   S701_TL_LOCATE1_ERR.Visu_Adv_Arr[15] := FALSE;
   S701_TL_LOCATE1_ERR.Visu_Ret_Arr[0] := FALSE;
   S701_TL_LOCATE1_ERR.Visu_Ret_Arr[1] := FALSE;
   S701_TL_LOCATE1_ERR.Visu_Ret_Arr[2] := FALSE;
   S701_TL_LOCATE1_ERR.Visu_Ret_Arr[3] := FALSE;
   S701_TL_LOCATE1_ERR.Visu_Ret_Arr[4] := FALSE;
   S701_TL_LOCATE1_ERR.Visu_Ret_Arr[5] := FALSE;
   S701_TL_LOCATE1_ERR.Visu_Ret_Arr[6] := FALSE;
   S701_TL_LOCATE1_ERR.Visu_Ret_Arr[7] := FALSE;
   S701_TL_LOCATE1_ERR.Visu_Ret_Arr[8] := FALSE;
   S701_TL_LOCATE1_ERR.Visu_Ret_Arr[9] := FALSE;
   S701_TL_LOCATE1_ERR.Visu_Ret_Arr[10] := FALSE;
   S701_TL_LOCATE1_ERR.Visu_Ret_Arr[11] := FALSE;
   S701_TL_LOCATE1_ERR.Visu_Ret_Arr[12] := FALSE;
   S701_TL_LOCATE1_ERR.Visu_Ret_Arr[13] := FALSE;
   S701_TL_LOCATE1_ERR.Visu_Ret_Arr[14] := FALSE;
   S701_TL_LOCATE1_ERR.Visu_Ret_Arr[15] := FALSE;
   S701_TL_LOCATE1_ERR.BLK_Move_Ret := 0;
   S701_TL_LOCATE1_ERR.Enable := FALSE;
   S701_TL_LOCATE1_ERR.Adv_End := FALSE;
   S701_TL_LOCATE1_ERR.Ret_End := FALSE;
   S701_TL_LOCATE2_ERR.Enable_Aux := FALSE;
   S701_TL_LOCATE2_ERR.Adv_Amount := 0;
   S701_TL_LOCATE2_ERR.Ret_Amount := 0;
   S701_TL_LOCATE2_ERR.LS_Adv1 := FALSE;
   S701_TL_LOCATE2_ERR.LS_Ret1 := FALSE;
   S701_TL_LOCATE2_ERR.LS_Adv2 := FALSE;
   S701_TL_LOCATE2_ERR.LS_Ret2 := FALSE;
   S701_TL_LOCATE2_ERR.LS_Adv3 := FALSE;
   S701_TL_LOCATE2_ERR.LS_Ret3 := FALSE;
   S701_TL_LOCATE2_ERR.LS_Adv4 := FALSE;
   S701_TL_LOCATE2_ERR.LS_Ret4 := FALSE;
   S701_TL_LOCATE2_ERR.SOL_Adv := FALSE;
   S701_TL_LOCATE2_ERR.SOL_Ret := FALSE;
   S701_TL_LOCATE2_ERR.M_Ready := FALSE;
   S701_TL_LOCATE2_ERR.T_CHK1 := T#0MS;
   S701_TL_LOCATE2_ERR.T_CHK2 := T#0MS;
   S701_TL_LOCATE2_ERR.PB_Lamp_CHK := FALSE;
   S701_TL_LOCATE2_ERR.PB_Error_Rst := FALSE;
   S701_TL_LOCATE2_ERR.M_FLICK := FALSE;
   S701_TL_LOCATE2_ERR.M_Adv_Err := FALSE;
   S701_TL_LOCATE2_ERR.M_Ret_Err := FALSE;
   S701_TL_LOCATE2_ERR.LP_Adv := FALSE;
   S701_TL_LOCATE2_ERR.LP_Ret := FALSE;
   S701_TL_LOCATE2_ERR.Visu_Adv := W#16#0;
   S701_TL_LOCATE2_ERR.Visu_Ret := W#16#0;
   S701_TL_LOCATE2_ERR.Error_T1.IN := FALSE;
   S701_TL_LOCATE2_ERR.Error_T1.PT := T#0MS;
   S701_TL_LOCATE2_ERR.Error_T1.Q := FALSE;
   S701_TL_LOCATE2_ERR.Error_T1.ET := T#0MS;
   S701_TL_LOCATE2_ERR.Error_T1.STATE := B#16#0;
   S701_TL_LOCATE2_ERR.Error_T1.STIME := T#0MS;
   S701_TL_LOCATE2_ERR.Error_T1.ATIME := T#0MS;
   S701_TL_LOCATE2_ERR.Error_T2.IN := FALSE;
   S701_TL_LOCATE2_ERR.Error_T2.PT := T#0MS;
   S701_TL_LOCATE2_ERR.Error_T2.Q := FALSE;
   S701_TL_LOCATE2_ERR.Error_T2.ET := T#0MS;
   S701_TL_LOCATE2_ERR.Error_T2.STATE := B#16#0;
   S701_TL_LOCATE2_ERR.Error_T2.STIME := T#0MS;
   S701_TL_LOCATE2_ERR.Error_T2.ATIME := T#0MS;
   S701_TL_LOCATE2_ERR.CHK_Aux1 := FALSE;
   S701_TL_LOCATE2_ERR.CHK_Aux2 := FALSE;
   S701_TL_LOCATE2_ERR.Error_T1_DN := FALSE;
   S701_TL_LOCATE2_ERR.Error_T2_DN := FALSE;
   S701_TL_LOCATE2_ERR.Adv_Memo := FALSE;
   S701_TL_LOCATE2_ERR.Visu_Adv_Arr[0] := FALSE;
   S701_TL_LOCATE2_ERR.Visu_Adv_Arr[1] := FALSE;
   S701_TL_LOCATE2_ERR.Visu_Adv_Arr[2] := FALSE;
   S701_TL_LOCATE2_ERR.Visu_Adv_Arr[3] := FALSE;
   S701_TL_LOCATE2_ERR.Visu_Adv_Arr[4] := FALSE;
   S701_TL_LOCATE2_ERR.Visu_Adv_Arr[5] := FALSE;
   S701_TL_LOCATE2_ERR.Visu_Adv_Arr[6] := FALSE;
   S701_TL_LOCATE2_ERR.Visu_Adv_Arr[7] := FALSE;
   S701_TL_LOCATE2_ERR.Visu_Adv_Arr[8] := FALSE;
   S701_TL_LOCATE2_ERR.Visu_Adv_Arr[9] := FALSE;
   S701_TL_LOCATE2_ERR.Visu_Adv_Arr[10] := FALSE;
   S701_TL_LOCATE2_ERR.Visu_Adv_Arr[11] := FALSE;
   S701_TL_LOCATE2_ERR.Visu_Adv_Arr[12] := FALSE;
   S701_TL_LOCATE2_ERR.Visu_Adv_Arr[13] := FALSE;
   S701_TL_LOCATE2_ERR.Visu_Adv_Arr[14] := FALSE;
   S701_TL_LOCATE2_ERR.Visu_Adv_Arr[15] := FALSE;
   S701_TL_LOCATE2_ERR.Visu_Ret_Arr[0] := FALSE;
   S701_TL_LOCATE2_ERR.Visu_Ret_Arr[1] := FALSE;
   S701_TL_LOCATE2_ERR.Visu_Ret_Arr[2] := FALSE;
   S701_TL_LOCATE2_ERR.Visu_Ret_Arr[3] := FALSE;
   S701_TL_LOCATE2_ERR.Visu_Ret_Arr[4] := FALSE;
   S701_TL_LOCATE2_ERR.Visu_Ret_Arr[5] := FALSE;
   S701_TL_LOCATE2_ERR.Visu_Ret_Arr[6] := FALSE;
   S701_TL_LOCATE2_ERR.Visu_Ret_Arr[7] := FALSE;
   S701_TL_LOCATE2_ERR.Visu_Ret_Arr[8] := FALSE;
   S701_TL_LOCATE2_ERR.Visu_Ret_Arr[9] := FALSE;
   S701_TL_LOCATE2_ERR.Visu_Ret_Arr[10] := FALSE;
   S701_TL_LOCATE2_ERR.Visu_Ret_Arr[11] := FALSE;
   S701_TL_LOCATE2_ERR.Visu_Ret_Arr[12] := FALSE;
   S701_TL_LOCATE2_ERR.Visu_Ret_Arr[13] := FALSE;
   S701_TL_LOCATE2_ERR.Visu_Ret_Arr[14] := FALSE;
   S701_TL_LOCATE2_ERR.Visu_Ret_Arr[15] := FALSE;
   S701_TL_LOCATE2_ERR.BLK_Move_Ret := 0;
   S701_TL_LOCATE2_ERR.Enable := FALSE;
   S701_TL_LOCATE2_ERR.Adv_End := FALSE;
   S701_TL_LOCATE2_ERR.Ret_End := FALSE;
   S701_TL_LOCATE3_ERR.Enable_Aux := FALSE;
   S701_TL_LOCATE3_ERR.Adv_Amount := 0;
   S701_TL_LOCATE3_ERR.Ret_Amount := 0;
   S701_TL_LOCATE3_ERR.LS_Adv1 := FALSE;
   S701_TL_LOCATE3_ERR.LS_Ret1 := FALSE;
   S701_TL_LOCATE3_ERR.LS_Adv2 := FALSE;
   S701_TL_LOCATE3_ERR.LS_Ret2 := FALSE;
   S701_TL_LOCATE3_ERR.LS_Adv3 := FALSE;
   S701_TL_LOCATE3_ERR.LS_Ret3 := FALSE;
   S701_TL_LOCATE3_ERR.LS_Adv4 := FALSE;
   S701_TL_LOCATE3_ERR.LS_Ret4 := FALSE;
   S701_TL_LOCATE3_ERR.SOL_Adv := FALSE;
   S701_TL_LOCATE3_ERR.SOL_Ret := FALSE;
   S701_TL_LOCATE3_ERR.M_Ready := FALSE;
   S701_TL_LOCATE3_ERR.T_CHK1 := T#0MS;
   S701_TL_LOCATE3_ERR.T_CHK2 := T#0MS;
   S701_TL_LOCATE3_ERR.PB_Lamp_CHK := FALSE;
   S701_TL_LOCATE3_ERR.PB_Error_Rst := FALSE;
   S701_TL_LOCATE3_ERR.M_FLICK := FALSE;
   S701_TL_LOCATE3_ERR.M_Adv_Err := FALSE;
   S701_TL_LOCATE3_ERR.M_Ret_Err := FALSE;
   S701_TL_LOCATE3_ERR.LP_Adv := FALSE;
   S701_TL_LOCATE3_ERR.LP_Ret := FALSE;
   S701_TL_LOCATE3_ERR.Visu_Adv := W#16#0;
   S701_TL_LOCATE3_ERR.Visu_Ret := W#16#0;
   S701_TL_LOCATE3_ERR.Error_T1.IN := FALSE;
   S701_TL_LOCATE3_ERR.Error_T1.PT := T#0MS;
   S701_TL_LOCATE3_ERR.Error_T1.Q := FALSE;
   S701_TL_LOCATE3_ERR.Error_T1.ET := T#0MS;
   S701_TL_LOCATE3_ERR.Error_T1.STATE := B#16#0;
   S701_TL_LOCATE3_ERR.Error_T1.STIME := T#0MS;
   S701_TL_LOCATE3_ERR.Error_T1.ATIME := T#0MS;
   S701_TL_LOCATE3_ERR.Error_T2.IN := FALSE;
   S701_TL_LOCATE3_ERR.Error_T2.PT := T#0MS;
   S701_TL_LOCATE3_ERR.Error_T2.Q := FALSE;
   S701_TL_LOCATE3_ERR.Error_T2.ET := T#0MS;
   S701_TL_LOCATE3_ERR.Error_T2.STATE := B#16#0;
   S701_TL_LOCATE3_ERR.Error_T2.STIME := T#0MS;
   S701_TL_LOCATE3_ERR.Error_T2.ATIME := T#0MS;
   S701_TL_LOCATE3_ERR.CHK_Aux1 := FALSE;
   S701_TL_LOCATE3_ERR.CHK_Aux2 := FALSE;
   S701_TL_LOCATE3_ERR.Error_T1_DN := FALSE;
   S701_TL_LOCATE3_ERR.Error_T2_DN := FALSE;
   S701_TL_LOCATE3_ERR.Adv_Memo := FALSE;
   S701_TL_LOCATE3_ERR.Visu_Adv_Arr[0] := FALSE;
   S701_TL_LOCATE3_ERR.Visu_Adv_Arr[1] := FALSE;
   S701_TL_LOCATE3_ERR.Visu_Adv_Arr[2] := FALSE;
   S701_TL_LOCATE3_ERR.Visu_Adv_Arr[3] := FALSE;
   S701_TL_LOCATE3_ERR.Visu_Adv_Arr[4] := FALSE;
   S701_TL_LOCATE3_ERR.Visu_Adv_Arr[5] := FALSE;
   S701_TL_LOCATE3_ERR.Visu_Adv_Arr[6] := FALSE;
   S701_TL_LOCATE3_ERR.Visu_Adv_Arr[7] := FALSE;
   S701_TL_LOCATE3_ERR.Visu_Adv_Arr[8] := FALSE;
   S701_TL_LOCATE3_ERR.Visu_Adv_Arr[9] := FALSE;
   S701_TL_LOCATE3_ERR.Visu_Adv_Arr[10] := FALSE;
   S701_TL_LOCATE3_ERR.Visu_Adv_Arr[11] := FALSE;
   S701_TL_LOCATE3_ERR.Visu_Adv_Arr[12] := FALSE;
   S701_TL_LOCATE3_ERR.Visu_Adv_Arr[13] := FALSE;
   S701_TL_LOCATE3_ERR.Visu_Adv_Arr[14] := FALSE;
   S701_TL_LOCATE3_ERR.Visu_Adv_Arr[15] := FALSE;
   S701_TL_LOCATE3_ERR.Visu_Ret_Arr[0] := FALSE;
   S701_TL_LOCATE3_ERR.Visu_Ret_Arr[1] := FALSE;
   S701_TL_LOCATE3_ERR.Visu_Ret_Arr[2] := FALSE;
   S701_TL_LOCATE3_ERR.Visu_Ret_Arr[3] := FALSE;
   S701_TL_LOCATE3_ERR.Visu_Ret_Arr[4] := FALSE;
   S701_TL_LOCATE3_ERR.Visu_Ret_Arr[5] := FALSE;
   S701_TL_LOCATE3_ERR.Visu_Ret_Arr[6] := FALSE;
   S701_TL_LOCATE3_ERR.Visu_Ret_Arr[7] := FALSE;
   S701_TL_LOCATE3_ERR.Visu_Ret_Arr[8] := FALSE;
   S701_TL_LOCATE3_ERR.Visu_Ret_Arr[9] := FALSE;
   S701_TL_LOCATE3_ERR.Visu_Ret_Arr[10] := FALSE;
   S701_TL_LOCATE3_ERR.Visu_Ret_Arr[11] := FALSE;
   S701_TL_LOCATE3_ERR.Visu_Ret_Arr[12] := FALSE;
   S701_TL_LOCATE3_ERR.Visu_Ret_Arr[13] := FALSE;
   S701_TL_LOCATE3_ERR.Visu_Ret_Arr[14] := FALSE;
   S701_TL_LOCATE3_ERR.Visu_Ret_Arr[15] := FALSE;
   S701_TL_LOCATE3_ERR.BLK_Move_Ret := 0;
   S701_TL_LOCATE3_ERR.Enable := FALSE;
   S701_TL_LOCATE3_ERR.Adv_End := FALSE;
   S701_TL_LOCATE3_ERR.Ret_End := FALSE;
   S701_TL_1_CLAMP1_ERR.Enable_Aux := FALSE;
   S701_TL_1_CLAMP1_ERR.Adv_Amount := 0;
   S701_TL_1_CLAMP1_ERR.Ret_Amount := 0;
   S701_TL_1_CLAMP1_ERR.LS_Adv1 := FALSE;
   S701_TL_1_CLAMP1_ERR.LS_Ret1 := FALSE;
   S701_TL_1_CLAMP1_ERR.LS_Adv2 := FALSE;
   S701_TL_1_CLAMP1_ERR.LS_Ret2 := FALSE;
   S701_TL_1_CLAMP1_ERR.LS_Adv3 := FALSE;
   S701_TL_1_CLAMP1_ERR.LS_Ret3 := FALSE;
   S701_TL_1_CLAMP1_ERR.LS_Adv4 := FALSE;
   S701_TL_1_CLAMP1_ERR.LS_Ret4 := FALSE;
   S701_TL_1_CLAMP1_ERR.LS_Adv5 := FALSE;
   S701_TL_1_CLAMP1_ERR.LS_Ret5 := FALSE;
   S701_TL_1_CLAMP1_ERR.LS_Adv6 := FALSE;
   S701_TL_1_CLAMP1_ERR.LS_Ret6 := FALSE;
   S701_TL_1_CLAMP1_ERR.LS_Adv7 := FALSE;
   S701_TL_1_CLAMP1_ERR.LS_Ret7 := FALSE;
   S701_TL_1_CLAMP1_ERR.LS_Adv8 := FALSE;
   S701_TL_1_CLAMP1_ERR.LS_Ret8 := FALSE;
   S701_TL_1_CLAMP1_ERR.SOL_Adv := FALSE;
   S701_TL_1_CLAMP1_ERR.SOL_Ret := FALSE;
   S701_TL_1_CLAMP1_ERR.M_Ready := FALSE;
   S701_TL_1_CLAMP1_ERR.T_CHK1 := T#0MS;
   S701_TL_1_CLAMP1_ERR.T_CHK2 := T#0MS;
   S701_TL_1_CLAMP1_ERR.PB_Lamp_CHK := FALSE;
   S701_TL_1_CLAMP1_ERR.PB_Error_Rst := FALSE;
   S701_TL_1_CLAMP1_ERR.M_FLICK := FALSE;
   S701_TL_1_CLAMP1_ERR.M_Adv_Err := FALSE;
   S701_TL_1_CLAMP1_ERR.M_Ret_Err := FALSE;
   S701_TL_1_CLAMP1_ERR.LP_Adv := FALSE;
   S701_TL_1_CLAMP1_ERR.LP_Ret := FALSE;
   S701_TL_1_CLAMP1_ERR.Visu_Adv := W#16#0;
   S701_TL_1_CLAMP1_ERR.Visu_Ret := W#16#0;
   S701_TL_1_CLAMP1_ERR.Error_T1.IN := FALSE;
   S701_TL_1_CLAMP1_ERR.Error_T1.PT := T#0MS;
   S701_TL_1_CLAMP1_ERR.Error_T1.Q := FALSE;
   S701_TL_1_CLAMP1_ERR.Error_T1.ET := T#0MS;
   S701_TL_1_CLAMP1_ERR.Error_T1.STATE := B#16#0;
   S701_TL_1_CLAMP1_ERR.Error_T1.STIME := T#0MS;
   S701_TL_1_CLAMP1_ERR.Error_T1.ATIME := T#0MS;
   S701_TL_1_CLAMP1_ERR.Error_T2.IN := FALSE;
   S701_TL_1_CLAMP1_ERR.Error_T2.PT := T#0MS;
   S701_TL_1_CLAMP1_ERR.Error_T2.Q := FALSE;
   S701_TL_1_CLAMP1_ERR.Error_T2.ET := T#0MS;
   S701_TL_1_CLAMP1_ERR.Error_T2.STATE := B#16#0;
   S701_TL_1_CLAMP1_ERR.Error_T2.STIME := T#0MS;
   S701_TL_1_CLAMP1_ERR.Error_T2.ATIME := T#0MS;
   S701_TL_1_CLAMP1_ERR.Adv_End_Aux := FALSE;
   S701_TL_1_CLAMP1_ERR.Ret_End_Aux := FALSE;
   S701_TL_1_CLAMP1_ERR.CHK_Aux1 := FALSE;
   S701_TL_1_CLAMP1_ERR.CHK_Aux2 := FALSE;
   S701_TL_1_CLAMP1_ERR.Error_T1_DN := FALSE;
   S701_TL_1_CLAMP1_ERR.Error_T2_DN := FALSE;
   S701_TL_1_CLAMP1_ERR.Adv_Memo := FALSE;
   S701_TL_1_CLAMP1_ERR.Visu_Adv_Arr[0] := FALSE;
   S701_TL_1_CLAMP1_ERR.Visu_Adv_Arr[1] := FALSE;
   S701_TL_1_CLAMP1_ERR.Visu_Adv_Arr[2] := FALSE;
   S701_TL_1_CLAMP1_ERR.Visu_Adv_Arr[3] := FALSE;
   S701_TL_1_CLAMP1_ERR.Visu_Adv_Arr[4] := FALSE;
   S701_TL_1_CLAMP1_ERR.Visu_Adv_Arr[5] := FALSE;
   S701_TL_1_CLAMP1_ERR.Visu_Adv_Arr[6] := FALSE;
   S701_TL_1_CLAMP1_ERR.Visu_Adv_Arr[7] := FALSE;
   S701_TL_1_CLAMP1_ERR.Visu_Adv_Arr[8] := FALSE;
   S701_TL_1_CLAMP1_ERR.Visu_Adv_Arr[9] := FALSE;
   S701_TL_1_CLAMP1_ERR.Visu_Adv_Arr[10] := FALSE;
   S701_TL_1_CLAMP1_ERR.Visu_Adv_Arr[11] := FALSE;
   S701_TL_1_CLAMP1_ERR.Visu_Adv_Arr[12] := FALSE;
   S701_TL_1_CLAMP1_ERR.Visu_Adv_Arr[13] := FALSE;
   S701_TL_1_CLAMP1_ERR.Visu_Adv_Arr[14] := FALSE;
   S701_TL_1_CLAMP1_ERR.Visu_Adv_Arr[15] := FALSE;
   S701_TL_1_CLAMP1_ERR.Visu_Ret_Arr[0] := FALSE;
   S701_TL_1_CLAMP1_ERR.Visu_Ret_Arr[1] := FALSE;
   S701_TL_1_CLAMP1_ERR.Visu_Ret_Arr[2] := FALSE;
   S701_TL_1_CLAMP1_ERR.Visu_Ret_Arr[3] := FALSE;
   S701_TL_1_CLAMP1_ERR.Visu_Ret_Arr[4] := FALSE;
   S701_TL_1_CLAMP1_ERR.Visu_Ret_Arr[5] := FALSE;
   S701_TL_1_CLAMP1_ERR.Visu_Ret_Arr[6] := FALSE;
   S701_TL_1_CLAMP1_ERR.Visu_Ret_Arr[7] := FALSE;
   S701_TL_1_CLAMP1_ERR.Visu_Ret_Arr[8] := FALSE;
   S701_TL_1_CLAMP1_ERR.Visu_Ret_Arr[9] := FALSE;
   S701_TL_1_CLAMP1_ERR.Visu_Ret_Arr[10] := FALSE;
   S701_TL_1_CLAMP1_ERR.Visu_Ret_Arr[11] := FALSE;
   S701_TL_1_CLAMP1_ERR.Visu_Ret_Arr[12] := FALSE;
   S701_TL_1_CLAMP1_ERR.Visu_Ret_Arr[13] := FALSE;
   S701_TL_1_CLAMP1_ERR.Visu_Ret_Arr[14] := FALSE;
   S701_TL_1_CLAMP1_ERR.Visu_Ret_Arr[15] := FALSE;
   S701_TL_1_CLAMP1_ERR.BLK_Move_Ret := 0;
   S701_TL_1_CLAMP1_ERR.Enable := FALSE;
   S701_TL_1_CLAMP1_ERR.Adv_End := FALSE;
   S701_TL_1_CLAMP1_ERR.Ret_End := FALSE;
   S701_TL_1_CLAMP2_ERR.Enable_Aux := FALSE;
   S701_TL_1_CLAMP2_ERR.Adv_Amount := 0;
   S701_TL_1_CLAMP2_ERR.Ret_Amount := 0;
   S701_TL_1_CLAMP2_ERR.LS_Adv1 := FALSE;
   S701_TL_1_CLAMP2_ERR.LS_Ret1 := FALSE;
   S701_TL_1_CLAMP2_ERR.LS_Adv2 := FALSE;
   S701_TL_1_CLAMP2_ERR.LS_Ret2 := FALSE;
   S701_TL_1_CLAMP2_ERR.LS_Adv3 := FALSE;
   S701_TL_1_CLAMP2_ERR.LS_Ret3 := FALSE;
   S701_TL_1_CLAMP2_ERR.LS_Adv4 := FALSE;
   S701_TL_1_CLAMP2_ERR.LS_Ret4 := FALSE;
   S701_TL_1_CLAMP2_ERR.LS_Adv5 := FALSE;
   S701_TL_1_CLAMP2_ERR.LS_Ret5 := FALSE;
   S701_TL_1_CLAMP2_ERR.LS_Adv6 := FALSE;
   S701_TL_1_CLAMP2_ERR.LS_Ret6 := FALSE;
   S701_TL_1_CLAMP2_ERR.LS_Adv7 := FALSE;
   S701_TL_1_CLAMP2_ERR.LS_Ret7 := FALSE;
   S701_TL_1_CLAMP2_ERR.LS_Adv8 := FALSE;
   S701_TL_1_CLAMP2_ERR.LS_Ret8 := FALSE;
   S701_TL_1_CLAMP2_ERR.SOL_Adv := FALSE;
   S701_TL_1_CLAMP2_ERR.SOL_Ret := FALSE;
   S701_TL_1_CLAMP2_ERR.M_Ready := FALSE;
   S701_TL_1_CLAMP2_ERR.T_CHK1 := T#0MS;
   S701_TL_1_CLAMP2_ERR.T_CHK2 := T#0MS;
   S701_TL_1_CLAMP2_ERR.PB_Lamp_CHK := FALSE;
   S701_TL_1_CLAMP2_ERR.PB_Error_Rst := FALSE;
   S701_TL_1_CLAMP2_ERR.M_FLICK := FALSE;
   S701_TL_1_CLAMP2_ERR.M_Adv_Err := FALSE;
   S701_TL_1_CLAMP2_ERR.M_Ret_Err := FALSE;
   S701_TL_1_CLAMP2_ERR.LP_Adv := FALSE;
   S701_TL_1_CLAMP2_ERR.LP_Ret := FALSE;
   S701_TL_1_CLAMP2_ERR.Visu_Adv := W#16#0;
   S701_TL_1_CLAMP2_ERR.Visu_Ret := W#16#0;
   S701_TL_1_CLAMP2_ERR.Error_T1.IN := FALSE;
   S701_TL_1_CLAMP2_ERR.Error_T1.PT := T#0MS;
   S701_TL_1_CLAMP2_ERR.Error_T1.Q := FALSE;
   S701_TL_1_CLAMP2_ERR.Error_T1.ET := T#0MS;
   S701_TL_1_CLAMP2_ERR.Error_T1.STATE := B#16#0;
   S701_TL_1_CLAMP2_ERR.Error_T1.STIME := T#0MS;
   S701_TL_1_CLAMP2_ERR.Error_T1.ATIME := T#0MS;
   S701_TL_1_CLAMP2_ERR.Error_T2.IN := FALSE;
   S701_TL_1_CLAMP2_ERR.Error_T2.PT := T#0MS;
   S701_TL_1_CLAMP2_ERR.Error_T2.Q := FALSE;
   S701_TL_1_CLAMP2_ERR.Error_T2.ET := T#0MS;
   S701_TL_1_CLAMP2_ERR.Error_T2.STATE := B#16#0;
   S701_TL_1_CLAMP2_ERR.Error_T2.STIME := T#0MS;
   S701_TL_1_CLAMP2_ERR.Error_T2.ATIME := T#0MS;
   S701_TL_1_CLAMP2_ERR.Adv_End_Aux := FALSE;
   S701_TL_1_CLAMP2_ERR.Ret_End_Aux := FALSE;
   S701_TL_1_CLAMP2_ERR.CHK_Aux1 := FALSE;
   S701_TL_1_CLAMP2_ERR.CHK_Aux2 := FALSE;
   S701_TL_1_CLAMP2_ERR.Error_T1_DN := FALSE;
   S701_TL_1_CLAMP2_ERR.Error_T2_DN := FALSE;
   S701_TL_1_CLAMP2_ERR.Adv_Memo := FALSE;
   S701_TL_1_CLAMP2_ERR.Visu_Adv_Arr[0] := FALSE;
   S701_TL_1_CLAMP2_ERR.Visu_Adv_Arr[1] := FALSE;
   S701_TL_1_CLAMP2_ERR.Visu_Adv_Arr[2] := FALSE;
   S701_TL_1_CLAMP2_ERR.Visu_Adv_Arr[3] := FALSE;
   S701_TL_1_CLAMP2_ERR.Visu_Adv_Arr[4] := FALSE;
   S701_TL_1_CLAMP2_ERR.Visu_Adv_Arr[5] := FALSE;
   S701_TL_1_CLAMP2_ERR.Visu_Adv_Arr[6] := FALSE;
   S701_TL_1_CLAMP2_ERR.Visu_Adv_Arr[7] := FALSE;
   S701_TL_1_CLAMP2_ERR.Visu_Adv_Arr[8] := FALSE;
   S701_TL_1_CLAMP2_ERR.Visu_Adv_Arr[9] := FALSE;
   S701_TL_1_CLAMP2_ERR.Visu_Adv_Arr[10] := FALSE;
   S701_TL_1_CLAMP2_ERR.Visu_Adv_Arr[11] := FALSE;
   S701_TL_1_CLAMP2_ERR.Visu_Adv_Arr[12] := FALSE;
   S701_TL_1_CLAMP2_ERR.Visu_Adv_Arr[13] := FALSE;
   S701_TL_1_CLAMP2_ERR.Visu_Adv_Arr[14] := FALSE;
   S701_TL_1_CLAMP2_ERR.Visu_Adv_Arr[15] := FALSE;
   S701_TL_1_CLAMP2_ERR.Visu_Ret_Arr[0] := FALSE;
   S701_TL_1_CLAMP2_ERR.Visu_Ret_Arr[1] := FALSE;
   S701_TL_1_CLAMP2_ERR.Visu_Ret_Arr[2] := FALSE;
   S701_TL_1_CLAMP2_ERR.Visu_Ret_Arr[3] := FALSE;
   S701_TL_1_CLAMP2_ERR.Visu_Ret_Arr[4] := FALSE;
   S701_TL_1_CLAMP2_ERR.Visu_Ret_Arr[5] := FALSE;
   S701_TL_1_CLAMP2_ERR.Visu_Ret_Arr[6] := FALSE;
   S701_TL_1_CLAMP2_ERR.Visu_Ret_Arr[7] := FALSE;
   S701_TL_1_CLAMP2_ERR.Visu_Ret_Arr[8] := FALSE;
   S701_TL_1_CLAMP2_ERR.Visu_Ret_Arr[9] := FALSE;
   S701_TL_1_CLAMP2_ERR.Visu_Ret_Arr[10] := FALSE;
   S701_TL_1_CLAMP2_ERR.Visu_Ret_Arr[11] := FALSE;
   S701_TL_1_CLAMP2_ERR.Visu_Ret_Arr[12] := FALSE;
   S701_TL_1_CLAMP2_ERR.Visu_Ret_Arr[13] := FALSE;
   S701_TL_1_CLAMP2_ERR.Visu_Ret_Arr[14] := FALSE;
   S701_TL_1_CLAMP2_ERR.Visu_Ret_Arr[15] := FALSE;
   S701_TL_1_CLAMP2_ERR.BLK_Move_Ret := 0;
   S701_TL_1_CLAMP2_ERR.Enable := FALSE;
   S701_TL_1_CLAMP2_ERR.Adv_End := FALSE;
   S701_TL_1_CLAMP2_ERR.Ret_End := FALSE;
   S701_TL_2_CLAMP_ERR.Enable_Aux := FALSE;
   S701_TL_2_CLAMP_ERR.Adv_Amount := 0;
   S701_TL_2_CLAMP_ERR.Ret_Amount := 0;
   S701_TL_2_CLAMP_ERR.LS_Adv1 := FALSE;
   S701_TL_2_CLAMP_ERR.LS_Ret1 := FALSE;
   S701_TL_2_CLAMP_ERR.LS_Adv2 := FALSE;
   S701_TL_2_CLAMP_ERR.LS_Ret2 := FALSE;
   S701_TL_2_CLAMP_ERR.LS_Adv3 := FALSE;
   S701_TL_2_CLAMP_ERR.LS_Ret3 := FALSE;
   S701_TL_2_CLAMP_ERR.LS_Adv4 := FALSE;
   S701_TL_2_CLAMP_ERR.LS_Ret4 := FALSE;
   S701_TL_2_CLAMP_ERR.LS_Adv5 := FALSE;
   S701_TL_2_CLAMP_ERR.LS_Ret5 := FALSE;
   S701_TL_2_CLAMP_ERR.LS_Adv6 := FALSE;
   S701_TL_2_CLAMP_ERR.LS_Ret6 := FALSE;
   S701_TL_2_CLAMP_ERR.LS_Adv7 := FALSE;
   S701_TL_2_CLAMP_ERR.LS_Ret7 := FALSE;
   S701_TL_2_CLAMP_ERR.LS_Adv8 := FALSE;
   S701_TL_2_CLAMP_ERR.LS_Ret8 := FALSE;
   S701_TL_2_CLAMP_ERR.SOL_Adv := FALSE;
   S701_TL_2_CLAMP_ERR.SOL_Ret := FALSE;
   S701_TL_2_CLAMP_ERR.M_Ready := FALSE;
   S701_TL_2_CLAMP_ERR.T_CHK1 := T#0MS;
   S701_TL_2_CLAMP_ERR.T_CHK2 := T#0MS;
   S701_TL_2_CLAMP_ERR.PB_Lamp_CHK := FALSE;
   S701_TL_2_CLAMP_ERR.PB_Error_Rst := FALSE;
   S701_TL_2_CLAMP_ERR.M_FLICK := FALSE;
   S701_TL_2_CLAMP_ERR.M_Adv_Err := FALSE;
   S701_TL_2_CLAMP_ERR.M_Ret_Err := FALSE;
   S701_TL_2_CLAMP_ERR.LP_Adv := FALSE;
   S701_TL_2_CLAMP_ERR.LP_Ret := FALSE;
   S701_TL_2_CLAMP_ERR.Visu_Adv := W#16#0;
   S701_TL_2_CLAMP_ERR.Visu_Ret := W#16#0;
   S701_TL_2_CLAMP_ERR.Error_T1.IN := FALSE;
   S701_TL_2_CLAMP_ERR.Error_T1.PT := T#0MS;
   S701_TL_2_CLAMP_ERR.Error_T1.Q := FALSE;
   S701_TL_2_CLAMP_ERR.Error_T1.ET := T#0MS;
   S701_TL_2_CLAMP_ERR.Error_T1.STATE := B#16#0;
   S701_TL_2_CLAMP_ERR.Error_T1.STIME := T#0MS;
   S701_TL_2_CLAMP_ERR.Error_T1.ATIME := T#0MS;
   S701_TL_2_CLAMP_ERR.Error_T2.IN := FALSE;
   S701_TL_2_CLAMP_ERR.Error_T2.PT := T#0MS;
   S701_TL_2_CLAMP_ERR.Error_T2.Q := FALSE;
   S701_TL_2_CLAMP_ERR.Error_T2.ET := T#0MS;
   S701_TL_2_CLAMP_ERR.Error_T2.STATE := B#16#0;
   S701_TL_2_CLAMP_ERR.Error_T2.STIME := T#0MS;
   S701_TL_2_CLAMP_ERR.Error_T2.ATIME := T#0MS;
   S701_TL_2_CLAMP_ERR.Adv_End_Aux := FALSE;
   S701_TL_2_CLAMP_ERR.Ret_End_Aux := FALSE;
   S701_TL_2_CLAMP_ERR.CHK_Aux1 := FALSE;
   S701_TL_2_CLAMP_ERR.CHK_Aux2 := FALSE;
   S701_TL_2_CLAMP_ERR.Error_T1_DN := FALSE;
   S701_TL_2_CLAMP_ERR.Error_T2_DN := FALSE;
   S701_TL_2_CLAMP_ERR.Adv_Memo := FALSE;
   S701_TL_2_CLAMP_ERR.Visu_Adv_Arr[0] := FALSE;
   S701_TL_2_CLAMP_ERR.Visu_Adv_Arr[1] := FALSE;
   S701_TL_2_CLAMP_ERR.Visu_Adv_Arr[2] := FALSE;
   S701_TL_2_CLAMP_ERR.Visu_Adv_Arr[3] := FALSE;
   S701_TL_2_CLAMP_ERR.Visu_Adv_Arr[4] := FALSE;
   S701_TL_2_CLAMP_ERR.Visu_Adv_Arr[5] := FALSE;
   S701_TL_2_CLAMP_ERR.Visu_Adv_Arr[6] := FALSE;
   S701_TL_2_CLAMP_ERR.Visu_Adv_Arr[7] := FALSE;
   S701_TL_2_CLAMP_ERR.Visu_Adv_Arr[8] := FALSE;
   S701_TL_2_CLAMP_ERR.Visu_Adv_Arr[9] := FALSE;
   S701_TL_2_CLAMP_ERR.Visu_Adv_Arr[10] := FALSE;
   S701_TL_2_CLAMP_ERR.Visu_Adv_Arr[11] := FALSE;
   S701_TL_2_CLAMP_ERR.Visu_Adv_Arr[12] := FALSE;
   S701_TL_2_CLAMP_ERR.Visu_Adv_Arr[13] := FALSE;
   S701_TL_2_CLAMP_ERR.Visu_Adv_Arr[14] := FALSE;
   S701_TL_2_CLAMP_ERR.Visu_Adv_Arr[15] := FALSE;
   S701_TL_2_CLAMP_ERR.Visu_Ret_Arr[0] := FALSE;
   S701_TL_2_CLAMP_ERR.Visu_Ret_Arr[1] := FALSE;
   S701_TL_2_CLAMP_ERR.Visu_Ret_Arr[2] := FALSE;
   S701_TL_2_CLAMP_ERR.Visu_Ret_Arr[3] := FALSE;
   S701_TL_2_CLAMP_ERR.Visu_Ret_Arr[4] := FALSE;
   S701_TL_2_CLAMP_ERR.Visu_Ret_Arr[5] := FALSE;
   S701_TL_2_CLAMP_ERR.Visu_Ret_Arr[6] := FALSE;
   S701_TL_2_CLAMP_ERR.Visu_Ret_Arr[7] := FALSE;
   S701_TL_2_CLAMP_ERR.Visu_Ret_Arr[8] := FALSE;
   S701_TL_2_CLAMP_ERR.Visu_Ret_Arr[9] := FALSE;
   S701_TL_2_CLAMP_ERR.Visu_Ret_Arr[10] := FALSE;
   S701_TL_2_CLAMP_ERR.Visu_Ret_Arr[11] := FALSE;
   S701_TL_2_CLAMP_ERR.Visu_Ret_Arr[12] := FALSE;
   S701_TL_2_CLAMP_ERR.Visu_Ret_Arr[13] := FALSE;
   S701_TL_2_CLAMP_ERR.Visu_Ret_Arr[14] := FALSE;
   S701_TL_2_CLAMP_ERR.Visu_Ret_Arr[15] := FALSE;
   S701_TL_2_CLAMP_ERR.BLK_Move_Ret := 0;
   S701_TL_2_CLAMP_ERR.Enable := FALSE;
   S701_TL_2_CLAMP_ERR.Adv_End := FALSE;
   S701_TL_2_CLAMP_ERR.Ret_End := FALSE;
   S701_TL_3_CLAMP_ERR.Enable_Aux := FALSE;
   S701_TL_3_CLAMP_ERR.Adv_Amount := 0;
   S701_TL_3_CLAMP_ERR.Ret_Amount := 0;
   S701_TL_3_CLAMP_ERR.LS_Adv1 := FALSE;
   S701_TL_3_CLAMP_ERR.LS_Ret1 := FALSE;
   S701_TL_3_CLAMP_ERR.LS_Adv2 := FALSE;
   S701_TL_3_CLAMP_ERR.LS_Ret2 := FALSE;
   S701_TL_3_CLAMP_ERR.LS_Adv3 := FALSE;
   S701_TL_3_CLAMP_ERR.LS_Ret3 := FALSE;
   S701_TL_3_CLAMP_ERR.LS_Adv4 := FALSE;
   S701_TL_3_CLAMP_ERR.LS_Ret4 := FALSE;
   S701_TL_3_CLAMP_ERR.LS_Adv5 := FALSE;
   S701_TL_3_CLAMP_ERR.LS_Ret5 := FALSE;
   S701_TL_3_CLAMP_ERR.LS_Adv6 := FALSE;
   S701_TL_3_CLAMP_ERR.LS_Ret6 := FALSE;
   S701_TL_3_CLAMP_ERR.LS_Adv7 := FALSE;
   S701_TL_3_CLAMP_ERR.LS_Ret7 := FALSE;
   S701_TL_3_CLAMP_ERR.LS_Adv8 := FALSE;
   S701_TL_3_CLAMP_ERR.LS_Ret8 := FALSE;
   S701_TL_3_CLAMP_ERR.SOL_Adv := FALSE;
   S701_TL_3_CLAMP_ERR.SOL_Ret := FALSE;
   S701_TL_3_CLAMP_ERR.M_Ready := FALSE;
   S701_TL_3_CLAMP_ERR.T_CHK1 := T#0MS;
   S701_TL_3_CLAMP_ERR.T_CHK2 := T#0MS;
   S701_TL_3_CLAMP_ERR.PB_Lamp_CHK := FALSE;
   S701_TL_3_CLAMP_ERR.PB_Error_Rst := FALSE;
   S701_TL_3_CLAMP_ERR.M_FLICK := FALSE;
   S701_TL_3_CLAMP_ERR.M_Adv_Err := FALSE;
   S701_TL_3_CLAMP_ERR.M_Ret_Err := FALSE;
   S701_TL_3_CLAMP_ERR.LP_Adv := FALSE;
   S701_TL_3_CLAMP_ERR.LP_Ret := FALSE;
   S701_TL_3_CLAMP_ERR.Visu_Adv := W#16#0;
   S701_TL_3_CLAMP_ERR.Visu_Ret := W#16#0;
   S701_TL_3_CLAMP_ERR.Error_T1.IN := FALSE;
   S701_TL_3_CLAMP_ERR.Error_T1.PT := T#0MS;
   S701_TL_3_CLAMP_ERR.Error_T1.Q := FALSE;
   S701_TL_3_CLAMP_ERR.Error_T1.ET := T#0MS;
   S701_TL_3_CLAMP_ERR.Error_T1.STATE := B#16#0;
   S701_TL_3_CLAMP_ERR.Error_T1.STIME := T#0MS;
   S701_TL_3_CLAMP_ERR.Error_T1.ATIME := T#0MS;
   S701_TL_3_CLAMP_ERR.Error_T2.IN := FALSE;
   S701_TL_3_CLAMP_ERR.Error_T2.PT := T#0MS;
   S701_TL_3_CLAMP_ERR.Error_T2.Q := FALSE;
   S701_TL_3_CLAMP_ERR.Error_T2.ET := T#0MS;
   S701_TL_3_CLAMP_ERR.Error_T2.STATE := B#16#0;
   S701_TL_3_CLAMP_ERR.Error_T2.STIME := T#0MS;
   S701_TL_3_CLAMP_ERR.Error_T2.ATIME := T#0MS;
   S701_TL_3_CLAMP_ERR.Adv_End_Aux := FALSE;
   S701_TL_3_CLAMP_ERR.Ret_End_Aux := FALSE;
   S701_TL_3_CLAMP_ERR.CHK_Aux1 := FALSE;
   S701_TL_3_CLAMP_ERR.CHK_Aux2 := FALSE;
   S701_TL_3_CLAMP_ERR.Error_T1_DN := FALSE;
   S701_TL_3_CLAMP_ERR.Error_T2_DN := FALSE;
   S701_TL_3_CLAMP_ERR.Adv_Memo := FALSE;
   S701_TL_3_CLAMP_ERR.Visu_Adv_Arr[0] := FALSE;
   S701_TL_3_CLAMP_ERR.Visu_Adv_Arr[1] := FALSE;
   S701_TL_3_CLAMP_ERR.Visu_Adv_Arr[2] := FALSE;
   S701_TL_3_CLAMP_ERR.Visu_Adv_Arr[3] := FALSE;
   S701_TL_3_CLAMP_ERR.Visu_Adv_Arr[4] := FALSE;
   S701_TL_3_CLAMP_ERR.Visu_Adv_Arr[5] := FALSE;
   S701_TL_3_CLAMP_ERR.Visu_Adv_Arr[6] := FALSE;
   S701_TL_3_CLAMP_ERR.Visu_Adv_Arr[7] := FALSE;
   S701_TL_3_CLAMP_ERR.Visu_Adv_Arr[8] := FALSE;
   S701_TL_3_CLAMP_ERR.Visu_Adv_Arr[9] := FALSE;
   S701_TL_3_CLAMP_ERR.Visu_Adv_Arr[10] := FALSE;
   S701_TL_3_CLAMP_ERR.Visu_Adv_Arr[11] := FALSE;
   S701_TL_3_CLAMP_ERR.Visu_Adv_Arr[12] := FALSE;
   S701_TL_3_CLAMP_ERR.Visu_Adv_Arr[13] := FALSE;
   S701_TL_3_CLAMP_ERR.Visu_Adv_Arr[14] := FALSE;
   S701_TL_3_CLAMP_ERR.Visu_Adv_Arr[15] := FALSE;
   S701_TL_3_CLAMP_ERR.Visu_Ret_Arr[0] := FALSE;
   S701_TL_3_CLAMP_ERR.Visu_Ret_Arr[1] := FALSE;
   S701_TL_3_CLAMP_ERR.Visu_Ret_Arr[2] := FALSE;
   S701_TL_3_CLAMP_ERR.Visu_Ret_Arr[3] := FALSE;
   S701_TL_3_CLAMP_ERR.Visu_Ret_Arr[4] := FALSE;
   S701_TL_3_CLAMP_ERR.Visu_Ret_Arr[5] := FALSE;
   S701_TL_3_CLAMP_ERR.Visu_Ret_Arr[6] := FALSE;
   S701_TL_3_CLAMP_ERR.Visu_Ret_Arr[7] := FALSE;
   S701_TL_3_CLAMP_ERR.Visu_Ret_Arr[8] := FALSE;
   S701_TL_3_CLAMP_ERR.Visu_Ret_Arr[9] := FALSE;
   S701_TL_3_CLAMP_ERR.Visu_Ret_Arr[10] := FALSE;
   S701_TL_3_CLAMP_ERR.Visu_Ret_Arr[11] := FALSE;
   S701_TL_3_CLAMP_ERR.Visu_Ret_Arr[12] := FALSE;
   S701_TL_3_CLAMP_ERR.Visu_Ret_Arr[13] := FALSE;
   S701_TL_3_CLAMP_ERR.Visu_Ret_Arr[14] := FALSE;
   S701_TL_3_CLAMP_ERR.Visu_Ret_Arr[15] := FALSE;
   S701_TL_3_CLAMP_ERR.BLK_Move_Ret := 0;
   S701_TL_3_CLAMP_ERR.Enable := FALSE;
   S701_TL_3_CLAMP_ERR.Adv_End := FALSE;
   S701_TL_3_CLAMP_ERR.Ret_End := FALSE;
   S701_TL_4_CLAMP_ERR.Enable_Aux := FALSE;
   S701_TL_4_CLAMP_ERR.Adv_Amount := 0;
   S701_TL_4_CLAMP_ERR.Ret_Amount := 0;
   S701_TL_4_CLAMP_ERR.LS_Adv1 := FALSE;
   S701_TL_4_CLAMP_ERR.LS_Ret1 := FALSE;
   S701_TL_4_CLAMP_ERR.LS_Adv2 := FALSE;
   S701_TL_4_CLAMP_ERR.LS_Ret2 := FALSE;
   S701_TL_4_CLAMP_ERR.LS_Adv3 := FALSE;
   S701_TL_4_CLAMP_ERR.LS_Ret3 := FALSE;
   S701_TL_4_CLAMP_ERR.LS_Adv4 := FALSE;
   S701_TL_4_CLAMP_ERR.LS_Ret4 := FALSE;
   S701_TL_4_CLAMP_ERR.LS_Adv5 := FALSE;
   S701_TL_4_CLAMP_ERR.LS_Ret5 := FALSE;
   S701_TL_4_CLAMP_ERR.LS_Adv6 := FALSE;
   S701_TL_4_CLAMP_ERR.LS_Ret6 := FALSE;
   S701_TL_4_CLAMP_ERR.LS_Adv7 := FALSE;
   S701_TL_4_CLAMP_ERR.LS_Ret7 := FALSE;
   S701_TL_4_CLAMP_ERR.LS_Adv8 := FALSE;
   S701_TL_4_CLAMP_ERR.LS_Ret8 := FALSE;
   S701_TL_4_CLAMP_ERR.SOL_Adv := FALSE;
   S701_TL_4_CLAMP_ERR.SOL_Ret := FALSE;
   S701_TL_4_CLAMP_ERR.M_Ready := FALSE;
   S701_TL_4_CLAMP_ERR.T_CHK1 := T#0MS;
   S701_TL_4_CLAMP_ERR.T_CHK2 := T#0MS;
   S701_TL_4_CLAMP_ERR.PB_Lamp_CHK := FALSE;
   S701_TL_4_CLAMP_ERR.PB_Error_Rst := FALSE;
   S701_TL_4_CLAMP_ERR.M_FLICK := FALSE;
   S701_TL_4_CLAMP_ERR.M_Adv_Err := FALSE;
   S701_TL_4_CLAMP_ERR.M_Ret_Err := FALSE;
   S701_TL_4_CLAMP_ERR.LP_Adv := FALSE;
   S701_TL_4_CLAMP_ERR.LP_Ret := FALSE;
   S701_TL_4_CLAMP_ERR.Visu_Adv := W#16#0;
   S701_TL_4_CLAMP_ERR.Visu_Ret := W#16#0;
   S701_TL_4_CLAMP_ERR.Error_T1.IN := FALSE;
   S701_TL_4_CLAMP_ERR.Error_T1.PT := T#0MS;
   S701_TL_4_CLAMP_ERR.Error_T1.Q := FALSE;
   S701_TL_4_CLAMP_ERR.Error_T1.ET := T#0MS;
   S701_TL_4_CLAMP_ERR.Error_T1.STATE := B#16#0;
   S701_TL_4_CLAMP_ERR.Error_T1.STIME := T#0MS;
   S701_TL_4_CLAMP_ERR.Error_T1.ATIME := T#0MS;
   S701_TL_4_CLAMP_ERR.Error_T2.IN := FALSE;
   S701_TL_4_CLAMP_ERR.Error_T2.PT := T#0MS;
   S701_TL_4_CLAMP_ERR.Error_T2.Q := FALSE;
   S701_TL_4_CLAMP_ERR.Error_T2.ET := T#0MS;
   S701_TL_4_CLAMP_ERR.Error_T2.STATE := B#16#0;
   S701_TL_4_CLAMP_ERR.Error_T2.STIME := T#0MS;
   S701_TL_4_CLAMP_ERR.Error_T2.ATIME := T#0MS;
   S701_TL_4_CLAMP_ERR.Adv_End_Aux := FALSE;
   S701_TL_4_CLAMP_ERR.Ret_End_Aux := FALSE;
   S701_TL_4_CLAMP_ERR.CHK_Aux1 := FALSE;
   S701_TL_4_CLAMP_ERR.CHK_Aux2 := FALSE;
   S701_TL_4_CLAMP_ERR.Error_T1_DN := FALSE;
   S701_TL_4_CLAMP_ERR.Error_T2_DN := FALSE;
   S701_TL_4_CLAMP_ERR.Adv_Memo := FALSE;
   S701_TL_4_CLAMP_ERR.Visu_Adv_Arr[0] := FALSE;
   S701_TL_4_CLAMP_ERR.Visu_Adv_Arr[1] := FALSE;
   S701_TL_4_CLAMP_ERR.Visu_Adv_Arr[2] := FALSE;
   S701_TL_4_CLAMP_ERR.Visu_Adv_Arr[3] := FALSE;
   S701_TL_4_CLAMP_ERR.Visu_Adv_Arr[4] := FALSE;
   S701_TL_4_CLAMP_ERR.Visu_Adv_Arr[5] := FALSE;
   S701_TL_4_CLAMP_ERR.Visu_Adv_Arr[6] := FALSE;
   S701_TL_4_CLAMP_ERR.Visu_Adv_Arr[7] := FALSE;
   S701_TL_4_CLAMP_ERR.Visu_Adv_Arr[8] := FALSE;
   S701_TL_4_CLAMP_ERR.Visu_Adv_Arr[9] := FALSE;
   S701_TL_4_CLAMP_ERR.Visu_Adv_Arr[10] := FALSE;
   S701_TL_4_CLAMP_ERR.Visu_Adv_Arr[11] := FALSE;
   S701_TL_4_CLAMP_ERR.Visu_Adv_Arr[12] := FALSE;
   S701_TL_4_CLAMP_ERR.Visu_Adv_Arr[13] := FALSE;
   S701_TL_4_CLAMP_ERR.Visu_Adv_Arr[14] := FALSE;
   S701_TL_4_CLAMP_ERR.Visu_Adv_Arr[15] := FALSE;
   S701_TL_4_CLAMP_ERR.Visu_Ret_Arr[0] := FALSE;
   S701_TL_4_CLAMP_ERR.Visu_Ret_Arr[1] := FALSE;
   S701_TL_4_CLAMP_ERR.Visu_Ret_Arr[2] := FALSE;
   S701_TL_4_CLAMP_ERR.Visu_Ret_Arr[3] := FALSE;
   S701_TL_4_CLAMP_ERR.Visu_Ret_Arr[4] := FALSE;
   S701_TL_4_CLAMP_ERR.Visu_Ret_Arr[5] := FALSE;
   S701_TL_4_CLAMP_ERR.Visu_Ret_Arr[6] := FALSE;
   S701_TL_4_CLAMP_ERR.Visu_Ret_Arr[7] := FALSE;
   S701_TL_4_CLAMP_ERR.Visu_Ret_Arr[8] := FALSE;
   S701_TL_4_CLAMP_ERR.Visu_Ret_Arr[9] := FALSE;
   S701_TL_4_CLAMP_ERR.Visu_Ret_Arr[10] := FALSE;
   S701_TL_4_CLAMP_ERR.Visu_Ret_Arr[11] := FALSE;
   S701_TL_4_CLAMP_ERR.Visu_Ret_Arr[12] := FALSE;
   S701_TL_4_CLAMP_ERR.Visu_Ret_Arr[13] := FALSE;
   S701_TL_4_CLAMP_ERR.Visu_Ret_Arr[14] := FALSE;
   S701_TL_4_CLAMP_ERR.Visu_Ret_Arr[15] := FALSE;
   S701_TL_4_CLAMP_ERR.BLK_Move_Ret := 0;
   S701_TL_4_CLAMP_ERR.Enable := FALSE;
   S701_TL_4_CLAMP_ERR.Adv_End := FALSE;
   S701_TL_4_CLAMP_ERR.Ret_End := FALSE;
   S701_TL_FDR_SFT_ERR.Enable_Aux := FALSE;
   S701_TL_FDR_SFT_ERR.Adv_Amount := 0;
   S701_TL_FDR_SFT_ERR.Ret_Amount := 0;
   S701_TL_FDR_SFT_ERR.LS_Adv1 := FALSE;
   S701_TL_FDR_SFT_ERR.LS_Ret1 := FALSE;
   S701_TL_FDR_SFT_ERR.LS_Adv2 := FALSE;
   S701_TL_FDR_SFT_ERR.LS_Ret2 := FALSE;
   S701_TL_FDR_SFT_ERR.LS_Adv3 := FALSE;
   S701_TL_FDR_SFT_ERR.LS_Ret3 := FALSE;
   S701_TL_FDR_SFT_ERR.LS_Adv4 := FALSE;
   S701_TL_FDR_SFT_ERR.LS_Ret4 := FALSE;
   S701_TL_FDR_SFT_ERR.LS_Adv5 := FALSE;
   S701_TL_FDR_SFT_ERR.LS_Ret5 := FALSE;
   S701_TL_FDR_SFT_ERR.LS_Adv6 := FALSE;
   S701_TL_FDR_SFT_ERR.LS_Ret6 := FALSE;
   S701_TL_FDR_SFT_ERR.LS_Adv7 := FALSE;
   S701_TL_FDR_SFT_ERR.LS_Ret7 := FALSE;
   S701_TL_FDR_SFT_ERR.LS_Adv8 := FALSE;
   S701_TL_FDR_SFT_ERR.LS_Ret8 := FALSE;
   S701_TL_FDR_SFT_ERR.SOL_Adv := FALSE;
   S701_TL_FDR_SFT_ERR.SOL_Ret := FALSE;
   S701_TL_FDR_SFT_ERR.M_Ready := FALSE;
   S701_TL_FDR_SFT_ERR.T_CHK1 := T#0MS;
   S701_TL_FDR_SFT_ERR.T_CHK2 := T#0MS;
   S701_TL_FDR_SFT_ERR.PB_Lamp_CHK := FALSE;
   S701_TL_FDR_SFT_ERR.PB_Error_Rst := FALSE;
   S701_TL_FDR_SFT_ERR.M_FLICK := FALSE;
   S701_TL_FDR_SFT_ERR.M_Adv_Err := FALSE;
   S701_TL_FDR_SFT_ERR.M_Ret_Err := FALSE;
   S701_TL_FDR_SFT_ERR.LP_Adv := FALSE;
   S701_TL_FDR_SFT_ERR.LP_Ret := FALSE;
   S701_TL_FDR_SFT_ERR.Visu_Adv := W#16#0;
   S701_TL_FDR_SFT_ERR.Visu_Ret := W#16#0;
   S701_TL_FDR_SFT_ERR.Error_T1.IN := FALSE;
   S701_TL_FDR_SFT_ERR.Error_T1.PT := T#0MS;
   S701_TL_FDR_SFT_ERR.Error_T1.Q := FALSE;
   S701_TL_FDR_SFT_ERR.Error_T1.ET := T#0MS;
   S701_TL_FDR_SFT_ERR.Error_T1.STATE := B#16#0;
   S701_TL_FDR_SFT_ERR.Error_T1.STIME := T#0MS;
   S701_TL_FDR_SFT_ERR.Error_T1.ATIME := T#0MS;
   S701_TL_FDR_SFT_ERR.Error_T2.IN := FALSE;
   S701_TL_FDR_SFT_ERR.Error_T2.PT := T#0MS;
   S701_TL_FDR_SFT_ERR.Error_T2.Q := FALSE;
   S701_TL_FDR_SFT_ERR.Error_T2.ET := T#0MS;
   S701_TL_FDR_SFT_ERR.Error_T2.STATE := B#16#0;
   S701_TL_FDR_SFT_ERR.Error_T2.STIME := T#0MS;
   S701_TL_FDR_SFT_ERR.Error_T2.ATIME := T#0MS;
   S701_TL_FDR_SFT_ERR.Adv_End_Aux := FALSE;
   S701_TL_FDR_SFT_ERR.Ret_End_Aux := FALSE;
   S701_TL_FDR_SFT_ERR.CHK_Aux1 := FALSE;
   S701_TL_FDR_SFT_ERR.CHK_Aux2 := FALSE;
   S701_TL_FDR_SFT_ERR.Error_T1_DN := FALSE;
   S701_TL_FDR_SFT_ERR.Error_T2_DN := FALSE;
   S701_TL_FDR_SFT_ERR.Adv_Memo := FALSE;
   S701_TL_FDR_SFT_ERR.Visu_Adv_Arr[0] := FALSE;
   S701_TL_FDR_SFT_ERR.Visu_Adv_Arr[1] := FALSE;
   S701_TL_FDR_SFT_ERR.Visu_Adv_Arr[2] := FALSE;
   S701_TL_FDR_SFT_ERR.Visu_Adv_Arr[3] := FALSE;
   S701_TL_FDR_SFT_ERR.Visu_Adv_Arr[4] := FALSE;
   S701_TL_FDR_SFT_ERR.Visu_Adv_Arr[5] := FALSE;
   S701_TL_FDR_SFT_ERR.Visu_Adv_Arr[6] := FALSE;
   S701_TL_FDR_SFT_ERR.Visu_Adv_Arr[7] := FALSE;
   S701_TL_FDR_SFT_ERR.Visu_Adv_Arr[8] := FALSE;
   S701_TL_FDR_SFT_ERR.Visu_Adv_Arr[9] := FALSE;
   S701_TL_FDR_SFT_ERR.Visu_Adv_Arr[10] := FALSE;
   S701_TL_FDR_SFT_ERR.Visu_Adv_Arr[11] := FALSE;
   S701_TL_FDR_SFT_ERR.Visu_Adv_Arr[12] := FALSE;
   S701_TL_FDR_SFT_ERR.Visu_Adv_Arr[13] := FALSE;
   S701_TL_FDR_SFT_ERR.Visu_Adv_Arr[14] := FALSE;
   S701_TL_FDR_SFT_ERR.Visu_Adv_Arr[15] := FALSE;
   S701_TL_FDR_SFT_ERR.Visu_Ret_Arr[0] := FALSE;
   S701_TL_FDR_SFT_ERR.Visu_Ret_Arr[1] := FALSE;
   S701_TL_FDR_SFT_ERR.Visu_Ret_Arr[2] := FALSE;
   S701_TL_FDR_SFT_ERR.Visu_Ret_Arr[3] := FALSE;
   S701_TL_FDR_SFT_ERR.Visu_Ret_Arr[4] := FALSE;
   S701_TL_FDR_SFT_ERR.Visu_Ret_Arr[5] := FALSE;
   S701_TL_FDR_SFT_ERR.Visu_Ret_Arr[6] := FALSE;
   S701_TL_FDR_SFT_ERR.Visu_Ret_Arr[7] := FALSE;
   S701_TL_FDR_SFT_ERR.Visu_Ret_Arr[8] := FALSE;
   S701_TL_FDR_SFT_ERR.Visu_Ret_Arr[9] := FALSE;
   S701_TL_FDR_SFT_ERR.Visu_Ret_Arr[10] := FALSE;
   S701_TL_FDR_SFT_ERR.Visu_Ret_Arr[11] := FALSE;
   S701_TL_FDR_SFT_ERR.Visu_Ret_Arr[12] := FALSE;
   S701_TL_FDR_SFT_ERR.Visu_Ret_Arr[13] := FALSE;
   S701_TL_FDR_SFT_ERR.Visu_Ret_Arr[14] := FALSE;
   S701_TL_FDR_SFT_ERR.Visu_Ret_Arr[15] := FALSE;
   S701_TL_FDR_SFT_ERR.BLK_Move_Ret := 0;
   S701_TL_FDR_SFT_ERR.Enable := FALSE;
   S701_TL_FDR_SFT_ERR.Adv_End := FALSE;
   S701_TL_FDR_SFT_ERR.Ret_End := FALSE;
END_DATA_BLOCK

FUNCTION FC 121 : VOID
TITLE =
VERSION : 0.1

BEGIN
NETWORK
TITLE =
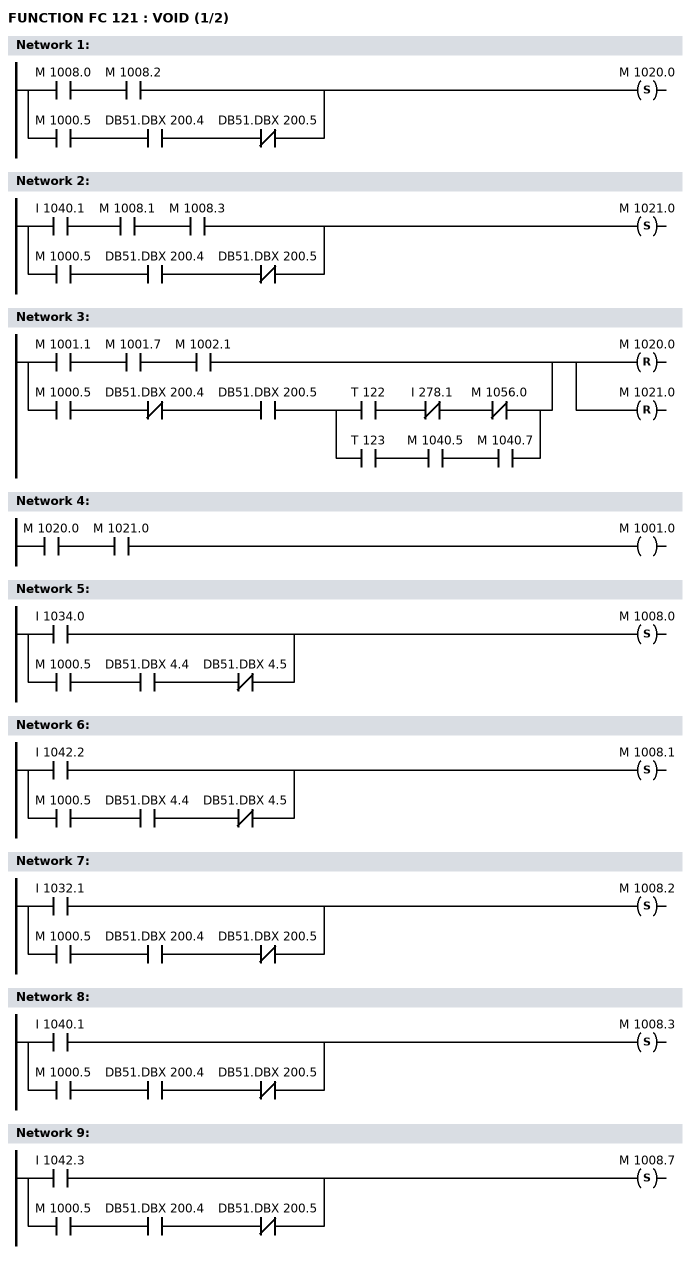

      A     M   1008.0;
      A     M   1008.2;
      O     ;
      A     M   1000.5;
      A     DB51.DBX  200.4;
      AN    DB51.DBX  200.5;
      S     M   1020.0;
NETWORK
TITLE =

      A     I   1040.1;
      A     M   1008.1;
      A     M   1008.3;
      O     ;
      A     M   1000.5;
      A     DB51.DBX  200.4;
      AN    DB51.DBX  200.5;
      S     M   1021.0;
NETWORK
TITLE =

      A     M   1001.1;
      A     M   1001.7;
      A     M   1002.1;
      O     ;
      A     M   1000.5;
      AN    DB51.DBX  200.4;
      A     DB51.DBX  200.5;
      A(    ;
      A     T    122;
      AN    I    278.1;
      AN    M   1056.0;
      O     ;
      A     T    123;
      A     M   1040.5;
      A     M   1040.7;
      )     ;
      R     M   1020.0;
      R     M   1021.0;
NETWORK
TITLE =

      A     M   1020.0;
      A     M   1021.0;
      =     M   1001.0;
NETWORK
TITLE =

      O     I   1034.0;
      O     ;
      A     M   1000.5;
      A     DB51.DBX    4.4;
      AN    DB51.DBX    4.5;
      S     M   1008.0;
NETWORK
TITLE =

      O     I   1042.2;
      O     ;
      A     M   1000.5;
      A     DB51.DBX    4.4;
      AN    DB51.DBX    4.5;
      S     M   1008.1;
NETWORK
TITLE =

      O     I   1032.1;
      O     ;
      A     M   1000.5;
      A     DB51.DBX  200.4;
      AN    DB51.DBX  200.5;
      S     M   1008.2;
NETWORK
TITLE =

      O     I   1040.1;
      O     ;
      A     M   1000.5;
      A     DB51.DBX  200.4;
      AN    DB51.DBX  200.5;
      S     M   1008.3;
NETWORK
TITLE =

      O     I   1042.3;
      O     ;
      A     M   1000.5;
      A     DB51.DBX  200.4;
      AN    DB51.DBX  200.5;
      S     M   1008.7;
NETWORK
TITLE =
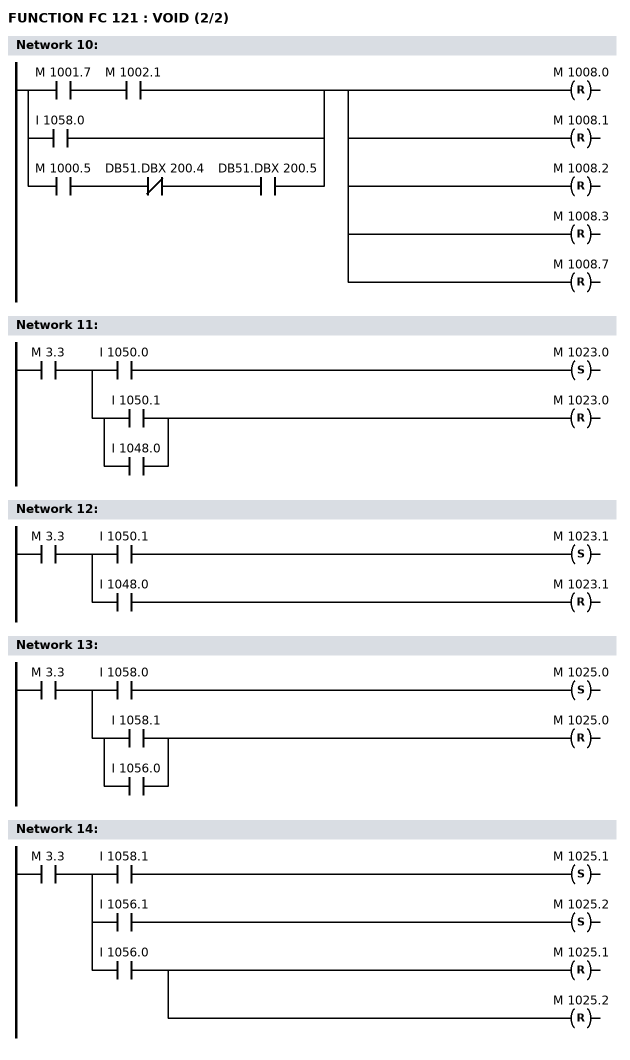

      A     M   1001.7;
      A     M   1002.1;
      O     I   1058.0;
      O     ;
      A     M   1000.5;
      AN    DB51.DBX  200.4;
      A     DB51.DBX  200.5;
      R     M   1008.0;
      R     M   1008.1;
      R     M   1008.2;
      R     M   1008.3;
      R     M   1008.7;
NETWORK
TITLE =

      A     M      3.3;
      =     L      0.0;
      A     L      0.0;
      A     I   1050.0;
      S     M   1023.0;
      A     L      0.0;
      A(    ;
      O     I   1050.1;
      O     I   1048.0;
      )     ;
      R     M   1023.0;
NETWORK
TITLE =

      A     M      3.3;
      =     L      0.0;
      A     L      0.0;
      A     I   1050.1;
      S     M   1023.1;
      A     L      0.0;
      A     I   1048.0;
      R     M   1023.1;
NETWORK
TITLE =

      A     M      3.3;
      =     L      0.0;
      A     L      0.0;
      A     I   1058.0;
      S     M   1025.0;
      A     L      0.0;
      A(    ;
      O     I   1058.1;
      O     I   1056.0;
      )     ;
      R     M   1025.0;
NETWORK
TITLE =

      A     M      3.3;
      =     L      0.0;
      A     L      0.0;
      A     I   1058.1;
      S     M   1025.1;
      A     L      0.0;
      A     I   1056.1;
      S     M   1025.2;
      A     L      0.0;
      A     I   1056.0;
      R     M   1025.1;
      R     M   1025.2;
END_FUNCTION

FUNCTION_BLOCK FB 122
TITLE =
VERSION : 0.1

BEGIN
NETWORK
TITLE =
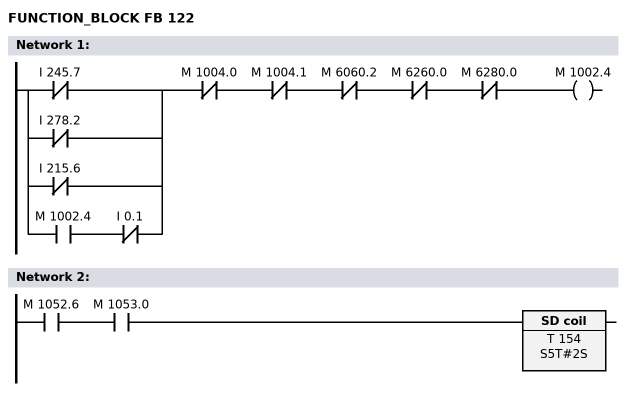

      A(    ;
      ON    I    245.7;
      ON    I    278.2;
      ON    I    215.6;
      O     ;
      A     M   1002.4;
      AN    I      0.1;
      )     ;
      AN    M   1004.0;
      AN    M   1004.1;
      AN    M   6060.2;
      AN    M   6260.0;
      AN    M   6280.0;
      =     M   1002.4;
NETWORK
TITLE =

      A     M   1052.6;
      A     M   1053.0;
      L     S5T#2S;
      SD    T    154;
NETWORK
TITLE =

      A(    ;
      A(    ;
      AN    I    278.6;
      A     I    278.6;
      A     M    205.2;
      A     M    205.6;
      O     ;
      A     I    278.6;
      A(    ;
      O     M    205.1;
      O     ;
      A     M    205.2;
      A(    ;
      ON    M    205.6;
      O     M    205.7;
      )     ;
      )     ;
      )     ;
      =     M     16.0;
      A     M     16.0;
      O(    ;
      A(    ;
      AN    I    278.7;
      A(    ;
      O     M    205.5;
      O     ;
      A     M    205.4;
      A     M    205.2;
      O     ;
      A     M    205.6;
      A     M    205.2;
      O     ;
      A     M    205.7;
      A     M    205.2;
      )     ;
      O     ;
      A     I    278.7;
      AN    M    205.4;
      AN    M    205.5;
      AN    M    205.6;
      AN    M    205.7;
      )     ;
      =     M     16.1;
      A     M     16.1;
      )     ;
      O(    ;
      A(    ;
      AN    I    279.0;
      A     M    205.5;
      O     ;
      A     I    279.0;
      AN    M    205.5;
      )     ;
      =     M     16.2;
      A     M     16.2;
      )     ;
      )     ;
      A     M    204.1;
      A     T    154;
      AN    M   1001.0;
      A(    ;
      O     T    131;
      O     T    122;
      )     ;
      O     ;
      A     M    204.0;
      A(    ;
      A     M    208.2;
      AN    I    209.4;
      O     ;
      A     M    208.6;
      A     I    209.4;
      )     ;
      A     M   1042.4;
      AN    M   1001.0;
      A     T    123;
      O     ;
      A     M   1002.5;
      AN    I      0.1;
      AN    I    180.1;
      =     L      0.0;
      A     L      0.0;
      A     T    134;
      =     M   1002.5;
      A     L      0.0;
      AN    M   1004.0;
      AN    M   1004.1;
      AN    M   6060.2;
      AN    M   6260.0;
      AN    M   6280.0;
      AN    M   1002.4;
      L     S5T#1S;
      SD    T    134;
NETWORK
TITLE =
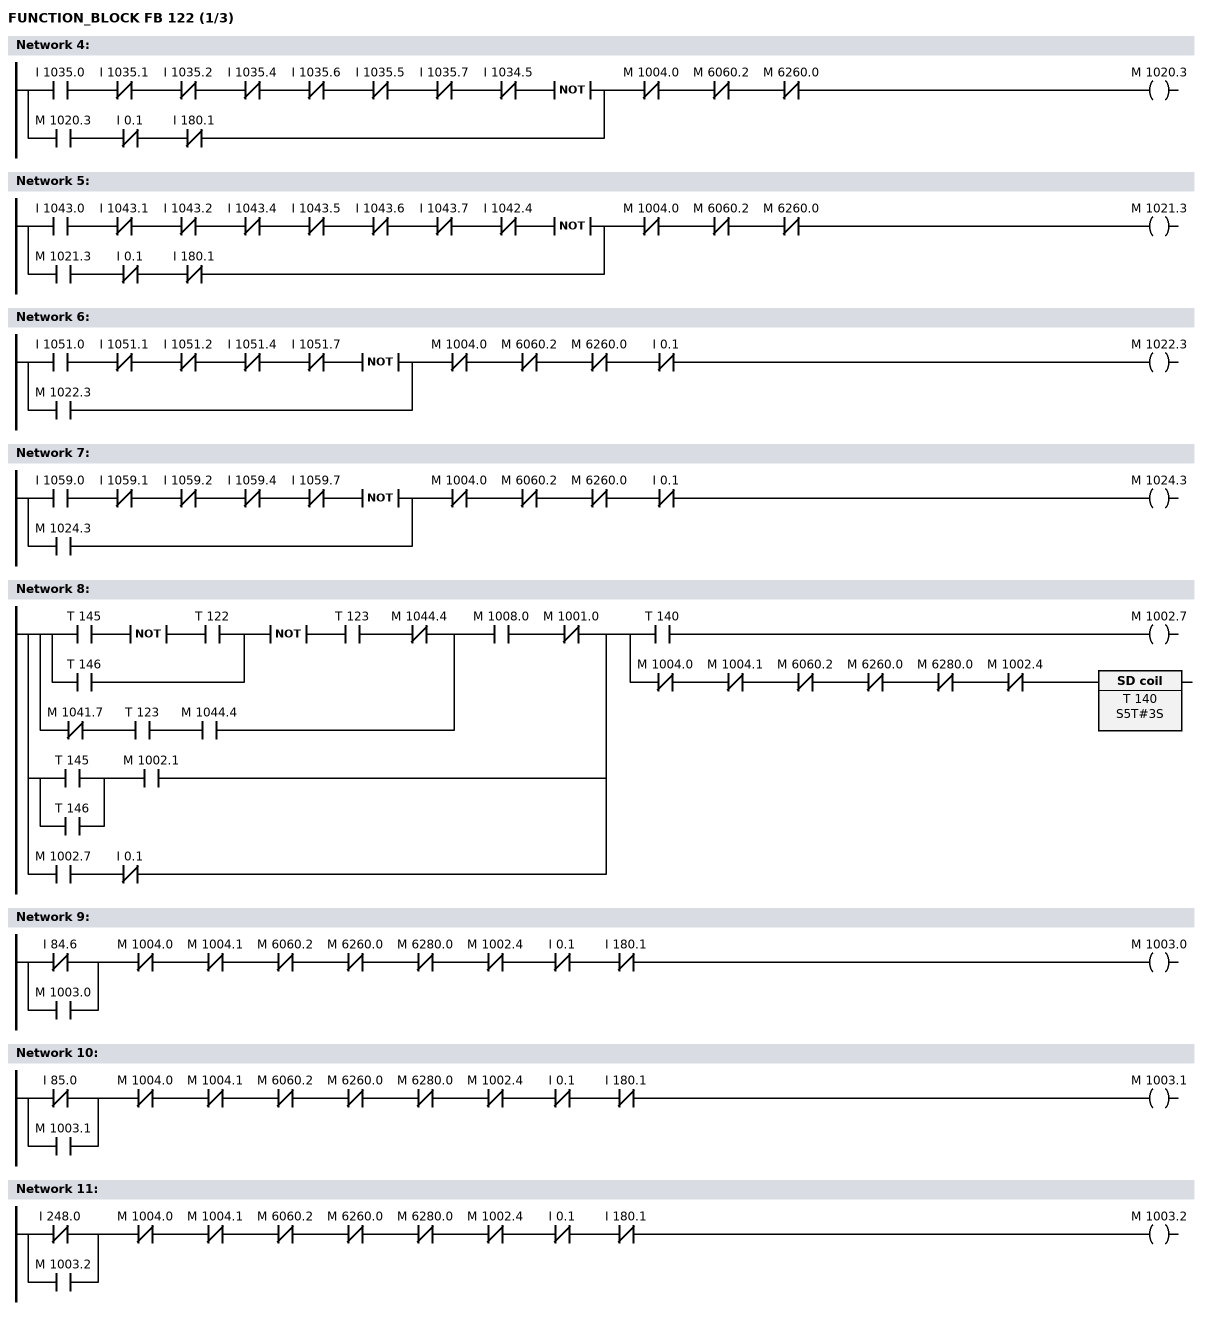

      A(    ;
      A     I   1035.0;
      AN    I   1035.1;
      AN    I   1035.2;
      AN    I   1035.4;
      AN    I   1035.6;
      AN    I   1035.5;
      AN    I   1035.7;
      AN    I   1034.5;
      NOT   ;
      O     ;
      A     M   1020.3;
      AN    I      0.1;
      AN    I    180.1;
      )     ;
      AN    M   1004.0;
      AN    M   6060.2;
      AN    M   6260.0;
      =     M   1020.3;
NETWORK
TITLE =

      A(    ;
      A     I   1043.0;
      AN    I   1043.1;
      AN    I   1043.2;
      AN    I   1043.4;
      AN    I   1043.5;
      AN    I   1043.6;
      AN    I   1043.7;
      AN    I   1042.4;
      NOT   ;
      O     ;
      A     M   1021.3;
      AN    I      0.1;
      AN    I    180.1;
      )     ;
      AN    M   1004.0;
      AN    M   6060.2;
      AN    M   6260.0;
      =     M   1021.3;
NETWORK
TITLE =

      A(    ;
      A     I   1051.0;
      AN    I   1051.1;
      AN    I   1051.2;
      AN    I   1051.4;
      AN    I   1051.7;
      NOT   ;
      O     M   1022.3;
      )     ;
      AN    M   1004.0;
      AN    M   6060.2;
      AN    M   6260.0;
      AN    I      0.1;
      =     M   1022.3;
NETWORK
TITLE =

      A(    ;
      A     I   1059.0;
      AN    I   1059.1;
      AN    I   1059.2;
      AN    I   1059.4;
      AN    I   1059.7;
      NOT   ;
      O     M   1024.3;
      )     ;
      AN    M   1004.0;
      AN    M   6060.2;
      AN    M   6260.0;
      AN    I      0.1;
      =     M   1024.3;
NETWORK
TITLE =

      A(    ;
      A     T    145;
      NOT   ;
      A     T    122;
      O     ;
      A     T    146;
      NOT   ;
      A     T    123;
      AN    M   1044.4;
      O     ;
      AN    M   1041.7;
      A     T    123;
      A     M   1044.4;
      )     ;
      A     M   1008.0;
      AN    M   1001.0;
      O     ;
      A(    ;
      O     T    145;
      O     T    146;
      )     ;
      A     M   1002.1;
      O     ;
      A     M   1002.7;
      AN    I      0.1;
      =     L      0.0;
      A     L      0.0;
      A     T    140;
      =     M   1002.7;
      A     L      0.0;
      AN    M   1004.0;
      AN    M   1004.1;
      AN    M   6060.2;
      AN    M   6260.0;
      AN    M   6280.0;
      AN    M   1002.4;
      L     S5T#3S;
      SD    T    140;
NETWORK
TITLE =

      A(    ;
      ON    I     84.6;
      O     M   1003.0;
      )     ;
      AN    M   1004.0;
      AN    M   1004.1;
      AN    M   6060.2;
      AN    M   6260.0;
      AN    M   6280.0;
      AN    M   1002.4;
      AN    I      0.1;
      AN    I    180.1;
      =     M   1003.0;
NETWORK
TITLE =

      A(    ;
      ON    I     85.0;
      O     M   1003.1;
      )     ;
      AN    M   1004.0;
      AN    M   1004.1;
      AN    M   6060.2;
      AN    M   6260.0;
      AN    M   6280.0;
      AN    M   1002.4;
      AN    I      0.1;
      AN    I    180.1;
      =     M   1003.1;
NETWORK
TITLE =

      A(    ;
      ON    I    248.0;
      O     M   1003.2;
      )     ;
      AN    M   1004.0;
      AN    M   1004.1;
      AN    M   6060.2;
      AN    M   6260.0;
      AN    M   6280.0;
      AN    M   1002.4;
      AN    I      0.1;
      AN    I    180.1;
      =     M   1003.2;
NETWORK
TITLE =
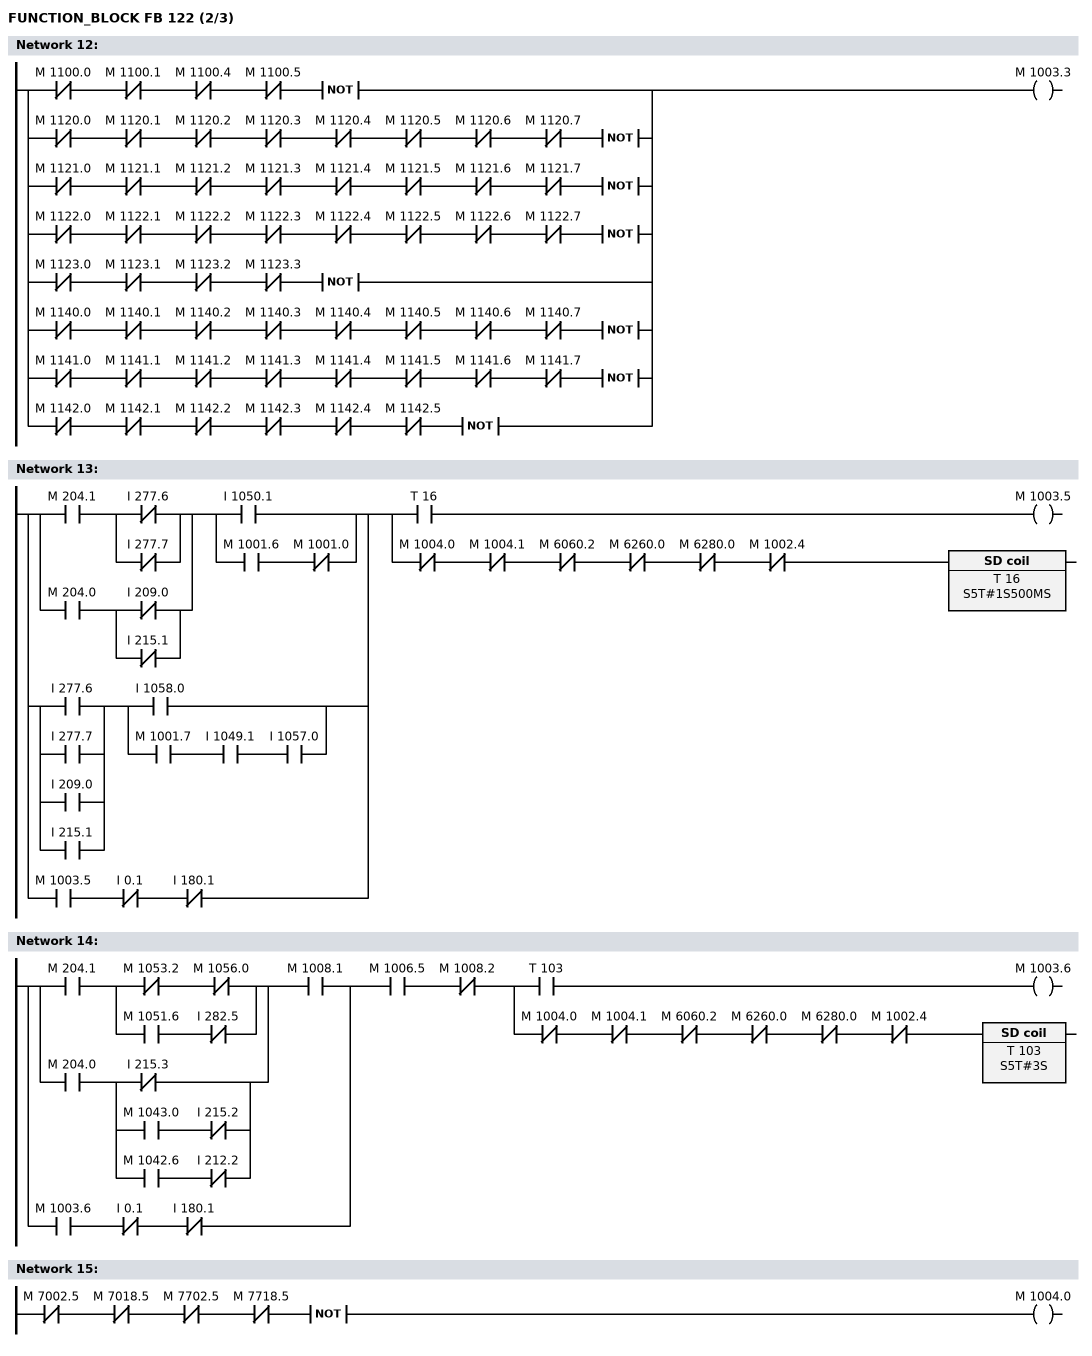

      AN    M   1100.0;
      AN    M   1100.1;
      AN    M   1100.4;
      AN    M   1100.5;
      NOT   ;
      O(    ;
      AN    M   1120.0;
      AN    M   1120.1;
      AN    M   1120.2;
      AN    M   1120.3;
      AN    M   1120.4;
      AN    M   1120.5;
      AN    M   1120.6;
      AN    M   1120.7;
      NOT   ;
      )     ;
      O(    ;
      AN    M   1121.0;
      AN    M   1121.1;
      AN    M   1121.2;
      AN    M   1121.3;
      AN    M   1121.4;
      AN    M   1121.5;
      AN    M   1121.6;
      AN    M   1121.7;
      NOT   ;
      )     ;
      O(    ;
      AN    M   1122.0;
      AN    M   1122.1;
      AN    M   1122.2;
      AN    M   1122.3;
      AN    M   1122.4;
      AN    M   1122.5;
      AN    M   1122.6;
      AN    M   1122.7;
      NOT   ;
      )     ;
      O(    ;
      AN    M   1123.0;
      AN    M   1123.1;
      AN    M   1123.2;
      AN    M   1123.3;
      NOT   ;
      )     ;
      O(    ;
      AN    M   1140.0;
      AN    M   1140.1;
      AN    M   1140.2;
      AN    M   1140.3;
      AN    M   1140.4;
      AN    M   1140.5;
      AN    M   1140.6;
      AN    M   1140.7;
      NOT   ;
      )     ;
      O(    ;
      AN    M   1141.0;
      AN    M   1141.1;
      AN    M   1141.2;
      AN    M   1141.3;
      AN    M   1141.4;
      AN    M   1141.5;
      AN    M   1141.6;
      AN    M   1141.7;
      NOT   ;
      )     ;
      O(    ;
      AN    M   1142.0;
      AN    M   1142.1;
      AN    M   1142.2;
      AN    M   1142.3;
      AN    M   1142.4;
      AN    M   1142.5;
      NOT   ;
      )     ;
      =     M   1003.3;
NETWORK
TITLE =

      A(    ;
      A     M    204.1;
      A(    ;
      ON    I    277.6;
      ON    I    277.7;
      )     ;
      O     ;
      A     M    204.0;
      A(    ;
      ON    I    209.0;
      ON    I    215.1;
      )     ;
      )     ;
      A(    ;
      O     I   1050.1;
      O     ;
      A     M   1001.6;
      AN    M   1001.0;
      )     ;
      O     ;
      A(    ;
      O     I    277.6;
      O     I    277.7;
      O     I    209.0;
      O     I    215.1;
      )     ;
      A(    ;
      O     I   1058.0;
      O     ;
      A     M   1001.7;
      A     I   1049.1;
      A     I   1057.0;
      )     ;
      O     ;
      A     M   1003.5;
      AN    I      0.1;
      AN    I    180.1;
      =     L      0.0;
      A     L      0.0;
      A     T     16;
      =     M   1003.5;
      A     L      0.0;
      AN    M   1004.0;
      AN    M   1004.1;
      AN    M   6060.2;
      AN    M   6260.0;
      AN    M   6280.0;
      AN    M   1002.4;
      L     S5T#1S500MS;
      SD    T     16;
NETWORK
TITLE =

      A(    ;
      A(    ;
      A     M    204.1;
      A(    ;
      AN    M   1053.2;
      AN    M   1056.0;
      O     ;
      A     M   1051.6;
      AN    I    282.5;
      )     ;
      O     ;
      A     M    204.0;
      A(    ;
      ON    I    215.3;
      O     ;
      A     M   1043.0;
      AN    I    215.2;
      O     ;
      A     M   1042.6;
      AN    I    212.2;
      )     ;
      )     ;
      A     M   1008.1;
      O     ;
      A     M   1003.6;
      AN    I      0.1;
      AN    I    180.1;
      )     ;
      A     M   1006.5;
      AN    M   1008.2;
      =     L      0.0;
      A     L      0.0;
      A     T    103;
      =     M   1003.6;
      A     L      0.0;
      AN    M   1004.0;
      AN    M   1004.1;
      AN    M   6060.2;
      AN    M   6260.0;
      AN    M   6280.0;
      AN    M   1002.4;
      L     S5T#3S;
      SD    T    103;
NETWORK
TITLE =

      AN    M   7002.5;
      AN    M   7018.5;
      AN    M   7702.5;
      AN    M   7718.5;
      NOT   ;
      =     M   1004.0;
NETWORK
TITLE =
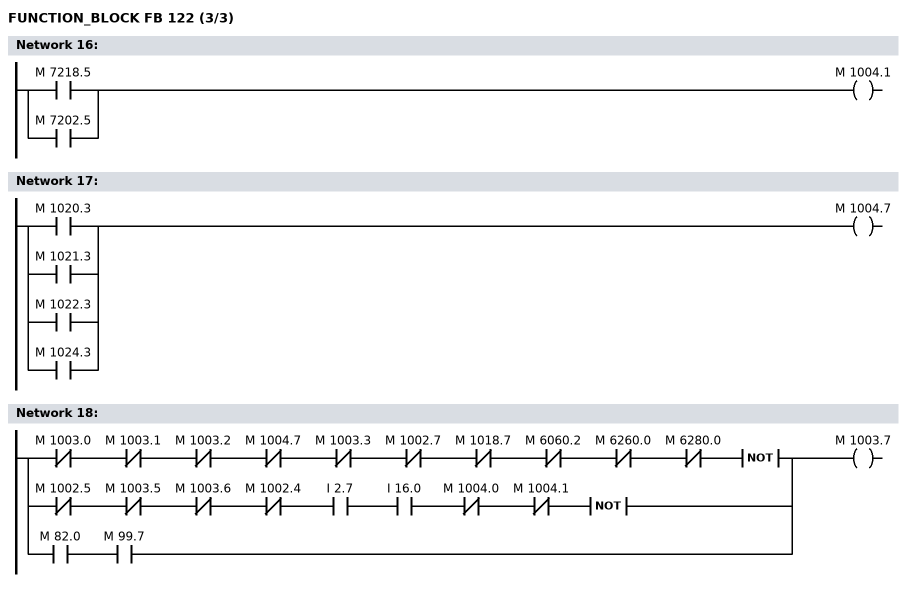

      O     M   7218.5;
      O     M   7202.5;
      =     M   1004.1;
NETWORK
TITLE =

      O     M   1020.3;
      O     M   1021.3;
      O     M   1022.3;
      O     M   1024.3;
      =     M   1004.7;
NETWORK
TITLE =

      AN    M   1003.0;
      AN    M   1003.1;
      AN    M   1003.2;
      AN    M   1004.7;
      AN    M   1003.3;
      AN    M   1002.7;
      AN    M   1018.7;
      AN    M   6060.2;
      AN    M   6260.0;
      AN    M   6280.0;
      NOT   ;
      O(    ;
      AN    M   1002.5;
      AN    M   1003.5;
      AN    M   1003.6;
      AN    M   1002.4;
      A     I      2.7;
      A     I     16.0;
      AN    M   1004.0;
      AN    M   1004.1;
      NOT   ;
      )     ;
      O     ;
      A     M     82.0;
      A     M     99.7;
      =     M   1003.7;
END_FUNCTION_BLOCK

DATA_BLOCK DB 122
TITLE =
VERSION : 0.0

 FB 122
BEGIN
END_DATA_BLOCK

FUNCTION FC 122 : VOID
TITLE =
VERSION : 0.1

BEGIN
NETWORK
TITLE =INDEX

NETWORK
TITLE =
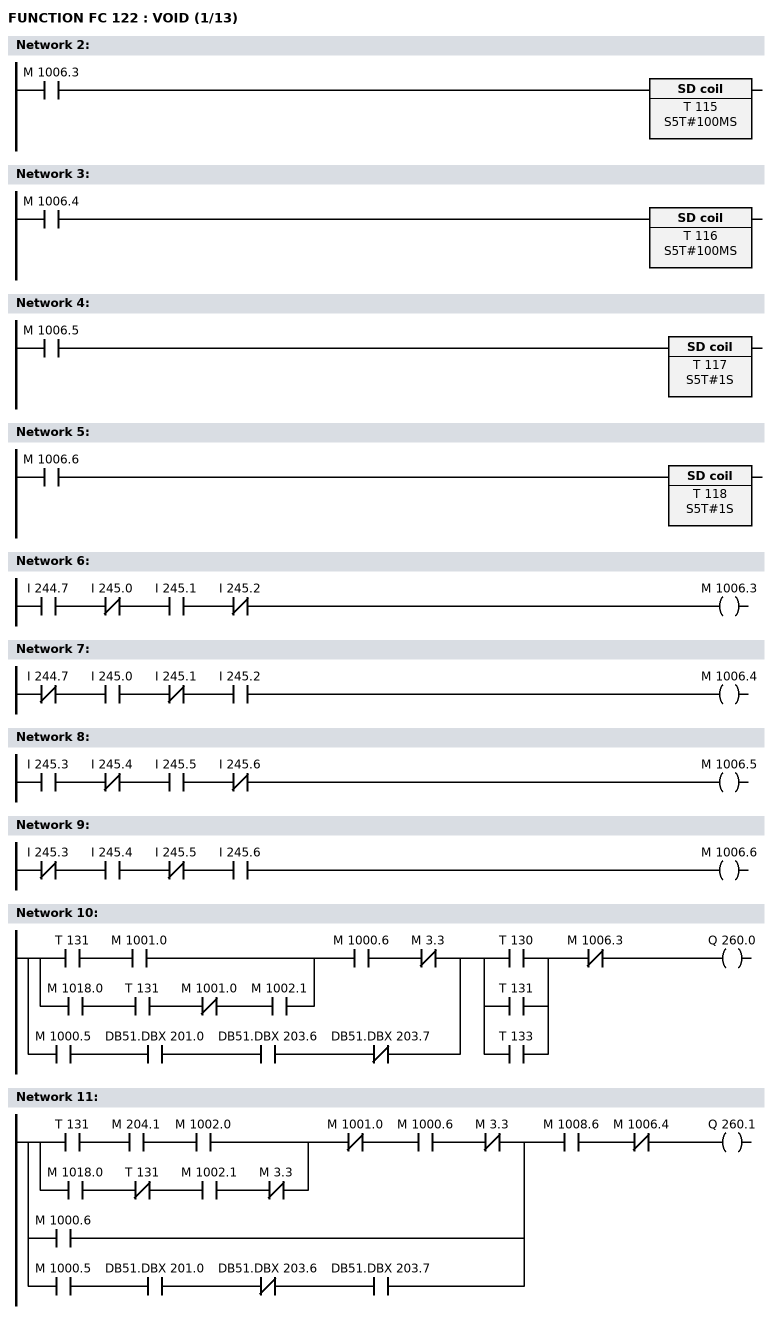

      A     M   1006.3;
      L     S5T#100MS;
      SD    T    115;
NETWORK
TITLE =

      A     M   1006.4;
      L     S5T#100MS;
      SD    T    116;
NETWORK
TITLE =

      A     M   1006.5;
      L     S5T#1S;
      SD    T    117;
NETWORK
TITLE =

      A     M   1006.6;
      L     S5T#1S;
      SD    T    118;
NETWORK
TITLE =

      A     I    244.7;
      AN    I    245.0;
      A     I    245.1;
      AN    I    245.2;
      =     M   1006.3;
NETWORK
TITLE =

      AN    I    244.7;
      A     I    245.0;
      AN    I    245.1;
      A     I    245.2;
      =     M   1006.4;
NETWORK
TITLE =

      A     I    245.3;
      AN    I    245.4;
      A     I    245.5;
      AN    I    245.6;
      =     M   1006.5;
NETWORK
TITLE =

      AN    I    245.3;
      A     I    245.4;
      AN    I    245.5;
      A     I    245.6;
      =     M   1006.6;
NETWORK
TITLE =

      A(    ;
      A(    ;
      A     T    131;
      A     M   1001.0;
      O     ;
      A     M   1018.0;
      A     T    131;
      AN    M   1001.0;
      A     M   1002.1;
      )     ;
      A     M   1000.6;
      AN    M      3.3;
      O     ;
      A     M   1000.5;
      A     DB51.DBX  201.0;
      A     DB51.DBX  203.6;
      AN    DB51.DBX  203.7;
      )     ;
      A(    ;
      O     T    130;
      O     T    131;
      O     T    133;
      )     ;
      AN    M   1006.3;
      =     Q    260.0;
NETWORK
TITLE =

      A(    ;
      A(    ;
      A     T    131;
      A     M    204.1;
      A     M   1002.0;
      O     ;
      A     M   1018.0;
      AN    T    131;
      A     M   1002.1;
      AN    M      3.3;
      )     ;
      AN    M   1001.0;
      A     M   1000.6;
      AN    M      3.3;
      O     M   1000.6;
      O     ;
      A     M   1000.5;
      A     DB51.DBX  201.0;
      AN    DB51.DBX  203.6;
      A     DB51.DBX  203.7;
      )     ;
      A     M   1008.6;
      AN    M   1006.4;
      =     Q    260.1;
NETWORK
TITLE =
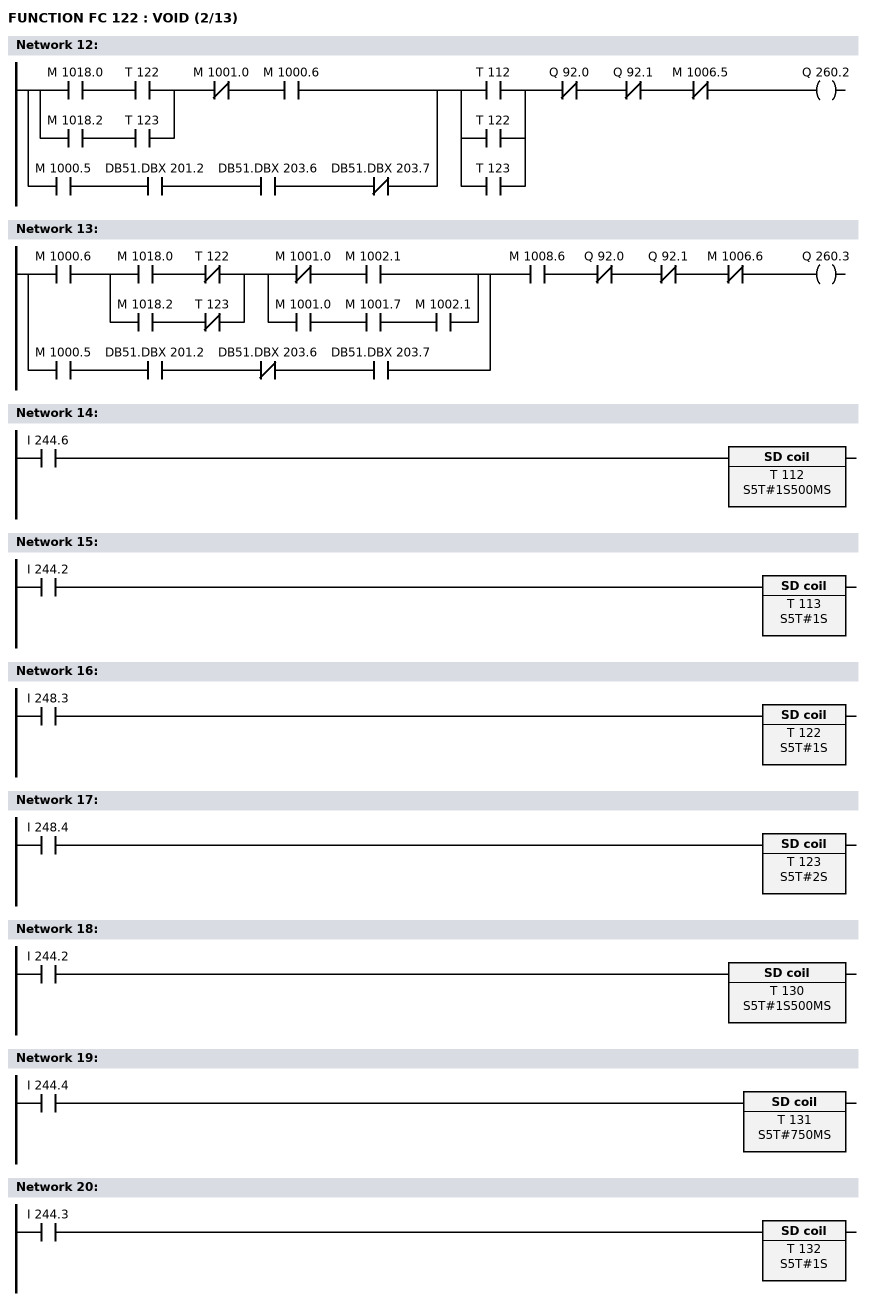

      A(    ;
      A(    ;
      A     M   1018.0;
      A     T    122;
      O     ;
      A     M   1018.2;
      A     T    123;
      )     ;
      AN    M   1001.0;
      A     M   1000.6;
      O     ;
      A     M   1000.5;
      A     DB51.DBX  201.2;
      A     DB51.DBX  203.6;
      AN    DB51.DBX  203.7;
      )     ;
      A(    ;
      O     T    112;
      O     T    122;
      O     T    123;
      )     ;
      AN    Q     92.0;
      AN    Q     92.1;
      AN    M   1006.5;
      =     Q    260.2;
NETWORK
TITLE =

      A(    ;
      A     M   1000.6;
      A(    ;
      A     M   1018.0;
      AN    T    122;
      O     ;
      A     M   1018.2;
      AN    T    123;
      )     ;
      A(    ;
      AN    M   1001.0;
      A     M   1002.1;
      O     ;
      A     M   1001.0;
      A     M   1001.7;
      A     M   1002.1;
      )     ;
      O     ;
      A     M   1000.5;
      A     DB51.DBX  201.2;
      AN    DB51.DBX  203.6;
      A     DB51.DBX  203.7;
      )     ;
      A     M   1008.6;
      AN    Q     92.0;
      AN    Q     92.1;
      AN    M   1006.6;
      =     Q    260.3;
NETWORK
TITLE =

      A     I    244.6;
      L     S5T#1S500MS;
      SD    T    112;
NETWORK
TITLE =

      A     I    244.2;
      L     S5T#1S;
      SD    T    113;
NETWORK
TITLE =

      A     I    248.3;
      L     S5T#1S;
      SD    T    122;
NETWORK
TITLE =

      A     I    248.4;
      L     S5T#2S;
      SD    T    123;
NETWORK
TITLE =

      A     I    244.2;
      L     S5T#1S500MS;
      SD    T    130;
NETWORK
TITLE =

      A     I    244.4;
      L     S5T#750MS;
      SD    T    131;
NETWORK
TITLE =

      A     I    244.3;
      L     S5T#1S;
      SD    T    132;
NETWORK
TITLE =
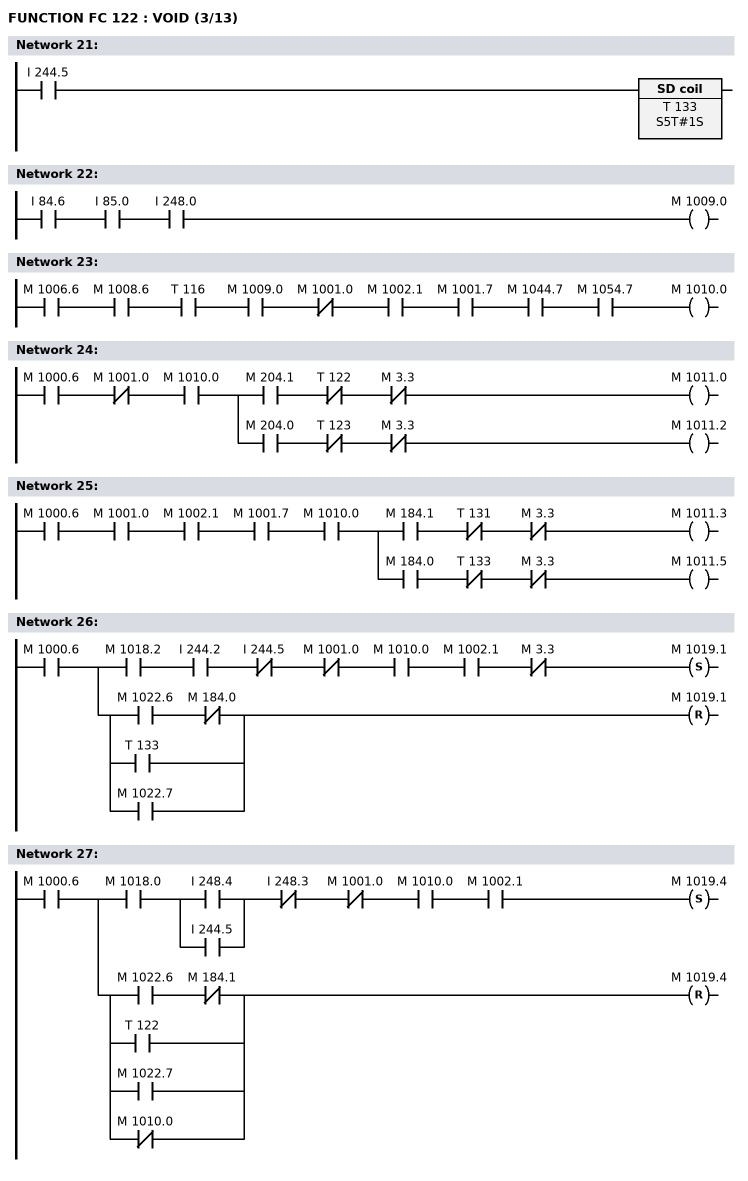

      A     I    244.5;
      L     S5T#1S;
      SD    T    133;
NETWORK
TITLE =

      A     I     84.6;
      A     I     85.0;
      A     I    248.0;
      =     M   1009.0;
NETWORK
TITLE =

      A     M   1006.6;
      A     M   1008.6;
      A     T    116;
      A     M   1009.0;
      AN    M   1001.0;
      A     M   1002.1;
      A     M   1001.7;
      A     M   1044.7;
      A     M   1054.7;
      =     M   1010.0;
NETWORK
TITLE =

      A     M   1000.6;
      AN    M   1001.0;
      A     M   1010.0;
      =     L      0.0;
      A     L      0.0;
      A     M    204.1;
      AN    T    122;
      AN    M      3.3;
      =     M   1011.0;
      A     L      0.0;
      A     M    204.0;
      AN    T    123;
      AN    M      3.3;
      =     M   1011.2;
NETWORK
TITLE =

      A     M   1000.6;
      A     M   1001.0;
      A     M   1002.1;
      A     M   1001.7;
      A     M   1010.0;
      =     L      0.0;
      A     L      0.0;
      A     M    184.1;
      AN    T    131;
      AN    M      3.3;
      =     M   1011.3;
      A     L      0.0;
      A     M    184.0;
      AN    T    133;
      AN    M      3.3;
      =     M   1011.5;
NETWORK
TITLE =

      A     M   1000.6;
      =     L      0.0;
      A     L      0.0;
      A     M   1018.2;
      A     I    244.2;
      AN    I    244.5;
      AN    M   1001.0;
      A     M   1010.0;
      A     M   1002.1;
      AN    M      3.3;
      S     M   1019.1;
      A     L      0.0;
      A(    ;
      A     M   1022.6;
      AN    M    184.0;
      O     T    133;
      O     M   1022.7;
      )     ;
      R     M   1019.1;
NETWORK
TITLE =

      A     M   1000.6;
      =     L      0.0;
      A     L      0.0;
      A     M   1018.0;
      A(    ;
      O     I    248.4;
      O     I    244.5;
      )     ;
      AN    I    248.3;
      AN    M   1001.0;
      A     M   1010.0;
      A     M   1002.1;
      S     M   1019.4;
      A     L      0.0;
      A(    ;
      A     M   1022.6;
      AN    M    184.1;
      O     T    122;
      O     M   1022.7;
      ON    M   1010.0;
      )     ;
      R     M   1019.4;
NETWORK
TITLE =
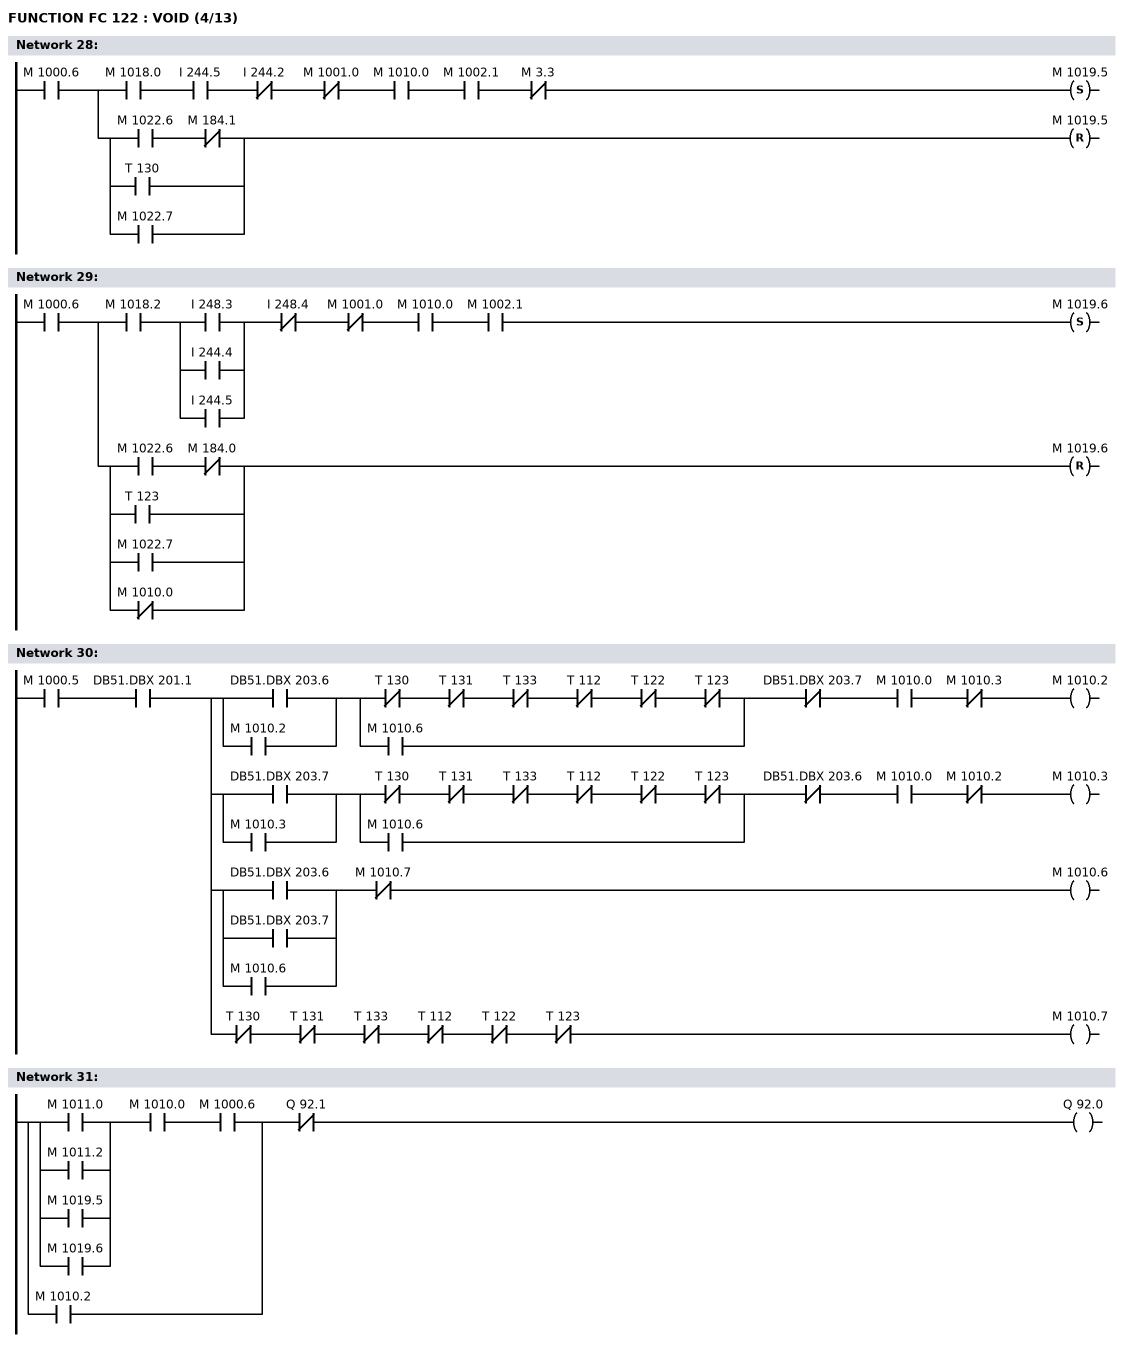

      A     M   1000.6;
      =     L      0.0;
      A     L      0.0;
      A     M   1018.0;
      A     I    244.5;
      AN    I    244.2;
      AN    M   1001.0;
      A     M   1010.0;
      A     M   1002.1;
      AN    M      3.3;
      S     M   1019.5;
      A     L      0.0;
      A(    ;
      A     M   1022.6;
      AN    M    184.1;
      O     T    130;
      O     M   1022.7;
      )     ;
      R     M   1019.5;
NETWORK
TITLE =

      A     M   1000.6;
      =     L      0.0;
      A     L      0.0;
      A     M   1018.2;
      A(    ;
      O     I    248.3;
      O     I    244.4;
      O     I    244.5;
      )     ;
      AN    I    248.4;
      AN    M   1001.0;
      A     M   1010.0;
      A     M   1002.1;
      S     M   1019.6;
      A     L      0.0;
      A(    ;
      A     M   1022.6;
      AN    M    184.0;
      O     T    123;
      O     M   1022.7;
      ON    M   1010.0;
      )     ;
      R     M   1019.6;
NETWORK
TITLE =

      A     M   1000.5;
      A     DB51.DBX  201.1;
      =     L      0.0;
      A     L      0.0;
      A(    ;
      O     DB51.DBX  203.6;
      O     M   1010.2;
      )     ;
      A(    ;
      AN    T    130;
      AN    T    131;
      AN    T    133;
      AN    T    112;
      AN    T    122;
      AN    T    123;
      O     M   1010.6;
      )     ;
      AN    DB51.DBX  203.7;
      A     M   1010.0;
      AN    M   1010.3;
      =     M   1010.2;
      A     L      0.0;
      A(    ;
      O     DB51.DBX  203.7;
      O     M   1010.3;
      )     ;
      A(    ;
      AN    T    130;
      AN    T    131;
      AN    T    133;
      AN    T    112;
      AN    T    122;
      AN    T    123;
      O     M   1010.6;
      )     ;
      AN    DB51.DBX  203.6;
      A     M   1010.0;
      AN    M   1010.2;
      =     M   1010.3;
      A     L      0.0;
      A(    ;
      O     DB51.DBX  203.6;
      O     DB51.DBX  203.7;
      O     M   1010.6;
      )     ;
      AN    M   1010.7;
      =     M   1010.6;
      A     L      0.0;
      AN    T    130;
      AN    T    131;
      AN    T    133;
      AN    T    112;
      AN    T    122;
      AN    T    123;
      =     M   1010.7;
NETWORK
TITLE =

      A(    ;
      A(    ;
      O     M   1011.0;
      O     M   1011.2;
      O     M   1019.5;
      O     M   1019.6;
      )     ;
      A     M   1010.0;
      A     M   1000.6;
      O     M   1010.2;
      )     ;
      AN    Q     92.1;
      =     Q     92.0;
NETWORK
TITLE =
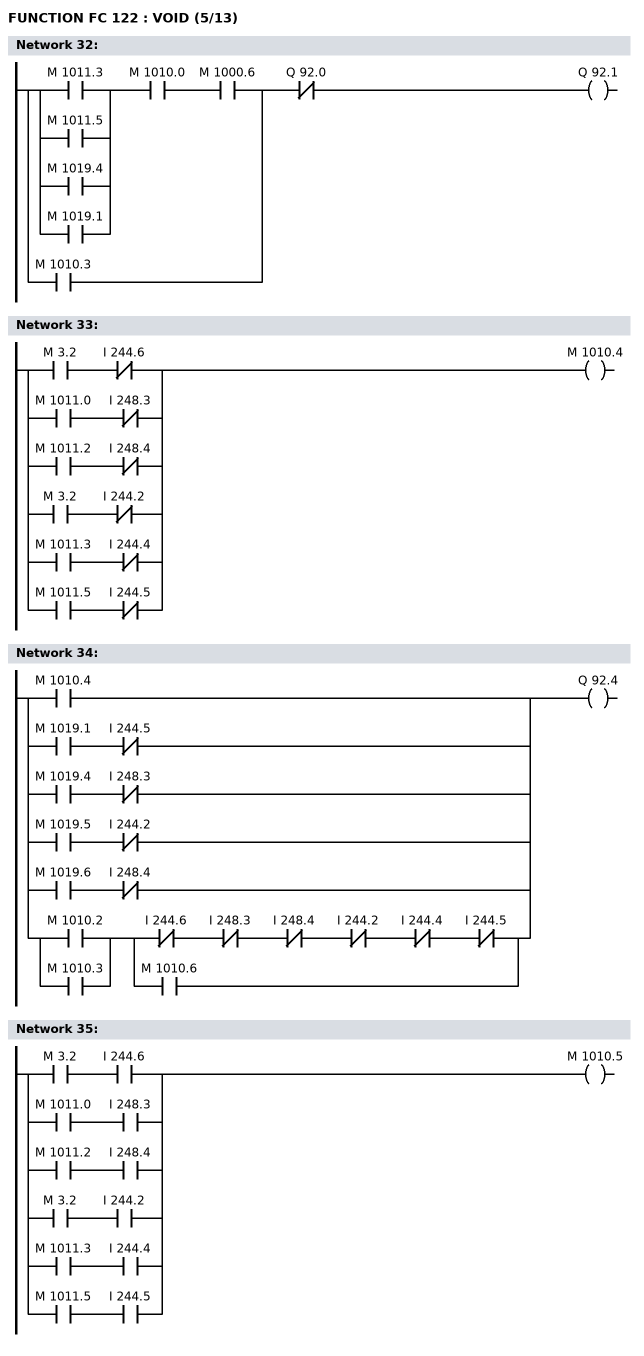

      A(    ;
      A(    ;
      O     M   1011.3;
      O     M   1011.5;
      O     M   1019.4;
      O     M   1019.1;
      )     ;
      A     M   1010.0;
      A     M   1000.6;
      O     M   1010.3;
      )     ;
      AN    Q     92.0;
      =     Q     92.1;
NETWORK
TITLE =

      A     M      3.2;
      AN    I    244.6;
      O     ;
      A     M   1011.0;
      AN    I    248.3;
      O     ;
      A     M   1011.2;
      AN    I    248.4;
      O     ;
      A     M      3.2;
      AN    I    244.2;
      O     ;
      A     M   1011.3;
      AN    I    244.4;
      O     ;
      A     M   1011.5;
      AN    I    244.5;
      =     M   1010.4;
NETWORK
TITLE =

      O     M   1010.4;
      O     ;
      A     M   1019.1;
      AN    I    244.5;
      O     ;
      A     M   1019.4;
      AN    I    248.3;
      O     ;
      A     M   1019.5;
      AN    I    244.2;
      O     ;
      A     M   1019.6;
      AN    I    248.4;
      O     ;
      A(    ;
      O     M   1010.2;
      O     M   1010.3;
      )     ;
      A(    ;
      AN    I    244.6;
      AN    I    248.3;
      AN    I    248.4;
      AN    I    244.2;
      AN    I    244.4;
      AN    I    244.5;
      O     M   1010.6;
      )     ;
      =     Q     92.4;
NETWORK
TITLE =

      A     M      3.2;
      A     I    244.6;
      O     ;
      A     M   1011.0;
      A     I    248.3;
      O     ;
      A     M   1011.2;
      A     I    248.4;
      O     ;
      A     M      3.2;
      A     I    244.2;
      O     ;
      A     M   1011.3;
      A     I    244.4;
      O     ;
      A     M   1011.5;
      A     I    244.5;
      =     M   1010.5;
NETWORK
TITLE =
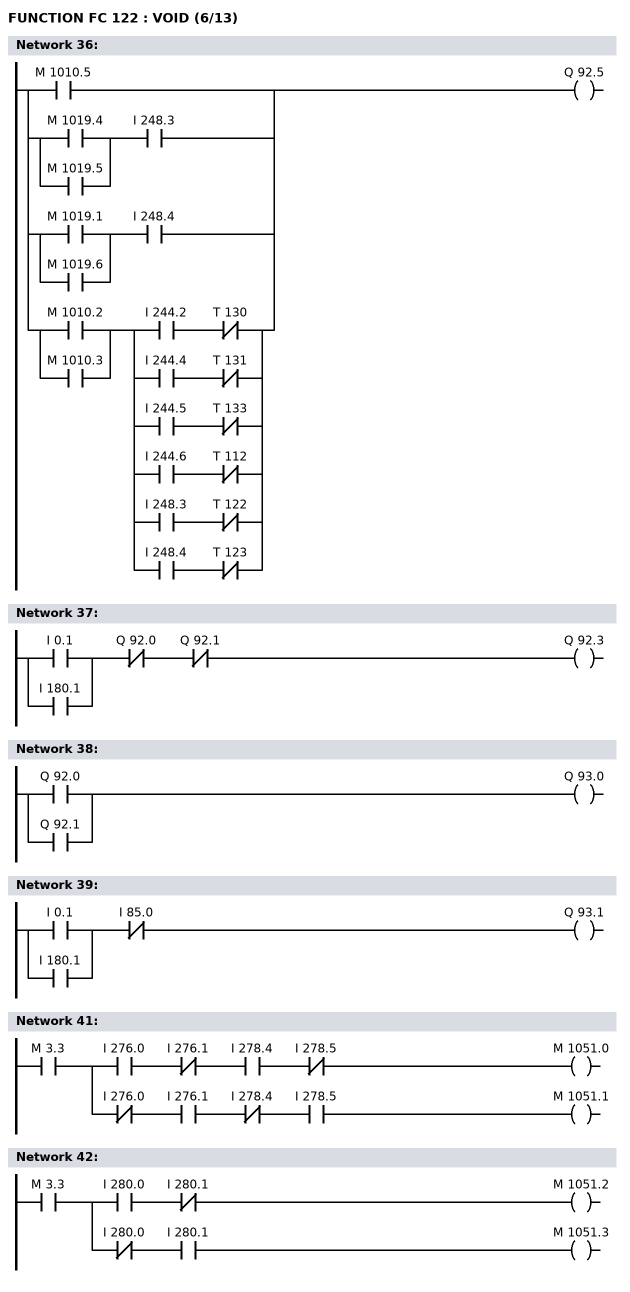

      O     M   1010.5;
      O     ;
      A(    ;
      O     M   1019.4;
      O     M   1019.5;
      )     ;
      A     I    248.3;
      O     ;
      A(    ;
      O     M   1019.1;
      O     M   1019.6;
      )     ;
      A     I    248.4;
      O     ;
      A(    ;
      O     M   1010.2;
      O     M   1010.3;
      )     ;
      A(    ;
      A     I    244.2;
      AN    T    130;
      O     ;
      A     I    244.4;
      AN    T    131;
      O     ;
      A     I    244.5;
      AN    T    133;
      O     ;
      A     I    244.6;
      AN    T    112;
      O     ;
      A     I    248.3;
      AN    T    122;
      O     ;
      A     I    248.4;
      AN    T    123;
      )     ;
      =     Q     92.5;
NETWORK
TITLE =

      A(    ;
      O     I      0.1;
      O     I    180.1;
      )     ;
      AN    Q     92.0;
      AN    Q     92.1;
      =     Q     92.3;
NETWORK
TITLE =

      O     Q     92.0;
      O     Q     92.1;
      =     Q     93.0;
NETWORK
TITLE =

      A(    ;
      O     I      0.1;
      O     I    180.1;
      )     ;
      AN    I     85.0;
      =     Q     93.1;
NETWORK
TITLE =INDEX LM

NETWORK
TITLE =

      A     M      3.3;
      =     L      0.0;
      A     L      0.0;
      A     I    276.0;
      AN    I    276.1;
      A     I    278.4;
      AN    I    278.5;
      =     M   1051.0;
      A     L      0.0;
      AN    I    276.0;
      A     I    276.1;
      AN    I    278.4;
      A     I    278.5;
      =     M   1051.1;
NETWORK
TITLE =

      A     M      3.3;
      =     L      0.0;
      A     L      0.0;
      A     I    280.0;
      AN    I    280.1;
      =     M   1051.2;
      A     L      0.0;
      AN    I    280.0;
      A     I    280.1;
      =     M   1051.3;
NETWORK
TITLE =
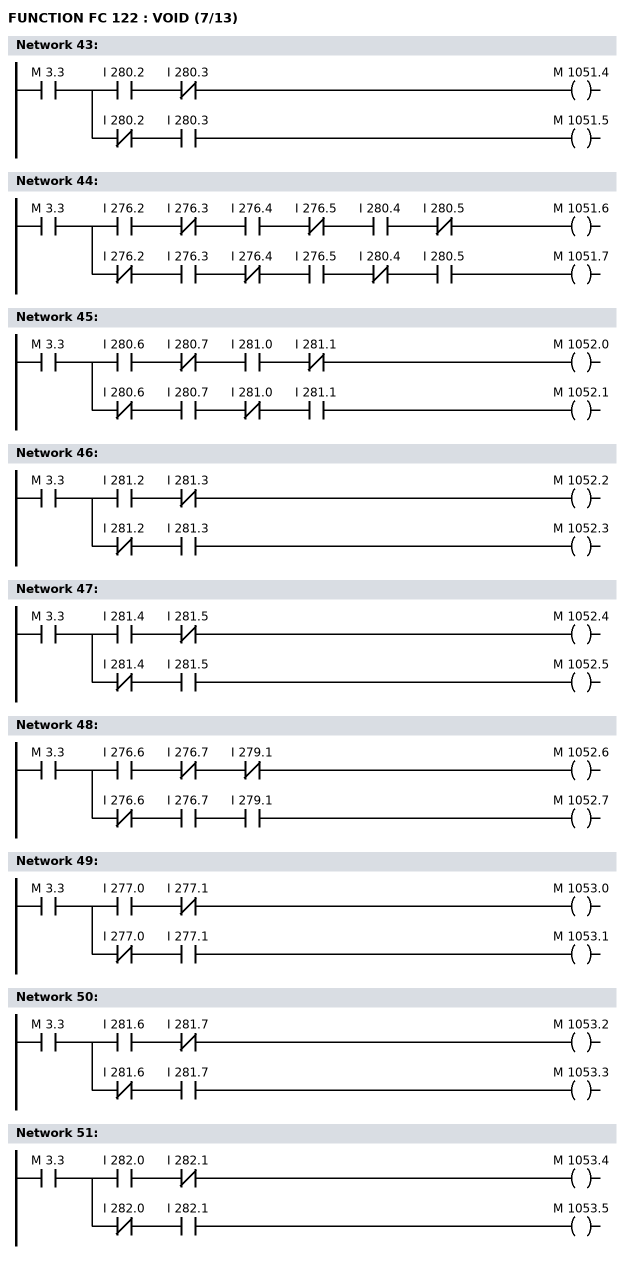

      A     M      3.3;
      =     L      0.0;
      A     L      0.0;
      A     I    280.2;
      AN    I    280.3;
      =     M   1051.4;
      A     L      0.0;
      AN    I    280.2;
      A     I    280.3;
      =     M   1051.5;
NETWORK
TITLE =

      A     M      3.3;
      =     L      0.0;
      A     L      0.0;
      A     I    276.2;
      AN    I    276.3;
      A     I    276.4;
      AN    I    276.5;
      A     I    280.4;
      AN    I    280.5;
      =     M   1051.6;
      A     L      0.0;
      AN    I    276.2;
      A     I    276.3;
      AN    I    276.4;
      A     I    276.5;
      AN    I    280.4;
      A     I    280.5;
      =     M   1051.7;
NETWORK
TITLE =

      A     M      3.3;
      =     L      0.0;
      A     L      0.0;
      A     I    280.6;
      AN    I    280.7;
      A     I    281.0;
      AN    I    281.1;
      =     M   1052.0;
      A     L      0.0;
      AN    I    280.6;
      A     I    280.7;
      AN    I    281.0;
      A     I    281.1;
      =     M   1052.1;
NETWORK
TITLE =

      A     M      3.3;
      =     L      0.0;
      A     L      0.0;
      A     I    281.2;
      AN    I    281.3;
      =     M   1052.2;
      A     L      0.0;
      AN    I    281.2;
      A     I    281.3;
      =     M   1052.3;
NETWORK
TITLE =

      A     M      3.3;
      =     L      0.0;
      A     L      0.0;
      A     I    281.4;
      AN    I    281.5;
      =     M   1052.4;
      A     L      0.0;
      AN    I    281.4;
      A     I    281.5;
      =     M   1052.5;
NETWORK
TITLE =

      A     M      3.3;
      =     L      0.0;
      A     L      0.0;
      A     I    276.6;
      AN    I    276.7;
      AN    I    279.1;
      =     M   1052.6;
      A     L      0.0;
      AN    I    276.6;
      A     I    276.7;
      A     I    279.1;
      =     M   1052.7;
NETWORK
TITLE =

      A     M      3.3;
      =     L      0.0;
      A     L      0.0;
      A     I    277.0;
      AN    I    277.1;
      =     M   1053.0;
      A     L      0.0;
      AN    I    277.0;
      A     I    277.1;
      =     M   1053.1;
NETWORK
TITLE =

      A     M      3.3;
      =     L      0.0;
      A     L      0.0;
      A     I    281.6;
      AN    I    281.7;
      =     M   1053.2;
      A     L      0.0;
      AN    I    281.6;
      A     I    281.7;
      =     M   1053.3;
NETWORK
TITLE =

      A     M      3.3;
      =     L      0.0;
      A     L      0.0;
      A     I    282.0;
      AN    I    282.1;
      =     M   1053.4;
      A     L      0.0;
      AN    I    282.0;
      A     I    282.1;
      =     M   1053.5;
NETWORK
TITLE =
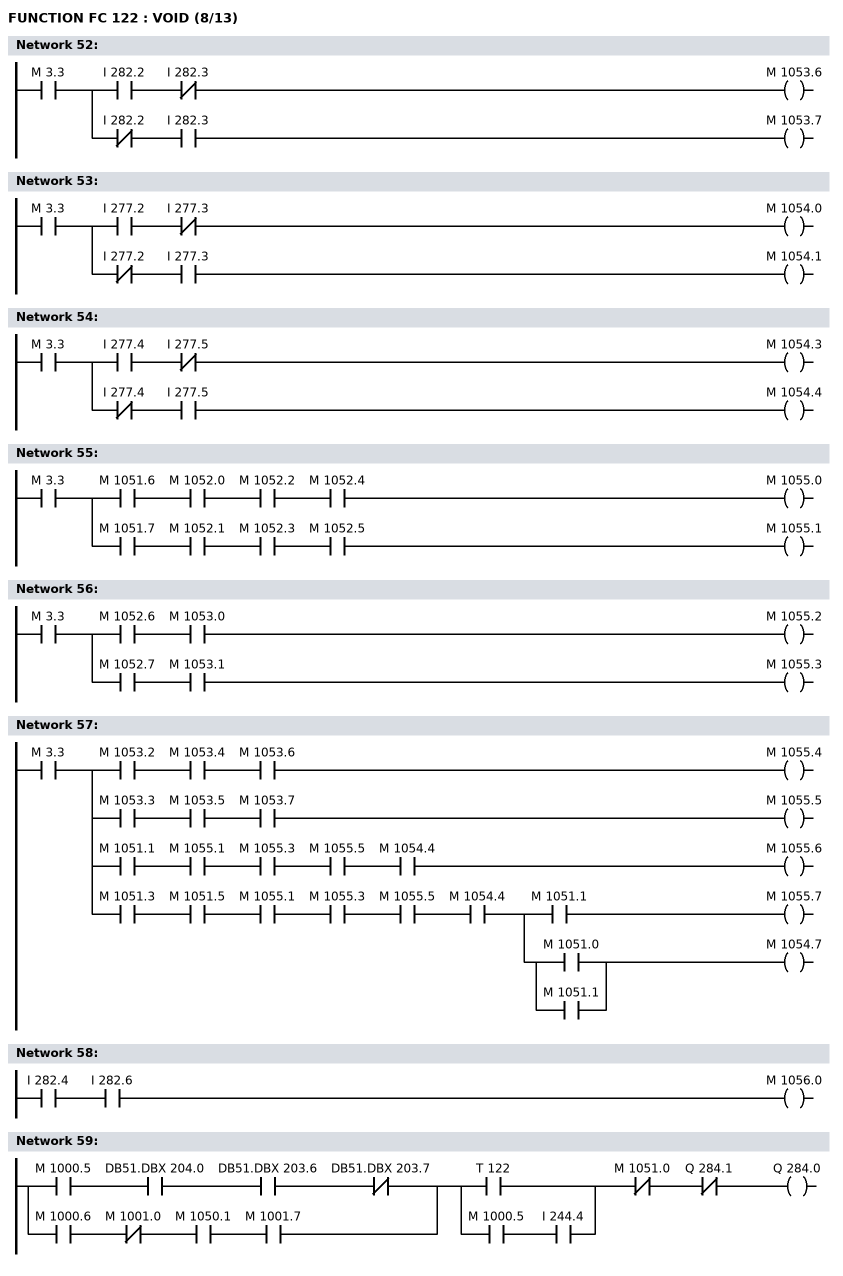

      A     M      3.3;
      =     L      0.0;
      A     L      0.0;
      A     I    282.2;
      AN    I    282.3;
      =     M   1053.6;
      A     L      0.0;
      AN    I    282.2;
      A     I    282.3;
      =     M   1053.7;
NETWORK
TITLE =

      A     M      3.3;
      =     L      0.0;
      A     L      0.0;
      A     I    277.2;
      AN    I    277.3;
      =     M   1054.0;
      A     L      0.0;
      AN    I    277.2;
      A     I    277.3;
      =     M   1054.1;
NETWORK
TITLE =

      A     M      3.3;
      =     L      0.0;
      A     L      0.0;
      A     I    277.4;
      AN    I    277.5;
      =     M   1054.3;
      A     L      0.0;
      AN    I    277.4;
      A     I    277.5;
      =     M   1054.4;
NETWORK
TITLE =

      A     M      3.3;
      =     L      0.0;
      A     L      0.0;
      A     M   1051.6;
      A     M   1052.0;
      A     M   1052.2;
      A     M   1052.4;
      =     M   1055.0;
      A     L      0.0;
      A     M   1051.7;
      A     M   1052.1;
      A     M   1052.3;
      A     M   1052.5;
      =     M   1055.1;
NETWORK
TITLE =

      A     M      3.3;
      =     L      0.0;
      A     L      0.0;
      A     M   1052.6;
      A     M   1053.0;
      =     M   1055.2;
      A     L      0.0;
      A     M   1052.7;
      A     M   1053.1;
      =     M   1055.3;
NETWORK
TITLE =

      A     M      3.3;
      =     L      0.0;
      A     L      0.0;
      A     M   1053.2;
      A     M   1053.4;
      A     M   1053.6;
      =     M   1055.4;
      A     L      0.0;
      A     M   1053.3;
      A     M   1053.5;
      A     M   1053.7;
      =     M   1055.5;
      A     L      0.0;
      A     M   1051.1;
      A     M   1055.1;
      A     M   1055.3;
      A     M   1055.5;
      A     M   1054.4;
      =     M   1055.6;
      A     L      0.0;
      A     M   1051.3;
      A     M   1051.5;
      A     M   1055.1;
      A     M   1055.3;
      A     M   1055.5;
      A     M   1054.4;
      =     L      0.1;
      A     L      0.1;
      A     M   1051.1;
      =     M   1055.7;
      A     L      0.1;
      A(    ;
      O     M   1051.0;
      O     M   1051.1;
      )     ;
      =     M   1054.7;
NETWORK
TITLE =

      A     I    282.4;
      A     I    282.6;
      =     M   1056.0;
NETWORK
TITLE =

      A(    ;
      A     M   1000.5;
      A     DB51.DBX  204.0;
      A     DB51.DBX  203.6;
      AN    DB51.DBX  203.7;
      O     ;
      A     M   1000.6;
      AN    M   1001.0;
      A     M   1050.1;
      A     M   1001.7;
      )     ;
      A(    ;
      O     T    122;
      O     ;
      A     M   1000.5;
      A     I    244.4;
      )     ;
      AN    M   1051.0;
      AN    Q    284.1;
      =     Q    284.0;
NETWORK
TITLE =
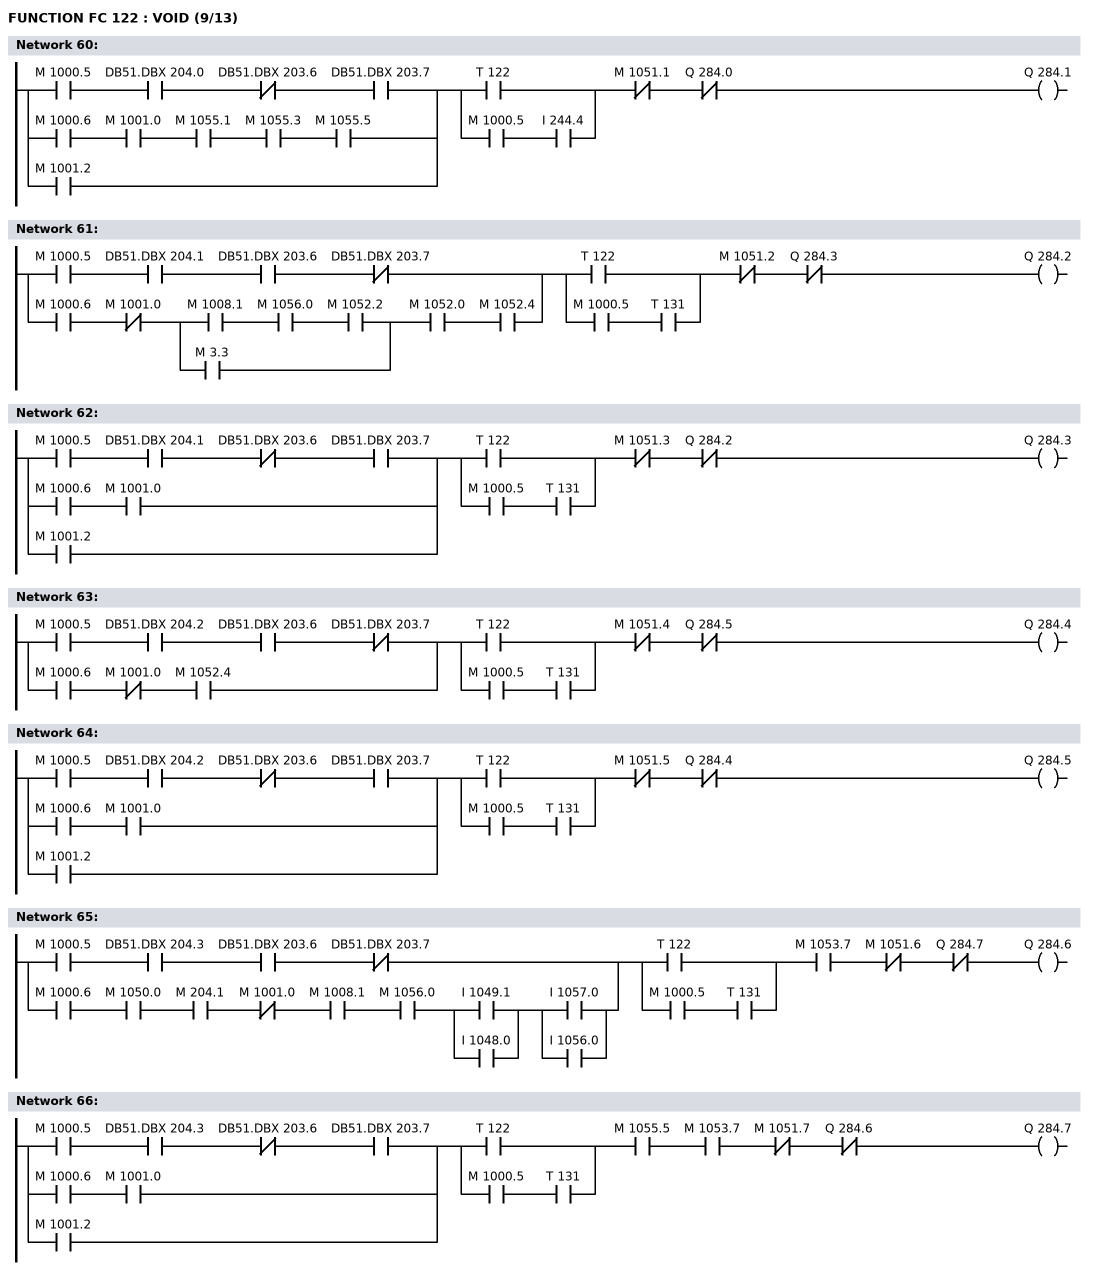

      A(    ;
      A     M   1000.5;
      A     DB51.DBX  204.0;
      AN    DB51.DBX  203.6;
      A     DB51.DBX  203.7;
      O     ;
      A     M   1000.6;
      A     M   1001.0;
      A     M   1055.1;
      A     M   1055.3;
      A     M   1055.5;
      O     M   1001.2;
      )     ;
      A(    ;
      O     T    122;
      O     ;
      A     M   1000.5;
      A     I    244.4;
      )     ;
      AN    M   1051.1;
      AN    Q    284.0;
      =     Q    284.1;
NETWORK
TITLE =

      A(    ;
      A     M   1000.5;
      A     DB51.DBX  204.1;
      A     DB51.DBX  203.6;
      AN    DB51.DBX  203.7;
      O     ;
      A     M   1000.6;
      AN    M   1001.0;
      A(    ;
      A     M   1008.1;
      A     M   1056.0;
      A     M   1052.2;
      O     M      3.3;
      )     ;
      A     M   1052.0;
      A     M   1052.4;
      )     ;
      A(    ;
      O     T    122;
      O     ;
      A     M   1000.5;
      A     T    131;
      )     ;
      AN    M   1051.2;
      AN    Q    284.3;
      =     Q    284.2;
NETWORK
TITLE =

      A(    ;
      A     M   1000.5;
      A     DB51.DBX  204.1;
      AN    DB51.DBX  203.6;
      A     DB51.DBX  203.7;
      O     ;
      A     M   1000.6;
      A     M   1001.0;
      O     M   1001.2;
      )     ;
      A(    ;
      O     T    122;
      O     ;
      A     M   1000.5;
      A     T    131;
      )     ;
      AN    M   1051.3;
      AN    Q    284.2;
      =     Q    284.3;
NETWORK
TITLE =

      A(    ;
      A     M   1000.5;
      A     DB51.DBX  204.2;
      A     DB51.DBX  203.6;
      AN    DB51.DBX  203.7;
      O     ;
      A     M   1000.6;
      AN    M   1001.0;
      A     M   1052.4;
      )     ;
      A(    ;
      O     T    122;
      O     ;
      A     M   1000.5;
      A     T    131;
      )     ;
      AN    M   1051.4;
      AN    Q    284.5;
      =     Q    284.4;
NETWORK
TITLE =

      A(    ;
      A     M   1000.5;
      A     DB51.DBX  204.2;
      AN    DB51.DBX  203.6;
      A     DB51.DBX  203.7;
      O     ;
      A     M   1000.6;
      A     M   1001.0;
      O     M   1001.2;
      )     ;
      A(    ;
      O     T    122;
      O     ;
      A     M   1000.5;
      A     T    131;
      )     ;
      AN    M   1051.5;
      AN    Q    284.4;
      =     Q    284.5;
NETWORK
TITLE =

      A(    ;
      A     M   1000.5;
      A     DB51.DBX  204.3;
      A     DB51.DBX  203.6;
      AN    DB51.DBX  203.7;
      O     ;
      A     M   1000.6;
      A     M   1050.0;
      A     M    204.1;
      AN    M   1001.0;
      A     M   1008.1;
      A     M   1056.0;
      A(    ;
      O     I   1049.1;
      O     I   1048.0;
      )     ;
      A(    ;
      O     I   1057.0;
      O     I   1056.0;
      )     ;
      )     ;
      A(    ;
      O     T    122;
      O     ;
      A     M   1000.5;
      A     T    131;
      )     ;
      A     M   1053.7;
      AN    M   1051.6;
      AN    Q    284.7;
      =     Q    284.6;
NETWORK
TITLE =

      A(    ;
      A     M   1000.5;
      A     DB51.DBX  204.3;
      AN    DB51.DBX  203.6;
      A     DB51.DBX  203.7;
      O     ;
      A     M   1000.6;
      A     M   1001.0;
      O     M   1001.2;
      )     ;
      A(    ;
      O     T    122;
      O     ;
      A     M   1000.5;
      A     T    131;
      )     ;
      A     M   1055.5;
      A     M   1053.7;
      AN    M   1051.7;
      AN    Q    284.6;
      =     Q    284.7;
NETWORK
TITLE =
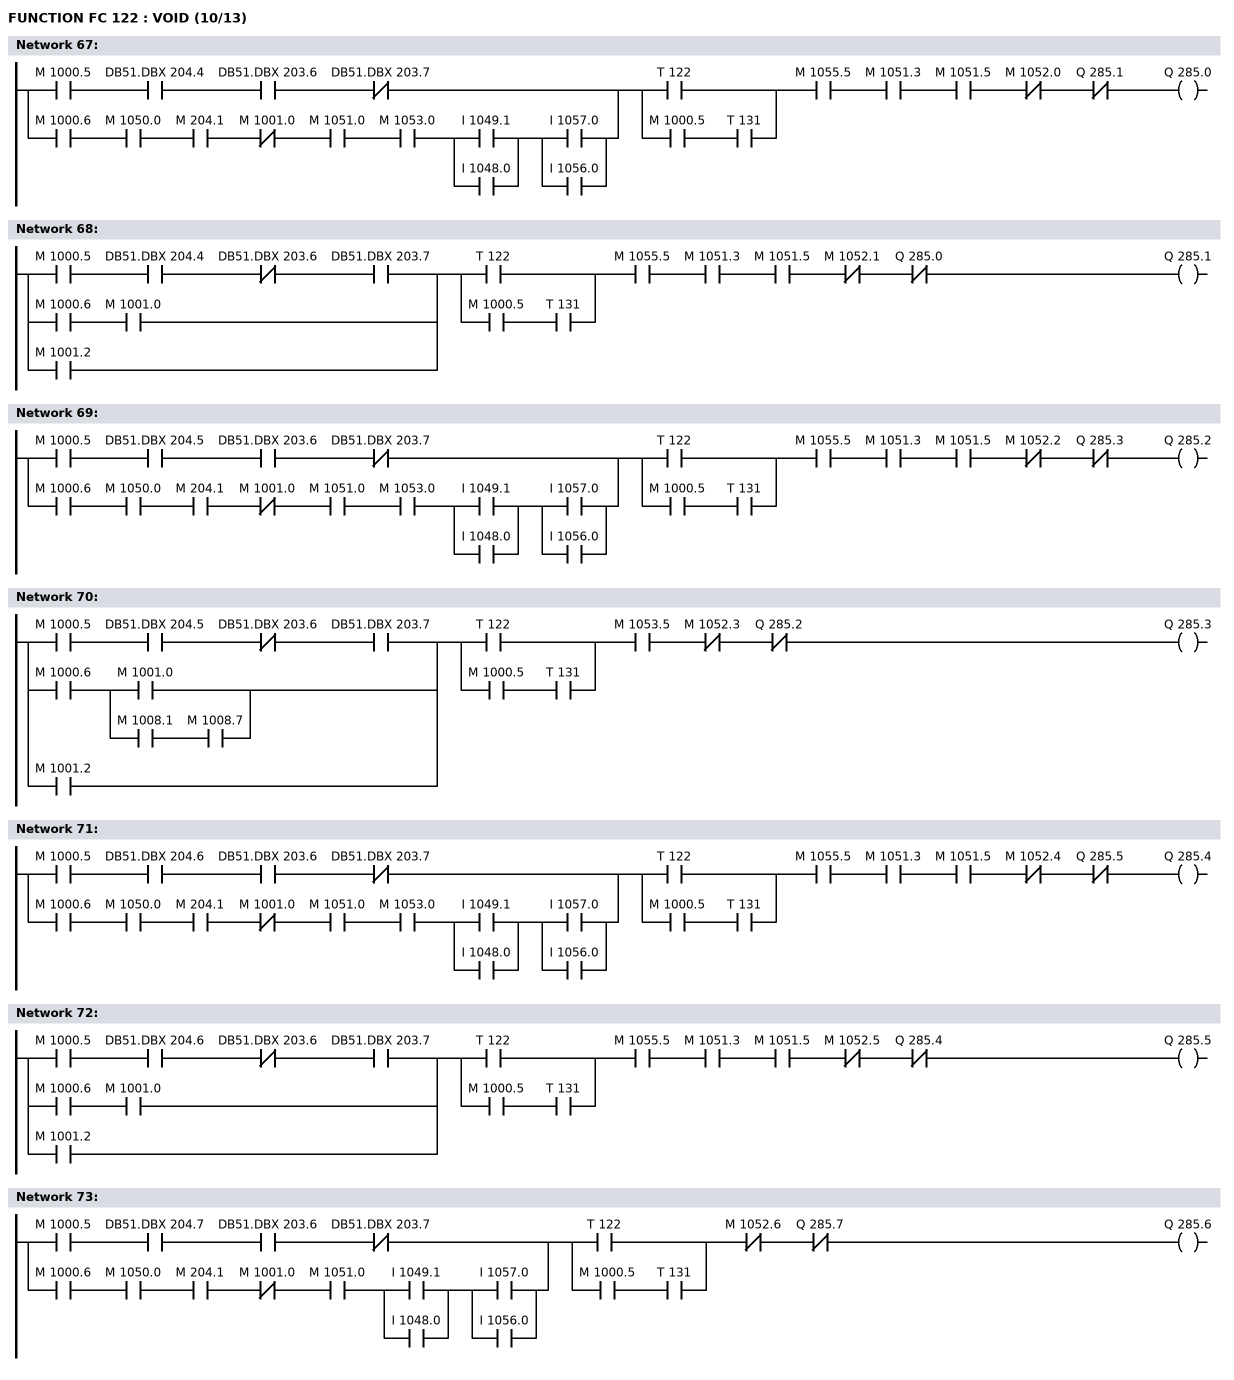

      A(    ;
      A     M   1000.5;
      A     DB51.DBX  204.4;
      A     DB51.DBX  203.6;
      AN    DB51.DBX  203.7;
      O     ;
      A     M   1000.6;
      A     M   1050.0;
      A     M    204.1;
      AN    M   1001.0;
      A     M   1051.0;
      A     M   1053.0;
      A(    ;
      O     I   1049.1;
      O     I   1048.0;
      )     ;
      A(    ;
      O     I   1057.0;
      O     I   1056.0;
      )     ;
      )     ;
      A(    ;
      O     T    122;
      O     ;
      A     M   1000.5;
      A     T    131;
      )     ;
      A     M   1055.5;
      A     M   1051.3;
      A     M   1051.5;
      AN    M   1052.0;
      AN    Q    285.1;
      =     Q    285.0;
NETWORK
TITLE =

      A(    ;
      A     M   1000.5;
      A     DB51.DBX  204.4;
      AN    DB51.DBX  203.6;
      A     DB51.DBX  203.7;
      O     ;
      A     M   1000.6;
      A     M   1001.0;
      O     M   1001.2;
      )     ;
      A(    ;
      O     T    122;
      O     ;
      A     M   1000.5;
      A     T    131;
      )     ;
      A     M   1055.5;
      A     M   1051.3;
      A     M   1051.5;
      AN    M   1052.1;
      AN    Q    285.0;
      =     Q    285.1;
NETWORK
TITLE =

      A(    ;
      A     M   1000.5;
      A     DB51.DBX  204.5;
      A     DB51.DBX  203.6;
      AN    DB51.DBX  203.7;
      O     ;
      A     M   1000.6;
      A     M   1050.0;
      A     M    204.1;
      AN    M   1001.0;
      A     M   1051.0;
      A     M   1053.0;
      A(    ;
      O     I   1049.1;
      O     I   1048.0;
      )     ;
      A(    ;
      O     I   1057.0;
      O     I   1056.0;
      )     ;
      )     ;
      A(    ;
      O     T    122;
      O     ;
      A     M   1000.5;
      A     T    131;
      )     ;
      A     M   1055.5;
      A     M   1051.3;
      A     M   1051.5;
      AN    M   1052.2;
      AN    Q    285.3;
      =     Q    285.2;
NETWORK
TITLE =

      A(    ;
      A     M   1000.5;
      A     DB51.DBX  204.5;
      AN    DB51.DBX  203.6;
      A     DB51.DBX  203.7;
      O     ;
      A     M   1000.6;
      A(    ;
      O     M   1001.0;
      O     ;
      A     M   1008.1;
      A     M   1008.7;
      )     ;
      O     M   1001.2;
      )     ;
      A(    ;
      O     T    122;
      O     ;
      A     M   1000.5;
      A     T    131;
      )     ;
      A     M   1053.5;
      AN    M   1052.3;
      AN    Q    285.2;
      =     Q    285.3;
NETWORK
TITLE =

      A(    ;
      A     M   1000.5;
      A     DB51.DBX  204.6;
      A     DB51.DBX  203.6;
      AN    DB51.DBX  203.7;
      O     ;
      A     M   1000.6;
      A     M   1050.0;
      A     M    204.1;
      AN    M   1001.0;
      A     M   1051.0;
      A     M   1053.0;
      A(    ;
      O     I   1049.1;
      O     I   1048.0;
      )     ;
      A(    ;
      O     I   1057.0;
      O     I   1056.0;
      )     ;
      )     ;
      A(    ;
      O     T    122;
      O     ;
      A     M   1000.5;
      A     T    131;
      )     ;
      A     M   1055.5;
      A     M   1051.3;
      A     M   1051.5;
      AN    M   1052.4;
      AN    Q    285.5;
      =     Q    285.4;
NETWORK
TITLE =

      A(    ;
      A     M   1000.5;
      A     DB51.DBX  204.6;
      AN    DB51.DBX  203.6;
      A     DB51.DBX  203.7;
      O     ;
      A     M   1000.6;
      A     M   1001.0;
      O     M   1001.2;
      )     ;
      A(    ;
      O     T    122;
      O     ;
      A     M   1000.5;
      A     T    131;
      )     ;
      A     M   1055.5;
      A     M   1051.3;
      A     M   1051.5;
      AN    M   1052.5;
      AN    Q    285.4;
      =     Q    285.5;
NETWORK
TITLE =

      A(    ;
      A     M   1000.5;
      A     DB51.DBX  204.7;
      A     DB51.DBX  203.6;
      AN    DB51.DBX  203.7;
      O     ;
      A     M   1000.6;
      A     M   1050.0;
      A     M    204.1;
      AN    M   1001.0;
      A     M   1051.0;
      A(    ;
      O     I   1049.1;
      O     I   1048.0;
      )     ;
      A(    ;
      O     I   1057.0;
      O     I   1056.0;
      )     ;
      )     ;
      A(    ;
      O     T    122;
      O     ;
      A     M   1000.5;
      A     T    131;
      )     ;
      AN    M   1052.6;
      AN    Q    285.7;
      =     Q    285.6;
NETWORK
TITLE =
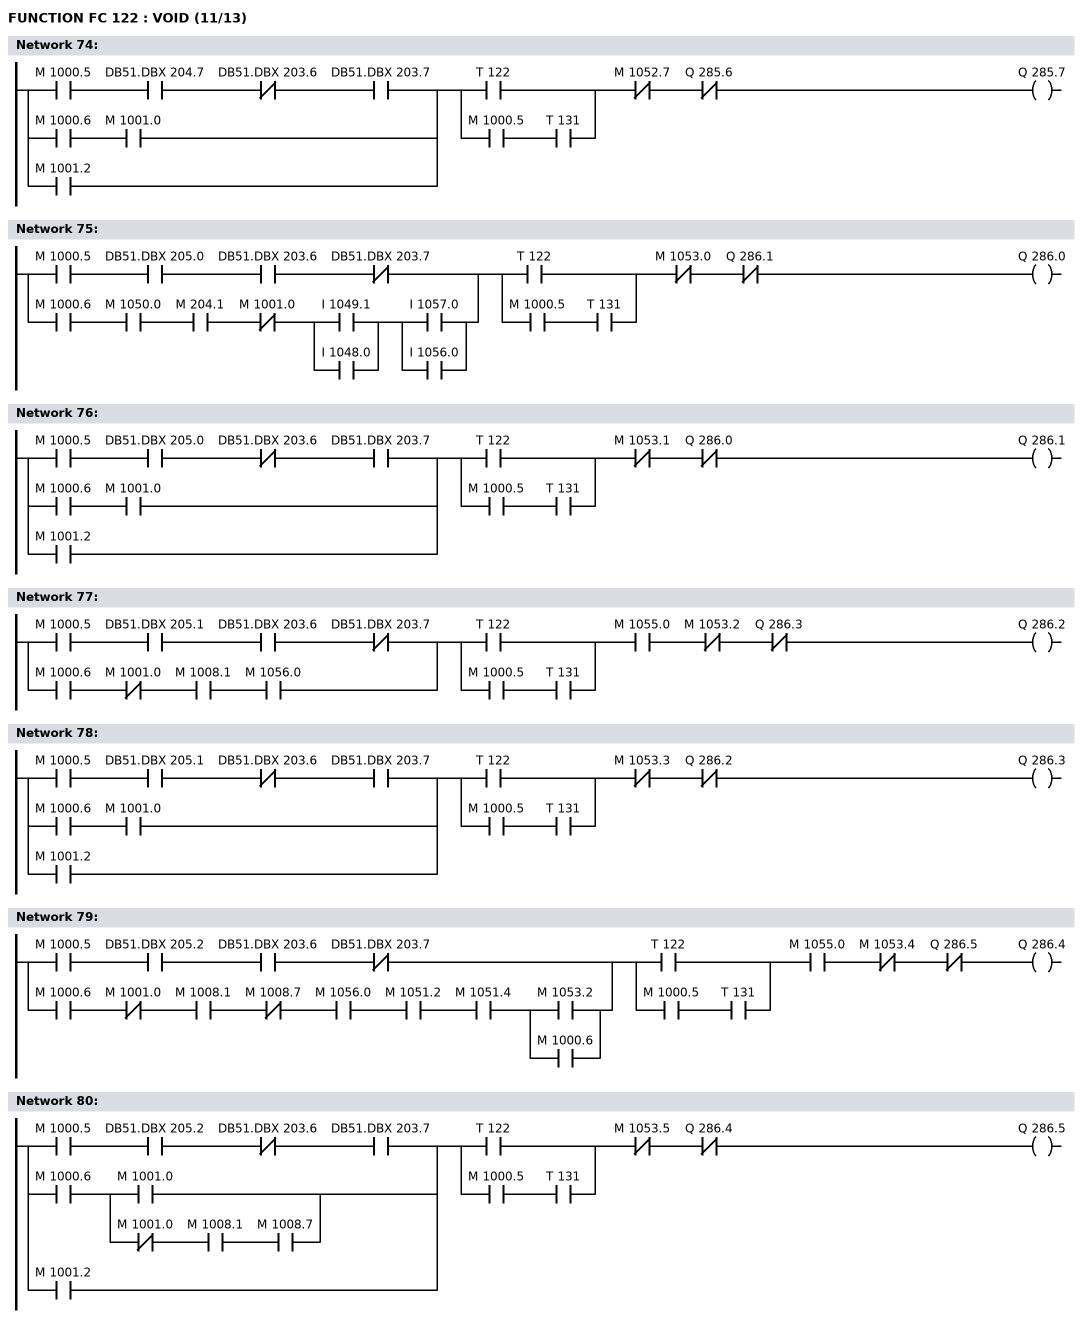

      A(    ;
      A     M   1000.5;
      A     DB51.DBX  204.7;
      AN    DB51.DBX  203.6;
      A     DB51.DBX  203.7;
      O     ;
      A     M   1000.6;
      A     M   1001.0;
      O     M   1001.2;
      )     ;
      A(    ;
      O     T    122;
      O     ;
      A     M   1000.5;
      A     T    131;
      )     ;
      AN    M   1052.7;
      AN    Q    285.6;
      =     Q    285.7;
NETWORK
TITLE =

      A(    ;
      A     M   1000.5;
      A     DB51.DBX  205.0;
      A     DB51.DBX  203.6;
      AN    DB51.DBX  203.7;
      O     ;
      A     M   1000.6;
      A     M   1050.0;
      A     M    204.1;
      AN    M   1001.0;
      A(    ;
      O     I   1049.1;
      O     I   1048.0;
      )     ;
      A(    ;
      O     I   1057.0;
      O     I   1056.0;
      )     ;
      )     ;
      A(    ;
      O     T    122;
      O     ;
      A     M   1000.5;
      A     T    131;
      )     ;
      AN    M   1053.0;
      AN    Q    286.1;
      =     Q    286.0;
NETWORK
TITLE =

      A(    ;
      A     M   1000.5;
      A     DB51.DBX  205.0;
      AN    DB51.DBX  203.6;
      A     DB51.DBX  203.7;
      O     ;
      A     M   1000.6;
      A     M   1001.0;
      O     M   1001.2;
      )     ;
      A(    ;
      O     T    122;
      O     ;
      A     M   1000.5;
      A     T    131;
      )     ;
      AN    M   1053.1;
      AN    Q    286.0;
      =     Q    286.1;
NETWORK
TITLE =

      A(    ;
      A     M   1000.5;
      A     DB51.DBX  205.1;
      A     DB51.DBX  203.6;
      AN    DB51.DBX  203.7;
      O     ;
      A     M   1000.6;
      AN    M   1001.0;
      A     M   1008.1;
      A     M   1056.0;
      )     ;
      A(    ;
      O     T    122;
      O     ;
      A     M   1000.5;
      A     T    131;
      )     ;
      A     M   1055.0;
      AN    M   1053.2;
      AN    Q    286.3;
      =     Q    286.2;
NETWORK
TITLE =

      A(    ;
      A     M   1000.5;
      A     DB51.DBX  205.1;
      AN    DB51.DBX  203.6;
      A     DB51.DBX  203.7;
      O     ;
      A     M   1000.6;
      A     M   1001.0;
      O     M   1001.2;
      )     ;
      A(    ;
      O     T    122;
      O     ;
      A     M   1000.5;
      A     T    131;
      )     ;
      AN    M   1053.3;
      AN    Q    286.2;
      =     Q    286.3;
NETWORK
TITLE =

      A(    ;
      A     M   1000.5;
      A     DB51.DBX  205.2;
      A     DB51.DBX  203.6;
      AN    DB51.DBX  203.7;
      O     ;
      A     M   1000.6;
      AN    M   1001.0;
      A     M   1008.1;
      AN    M   1008.7;
      A     M   1056.0;
      A     M   1051.2;
      A     M   1051.4;
      A(    ;
      O     M   1053.2;
      O     M   1000.6;
      )     ;
      )     ;
      A(    ;
      O     T    122;
      O     ;
      A     M   1000.5;
      A     T    131;
      )     ;
      A     M   1055.0;
      AN    M   1053.4;
      AN    Q    286.5;
      =     Q    286.4;
NETWORK
TITLE =

      A(    ;
      A     M   1000.5;
      A     DB51.DBX  205.2;
      AN    DB51.DBX  203.6;
      A     DB51.DBX  203.7;
      O     ;
      A     M   1000.6;
      A(    ;
      O     M   1001.0;
      O     ;
      AN    M   1001.0;
      A     M   1008.1;
      A     M   1008.7;
      )     ;
      O     M   1001.2;
      )     ;
      A(    ;
      O     T    122;
      O     ;
      A     M   1000.5;
      A     T    131;
      )     ;
      AN    M   1053.5;
      AN    Q    286.4;
      =     Q    286.5;
NETWORK
TITLE =
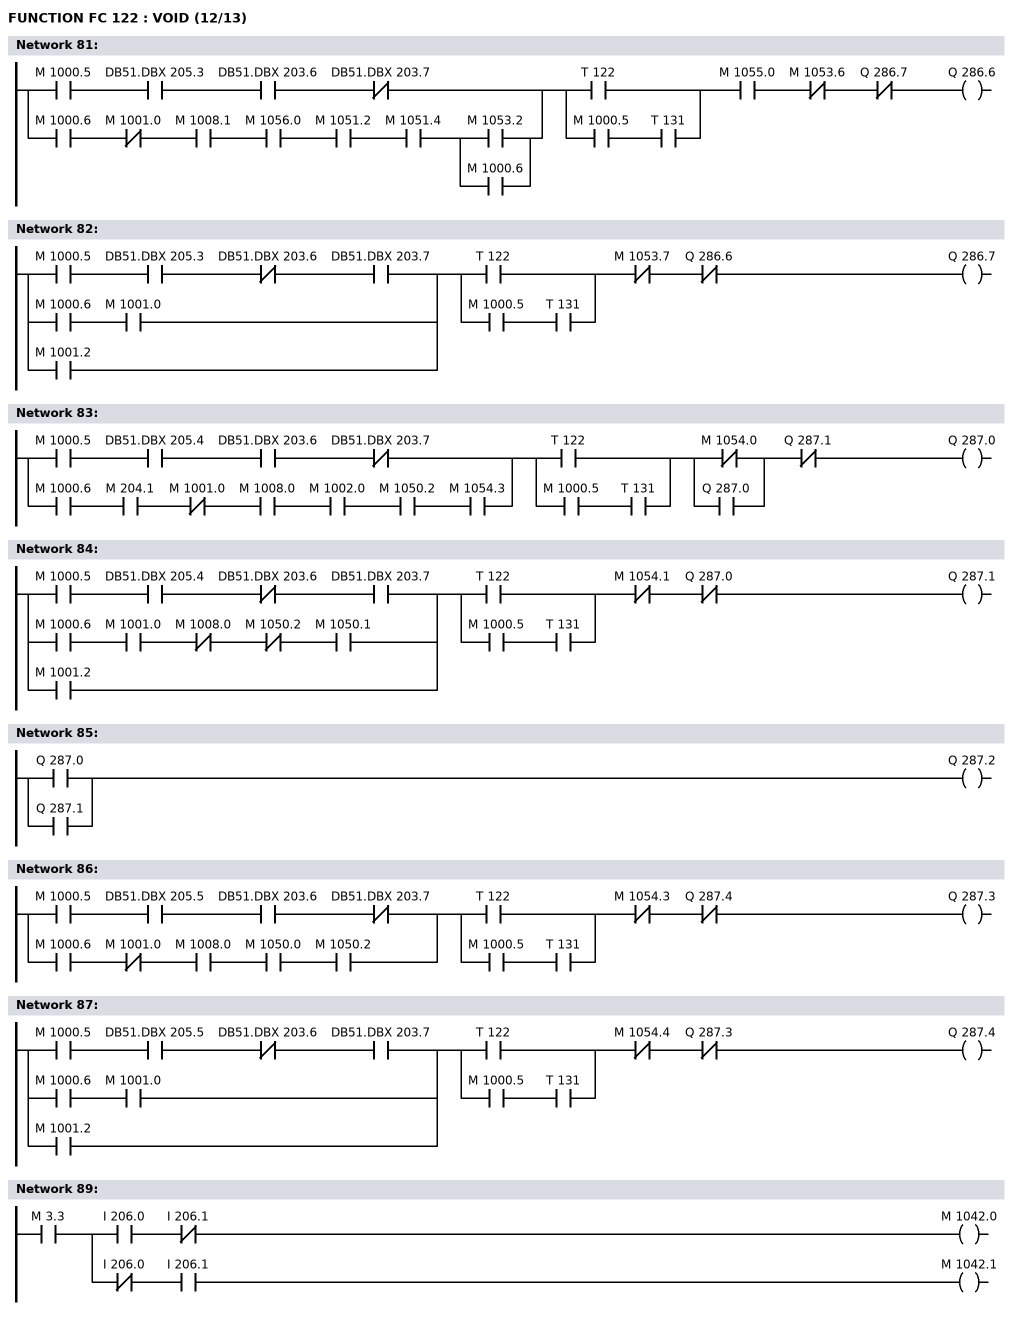

      A(    ;
      A     M   1000.5;
      A     DB51.DBX  205.3;
      A     DB51.DBX  203.6;
      AN    DB51.DBX  203.7;
      O     ;
      A     M   1000.6;
      AN    M   1001.0;
      A     M   1008.1;
      A     M   1056.0;
      A     M   1051.2;
      A     M   1051.4;
      A(    ;
      O     M   1053.2;
      O     M   1000.6;
      )     ;
      )     ;
      A(    ;
      O     T    122;
      O     ;
      A     M   1000.5;
      A     T    131;
      )     ;
      A     M   1055.0;
      AN    M   1053.6;
      AN    Q    286.7;
      =     Q    286.6;
NETWORK
TITLE =

      A(    ;
      A     M   1000.5;
      A     DB51.DBX  205.3;
      AN    DB51.DBX  203.6;
      A     DB51.DBX  203.7;
      O     ;
      A     M   1000.6;
      A     M   1001.0;
      O     M   1001.2;
      )     ;
      A(    ;
      O     T    122;
      O     ;
      A     M   1000.5;
      A     T    131;
      )     ;
      AN    M   1053.7;
      AN    Q    286.6;
      =     Q    286.7;
NETWORK
TITLE =

      A(    ;
      A     M   1000.5;
      A     DB51.DBX  205.4;
      A     DB51.DBX  203.6;
      AN    DB51.DBX  203.7;
      O     ;
      A     M   1000.6;
      A     M    204.1;
      AN    M   1001.0;
      A     M   1008.0;
      A     M   1002.0;
      A     M   1050.2;
      A     M   1054.3;
      )     ;
      A(    ;
      O     T    122;
      O     ;
      A     M   1000.5;
      A     T    131;
      )     ;
      A(    ;
      ON    M   1054.0;
      O     Q    287.0;
      )     ;
      AN    Q    287.1;
      =     Q    287.0;
NETWORK
TITLE =

      A(    ;
      A     M   1000.5;
      A     DB51.DBX  205.4;
      AN    DB51.DBX  203.6;
      A     DB51.DBX  203.7;
      O     ;
      A     M   1000.6;
      A     M   1001.0;
      AN    M   1008.0;
      AN    M   1050.2;
      A     M   1050.1;
      O     M   1001.2;
      )     ;
      A(    ;
      O     T    122;
      O     ;
      A     M   1000.5;
      A     T    131;
      )     ;
      AN    M   1054.1;
      AN    Q    287.0;
      =     Q    287.1;
NETWORK
TITLE =

      O     Q    287.0;
      O     Q    287.1;
      =     Q    287.2;
NETWORK
TITLE =

      A(    ;
      A     M   1000.5;
      A     DB51.DBX  205.5;
      A     DB51.DBX  203.6;
      AN    DB51.DBX  203.7;
      O     ;
      A     M   1000.6;
      AN    M   1001.0;
      A     M   1008.0;
      A     M   1050.0;
      A     M   1050.2;
      )     ;
      A(    ;
      O     T    122;
      O     ;
      A     M   1000.5;
      A     T    131;
      )     ;
      AN    M   1054.3;
      AN    Q    287.4;
      =     Q    287.3;
NETWORK
TITLE =

      A(    ;
      A     M   1000.5;
      A     DB51.DBX  205.5;
      AN    DB51.DBX  203.6;
      A     DB51.DBX  203.7;
      O     ;
      A     M   1000.6;
      A     M   1001.0;
      O     M   1001.2;
      )     ;
      A(    ;
      O     T    122;
      O     ;
      A     M   1000.5;
      A     T    131;
      )     ;
      AN    M   1054.4;
      AN    Q    287.3;
      =     Q    287.4;
NETWORK
TITLE =INDEX TL

NETWORK
TITLE =

      A     M      3.3;
      =     L      0.0;
      A     L      0.0;
      A     I    206.0;
      AN    I    206.1;
      =     M   1042.0;
      A     L      0.0;
      AN    I    206.0;
      A     I    206.1;
      =     M   1042.1;
NETWORK
TITLE =
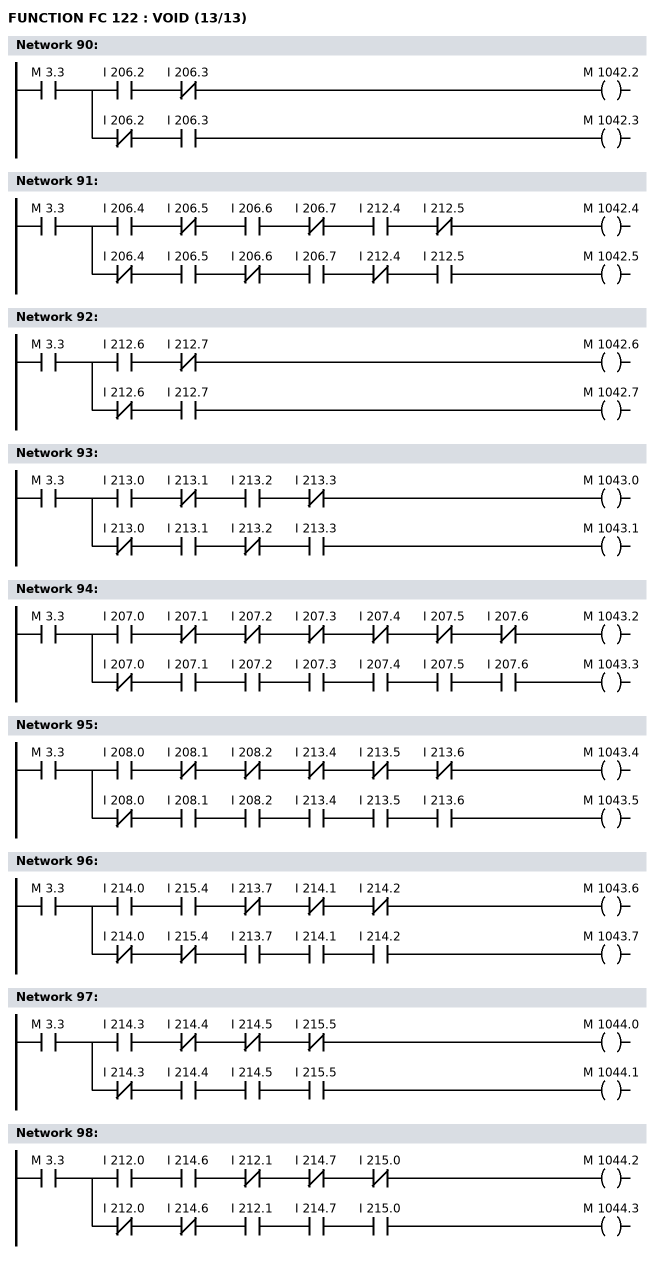

      A     M      3.3;
      =     L      0.0;
      A     L      0.0;
      A     I    206.2;
      AN    I    206.3;
      =     M   1042.2;
      A     L      0.0;
      AN    I    206.2;
      A     I    206.3;
      =     M   1042.3;
NETWORK
TITLE =

      A     M      3.3;
      =     L      0.0;
      A     L      0.0;
      A     I    206.4;
      AN    I    206.5;
      A     I    206.6;
      AN    I    206.7;
      A     I    212.4;
      AN    I    212.5;
      =     M   1042.4;
      A     L      0.0;
      AN    I    206.4;
      A     I    206.5;
      AN    I    206.6;
      A     I    206.7;
      AN    I    212.4;
      A     I    212.5;
      =     M   1042.5;
NETWORK
TITLE =

      A     M      3.3;
      =     L      0.0;
      A     L      0.0;
      A     I    212.6;
      AN    I    212.7;
      =     M   1042.6;
      A     L      0.0;
      AN    I    212.6;
      A     I    212.7;
      =     M   1042.7;
NETWORK
TITLE =

      A     M      3.3;
      =     L      0.0;
      A     L      0.0;
      A     I    213.0;
      AN    I    213.1;
      A     I    213.2;
      AN    I    213.3;
      =     M   1043.0;
      A     L      0.0;
      AN    I    213.0;
      A     I    213.1;
      AN    I    213.2;
      A     I    213.3;
      =     M   1043.1;
NETWORK
TITLE =

      A     M      3.3;
      =     L      0.0;
      A     L      0.0;
      A     I    207.0;
      AN    I    207.1;
      AN    I    207.2;
      AN    I    207.3;
      AN    I    207.4;
      AN    I    207.5;
      AN    I    207.6;
      =     M   1043.2;
      A     L      0.0;
      AN    I    207.0;
      A     I    207.1;
      A     I    207.2;
      A     I    207.3;
      A     I    207.4;
      A     I    207.5;
      A     I    207.6;
      =     M   1043.3;
NETWORK
TITLE =

      A     M      3.3;
      =     L      0.0;
      A     L      0.0;
      A     I    208.0;
      AN    I    208.1;
      AN    I    208.2;
      AN    I    213.4;
      AN    I    213.5;
      AN    I    213.6;
      =     M   1043.4;
      A     L      0.0;
      AN    I    208.0;
      A     I    208.1;
      A     I    208.2;
      A     I    213.4;
      A     I    213.5;
      A     I    213.6;
      =     M   1043.5;
NETWORK
TITLE =

      A     M      3.3;
      =     L      0.0;
      A     L      0.0;
      A     I    214.0;
      A     I    215.4;
      AN    I    213.7;
      AN    I    214.1;
      AN    I    214.2;
      =     M   1043.6;
      A     L      0.0;
      AN    I    214.0;
      AN    I    215.4;
      A     I    213.7;
      A     I    214.1;
      A     I    214.2;
      =     M   1043.7;
NETWORK
TITLE =

      A     M      3.3;
      =     L      0.0;
      A     L      0.0;
      A     I    214.3;
      AN    I    214.4;
      AN    I    214.5;
      AN    I    215.5;
      =     M   1044.0;
      A     L      0.0;
      AN    I    214.3;
      A     I    214.4;
      A     I    214.5;
      A     I    215.5;
      =     M   1044.1;
NETWORK
TITLE =

      A     M      3.3;
      =     L      0.0;
      A     L      0.0;
      A     I    212.0;
      A     I    214.6;
      AN    I    212.1;
      AN    I    214.7;
      AN    I    215.0;
      =     M   1044.2;
      A     L      0.0;
      AN    I    212.0;
      AN    I    214.6;
      A     I    212.1;
      A     I    214.7;
      A     I    215.0;
      =     M   1044.3;
NETWORK
TITLE =

      A     M      3.3;
      =     L      0.0;
      A     L      0.0;
      A     I    208.4;
      AN    I    208.5;
      =     L      0.1;
      A     L      0.1;
      A     T     10;
      =     M   1044.4;
      A     L      0.1;
      BLD   102;
      L     S5T#1S;
      SD    T     10;
      A     L      0.1;
      BLD   102;
      L     S5T#500MS;
      SD    T     30;
      A     L      0.0;
      AN    I    208.4;
      A     I    208.5;
      =     L      0.1;
      A     L      0.1;
      A     T     11;
      =     M   1044.5;
      A     L      0.1;
      BLD   102;
      L     S5T#1S;
      SD    T     11;
      A     L      0.1;
      BLD   102;
      L     S5T#500MS;
      SD    T     31;
NETWORK
TITLE =
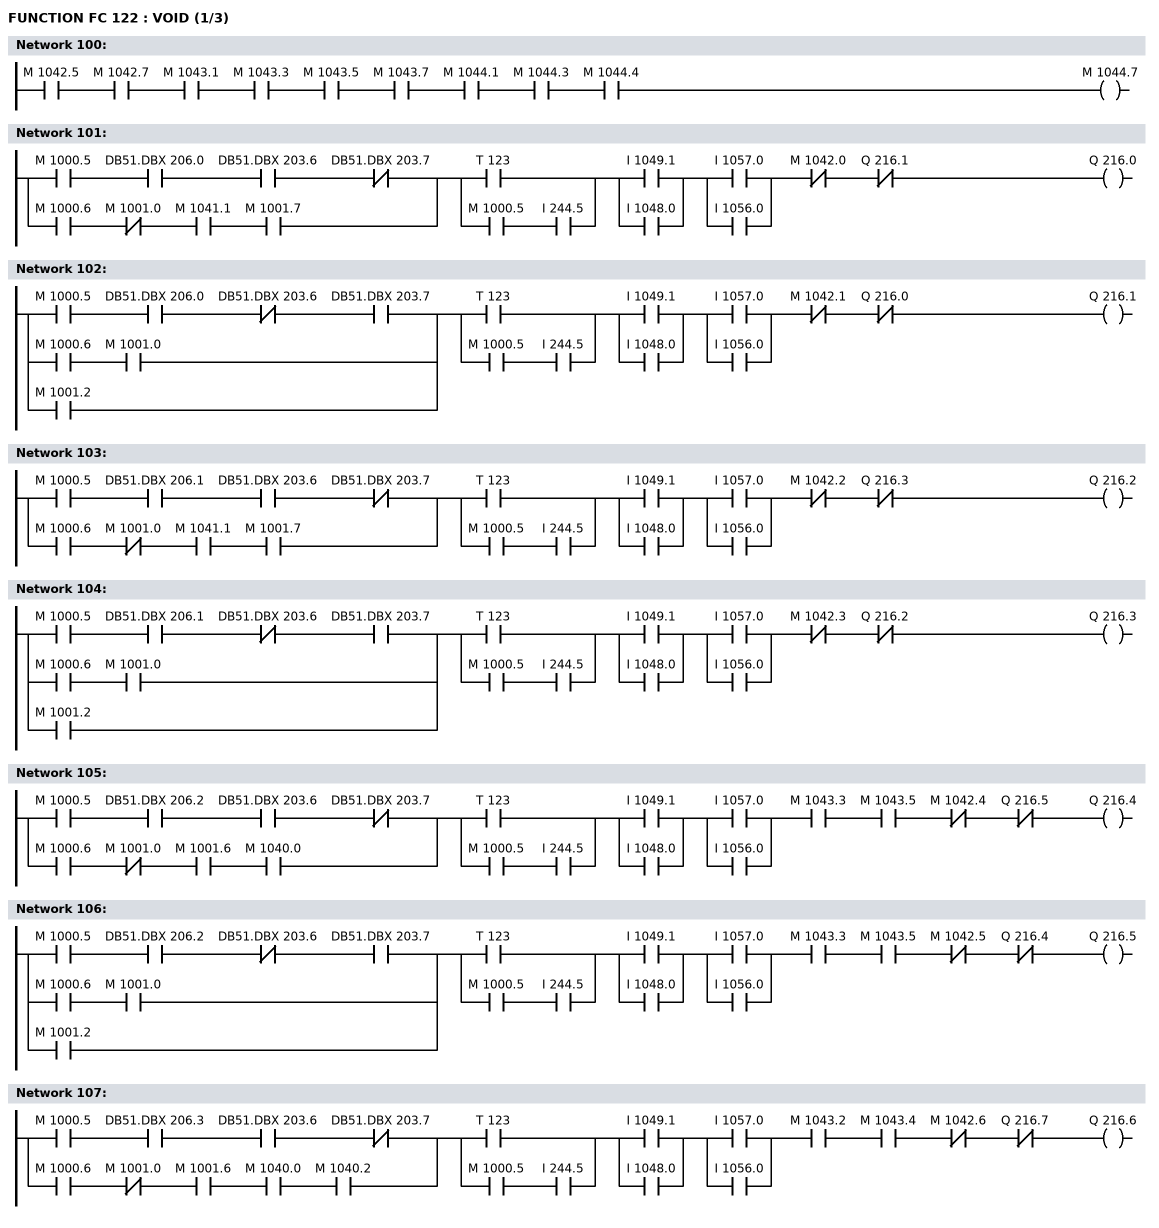

      A     M   1042.5;
      A     M   1042.7;
      A     M   1043.1;
      A     M   1043.3;
      A     M   1043.5;
      A     M   1043.7;
      A     M   1044.1;
      A     M   1044.3;
      A     M   1044.4;
      =     M   1044.7;
NETWORK
TITLE =

      A(    ;
      A     M   1000.5;
      A     DB51.DBX  206.0;
      A     DB51.DBX  203.6;
      AN    DB51.DBX  203.7;
      O     ;
      A     M   1000.6;
      AN    M   1001.0;
      A     M   1041.1;
      A     M   1001.7;
      )     ;
      A(    ;
      O     T    123;
      O     ;
      A     M   1000.5;
      A     I    244.5;
      )     ;
      A(    ;
      O     I   1049.1;
      O     I   1048.0;
      )     ;
      A(    ;
      O     I   1057.0;
      O     I   1056.0;
      )     ;
      AN    M   1042.0;
      AN    Q    216.1;
      =     Q    216.0;
NETWORK
TITLE =

      A(    ;
      A     M   1000.5;
      A     DB51.DBX  206.0;
      AN    DB51.DBX  203.6;
      A     DB51.DBX  203.7;
      O     ;
      A     M   1000.6;
      A     M   1001.0;
      O     M   1001.2;
      )     ;
      A(    ;
      O     T    123;
      O     ;
      A     M   1000.5;
      A     I    244.5;
      )     ;
      A(    ;
      O     I   1049.1;
      O     I   1048.0;
      )     ;
      A(    ;
      O     I   1057.0;
      O     I   1056.0;
      )     ;
      AN    M   1042.1;
      AN    Q    216.0;
      =     Q    216.1;
NETWORK
TITLE =

      A(    ;
      A     M   1000.5;
      A     DB51.DBX  206.1;
      A     DB51.DBX  203.6;
      AN    DB51.DBX  203.7;
      O     ;
      A     M   1000.6;
      AN    M   1001.0;
      A     M   1041.1;
      A     M   1001.7;
      )     ;
      A(    ;
      O     T    123;
      O     ;
      A     M   1000.5;
      A     I    244.5;
      )     ;
      A(    ;
      O     I   1049.1;
      O     I   1048.0;
      )     ;
      A(    ;
      O     I   1057.0;
      O     I   1056.0;
      )     ;
      AN    M   1042.2;
      AN    Q    216.3;
      =     Q    216.2;
NETWORK
TITLE =

      A(    ;
      A     M   1000.5;
      A     DB51.DBX  206.1;
      AN    DB51.DBX  203.6;
      A     DB51.DBX  203.7;
      O     ;
      A     M   1000.6;
      A     M   1001.0;
      O     M   1001.2;
      )     ;
      A(    ;
      O     T    123;
      O     ;
      A     M   1000.5;
      A     I    244.5;
      )     ;
      A(    ;
      O     I   1049.1;
      O     I   1048.0;
      )     ;
      A(    ;
      O     I   1057.0;
      O     I   1056.0;
      )     ;
      AN    M   1042.3;
      AN    Q    216.2;
      =     Q    216.3;
NETWORK
TITLE =

      A(    ;
      A     M   1000.5;
      A     DB51.DBX  206.2;
      A     DB51.DBX  203.6;
      AN    DB51.DBX  203.7;
      O     ;
      A     M   1000.6;
      AN    M   1001.0;
      A     M   1001.6;
      A     M   1040.0;
      )     ;
      A(    ;
      O     T    123;
      O     ;
      A     M   1000.5;
      A     I    244.5;
      )     ;
      A(    ;
      O     I   1049.1;
      O     I   1048.0;
      )     ;
      A(    ;
      O     I   1057.0;
      O     I   1056.0;
      )     ;
      A     M   1043.3;
      A     M   1043.5;
      AN    M   1042.4;
      AN    Q    216.5;
      =     Q    216.4;
NETWORK
TITLE =

      A(    ;
      A     M   1000.5;
      A     DB51.DBX  206.2;
      AN    DB51.DBX  203.6;
      A     DB51.DBX  203.7;
      O     ;
      A     M   1000.6;
      A     M   1001.0;
      O     M   1001.2;
      )     ;
      A(    ;
      O     T    123;
      O     ;
      A     M   1000.5;
      A     I    244.5;
      )     ;
      A(    ;
      O     I   1049.1;
      O     I   1048.0;
      )     ;
      A(    ;
      O     I   1057.0;
      O     I   1056.0;
      )     ;
      A     M   1043.3;
      A     M   1043.5;
      AN    M   1042.5;
      AN    Q    216.4;
      =     Q    216.5;
NETWORK
TITLE =

      A(    ;
      A     M   1000.5;
      A     DB51.DBX  206.3;
      A     DB51.DBX  203.6;
      AN    DB51.DBX  203.7;
      O     ;
      A     M   1000.6;
      AN    M   1001.0;
      A     M   1001.6;
      A     M   1040.0;
      A     M   1040.2;
      )     ;
      A(    ;
      O     T    123;
      O     ;
      A     M   1000.5;
      A     I    244.5;
      )     ;
      A(    ;
      O     I   1049.1;
      O     I   1048.0;
      )     ;
      A(    ;
      O     I   1057.0;
      O     I   1056.0;
      )     ;
      A     M   1043.2;
      A     M   1043.4;
      AN    M   1042.6;
      AN    Q    216.7;
      =     Q    216.6;
NETWORK
TITLE =
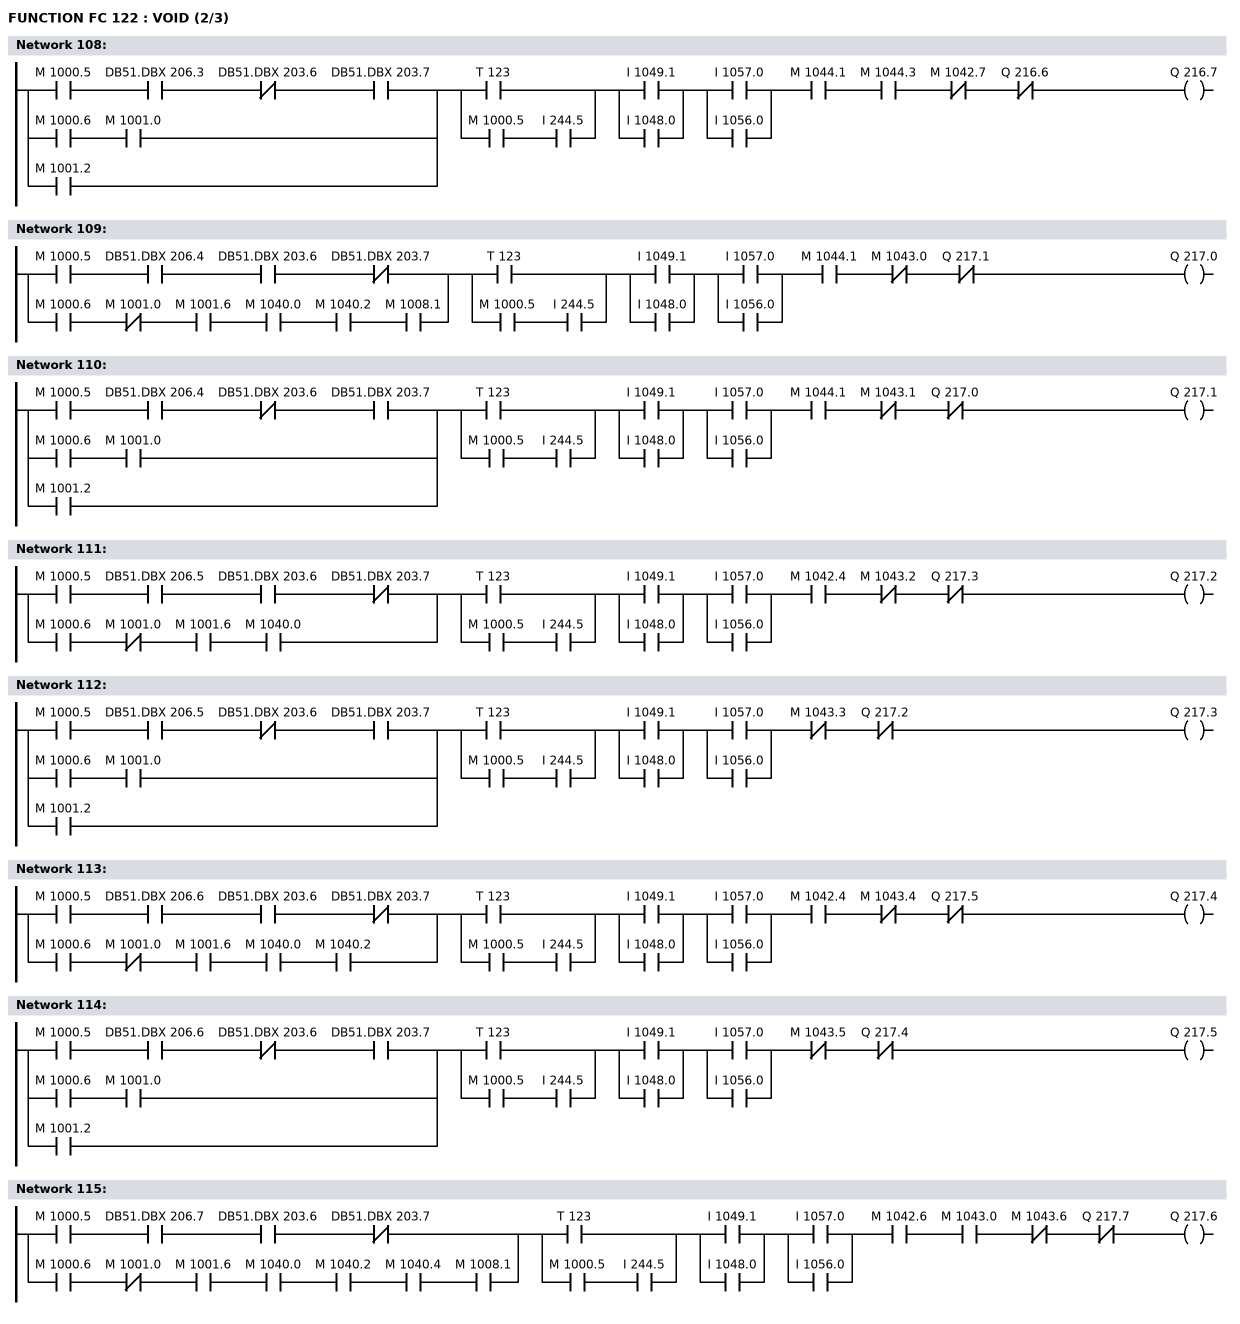

      A(    ;
      A     M   1000.5;
      A     DB51.DBX  206.3;
      AN    DB51.DBX  203.6;
      A     DB51.DBX  203.7;
      O     ;
      A     M   1000.6;
      A     M   1001.0;
      O     M   1001.2;
      )     ;
      A(    ;
      O     T    123;
      O     ;
      A     M   1000.5;
      A     I    244.5;
      )     ;
      A(    ;
      O     I   1049.1;
      O     I   1048.0;
      )     ;
      A(    ;
      O     I   1057.0;
      O     I   1056.0;
      )     ;
      A     M   1044.1;
      A     M   1044.3;
      AN    M   1042.7;
      AN    Q    216.6;
      =     Q    216.7;
NETWORK
TITLE =

      A(    ;
      A     M   1000.5;
      A     DB51.DBX  206.4;
      A     DB51.DBX  203.6;
      AN    DB51.DBX  203.7;
      O     ;
      A     M   1000.6;
      AN    M   1001.0;
      A     M   1001.6;
      A     M   1040.0;
      A     M   1040.2;
      A     M   1008.1;
      )     ;
      A(    ;
      O     T    123;
      O     ;
      A     M   1000.5;
      A     I    244.5;
      )     ;
      A(    ;
      O     I   1049.1;
      O     I   1048.0;
      )     ;
      A(    ;
      O     I   1057.0;
      O     I   1056.0;
      )     ;
      A     M   1044.1;
      AN    M   1043.0;
      AN    Q    217.1;
      =     Q    217.0;
NETWORK
TITLE =

      A(    ;
      A     M   1000.5;
      A     DB51.DBX  206.4;
      AN    DB51.DBX  203.6;
      A     DB51.DBX  203.7;
      O     ;
      A     M   1000.6;
      A     M   1001.0;
      O     M   1001.2;
      )     ;
      A(    ;
      O     T    123;
      O     ;
      A     M   1000.5;
      A     I    244.5;
      )     ;
      A(    ;
      O     I   1049.1;
      O     I   1048.0;
      )     ;
      A(    ;
      O     I   1057.0;
      O     I   1056.0;
      )     ;
      A     M   1044.1;
      AN    M   1043.1;
      AN    Q    217.0;
      =     Q    217.1;
NETWORK
TITLE =

      A(    ;
      A     M   1000.5;
      A     DB51.DBX  206.5;
      A     DB51.DBX  203.6;
      AN    DB51.DBX  203.7;
      O     ;
      A     M   1000.6;
      AN    M   1001.0;
      A     M   1001.6;
      A     M   1040.0;
      )     ;
      A(    ;
      O     T    123;
      O     ;
      A     M   1000.5;
      A     I    244.5;
      )     ;
      A(    ;
      O     I   1049.1;
      O     I   1048.0;
      )     ;
      A(    ;
      O     I   1057.0;
      O     I   1056.0;
      )     ;
      A     M   1042.4;
      AN    M   1043.2;
      AN    Q    217.3;
      =     Q    217.2;
NETWORK
TITLE =

      A(    ;
      A     M   1000.5;
      A     DB51.DBX  206.5;
      AN    DB51.DBX  203.6;
      A     DB51.DBX  203.7;
      O     ;
      A     M   1000.6;
      A     M   1001.0;
      O     M   1001.2;
      )     ;
      A(    ;
      O     T    123;
      O     ;
      A     M   1000.5;
      A     I    244.5;
      )     ;
      A(    ;
      O     I   1049.1;
      O     I   1048.0;
      )     ;
      A(    ;
      O     I   1057.0;
      O     I   1056.0;
      )     ;
      AN    M   1043.3;
      AN    Q    217.2;
      =     Q    217.3;
NETWORK
TITLE =

      A(    ;
      A     M   1000.5;
      A     DB51.DBX  206.6;
      A     DB51.DBX  203.6;
      AN    DB51.DBX  203.7;
      O     ;
      A     M   1000.6;
      AN    M   1001.0;
      A     M   1001.6;
      A     M   1040.0;
      A     M   1040.2;
      )     ;
      A(    ;
      O     T    123;
      O     ;
      A     M   1000.5;
      A     I    244.5;
      )     ;
      A(    ;
      O     I   1049.1;
      O     I   1048.0;
      )     ;
      A(    ;
      O     I   1057.0;
      O     I   1056.0;
      )     ;
      A     M   1042.4;
      AN    M   1043.4;
      AN    Q    217.5;
      =     Q    217.4;
NETWORK
TITLE =

      A(    ;
      A     M   1000.5;
      A     DB51.DBX  206.6;
      AN    DB51.DBX  203.6;
      A     DB51.DBX  203.7;
      O     ;
      A     M   1000.6;
      A     M   1001.0;
      O     M   1001.2;
      )     ;
      A(    ;
      O     T    123;
      O     ;
      A     M   1000.5;
      A     I    244.5;
      )     ;
      A(    ;
      O     I   1049.1;
      O     I   1048.0;
      )     ;
      A(    ;
      O     I   1057.0;
      O     I   1056.0;
      )     ;
      AN    M   1043.5;
      AN    Q    217.4;
      =     Q    217.5;
NETWORK
TITLE =

      A(    ;
      A     M   1000.5;
      A     DB51.DBX  206.7;
      A     DB51.DBX  203.6;
      AN    DB51.DBX  203.7;
      O     ;
      A     M   1000.6;
      AN    M   1001.0;
      A     M   1001.6;
      A     M   1040.0;
      A     M   1040.2;
      A     M   1040.4;
      A     M   1008.1;
      )     ;
      A(    ;
      O     T    123;
      O     ;
      A     M   1000.5;
      A     I    244.5;
      )     ;
      A(    ;
      O     I   1049.1;
      O     I   1048.0;
      )     ;
      A(    ;
      O     I   1057.0;
      O     I   1056.0;
      )     ;
      A     M   1042.6;
      A     M   1043.0;
      AN    M   1043.6;
      AN    Q    217.7;
      =     Q    217.6;
NETWORK
TITLE =
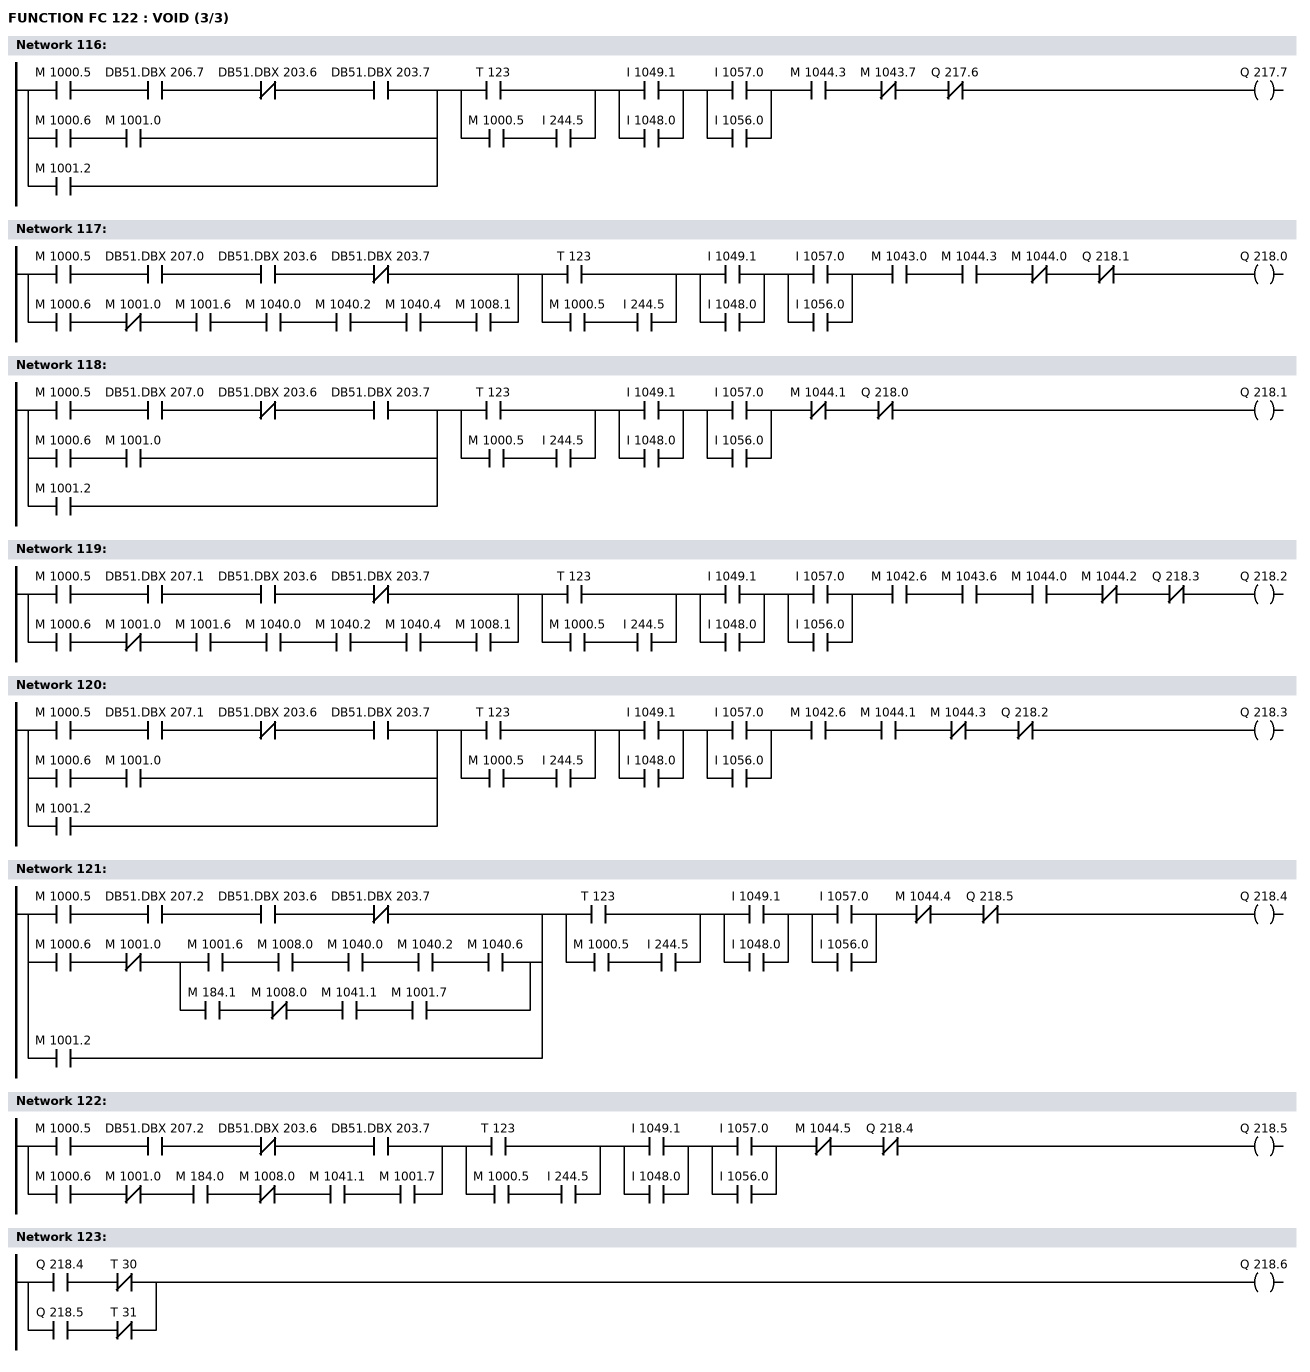

      A(    ;
      A     M   1000.5;
      A     DB51.DBX  206.7;
      AN    DB51.DBX  203.6;
      A     DB51.DBX  203.7;
      O     ;
      A     M   1000.6;
      A     M   1001.0;
      O     M   1001.2;
      )     ;
      A(    ;
      O     T    123;
      O     ;
      A     M   1000.5;
      A     I    244.5;
      )     ;
      A(    ;
      O     I   1049.1;
      O     I   1048.0;
      )     ;
      A(    ;
      O     I   1057.0;
      O     I   1056.0;
      )     ;
      A     M   1044.3;
      AN    M   1043.7;
      AN    Q    217.6;
      =     Q    217.7;
NETWORK
TITLE =

      A(    ;
      A     M   1000.5;
      A     DB51.DBX  207.0;
      A     DB51.DBX  203.6;
      AN    DB51.DBX  203.7;
      O     ;
      A     M   1000.6;
      AN    M   1001.0;
      A     M   1001.6;
      A     M   1040.0;
      A     M   1040.2;
      A     M   1040.4;
      A     M   1008.1;
      )     ;
      A(    ;
      O     T    123;
      O     ;
      A     M   1000.5;
      A     I    244.5;
      )     ;
      A(    ;
      O     I   1049.1;
      O     I   1048.0;
      )     ;
      A(    ;
      O     I   1057.0;
      O     I   1056.0;
      )     ;
      A     M   1043.0;
      A     M   1044.3;
      AN    M   1044.0;
      AN    Q    218.1;
      =     Q    218.0;
NETWORK
TITLE =

      A(    ;
      A     M   1000.5;
      A     DB51.DBX  207.0;
      AN    DB51.DBX  203.6;
      A     DB51.DBX  203.7;
      O     ;
      A     M   1000.6;
      A     M   1001.0;
      O     M   1001.2;
      )     ;
      A(    ;
      O     T    123;
      O     ;
      A     M   1000.5;
      A     I    244.5;
      )     ;
      A(    ;
      O     I   1049.1;
      O     I   1048.0;
      )     ;
      A(    ;
      O     I   1057.0;
      O     I   1056.0;
      )     ;
      AN    M   1044.1;
      AN    Q    218.0;
      =     Q    218.1;
NETWORK
TITLE =

      A(    ;
      A     M   1000.5;
      A     DB51.DBX  207.1;
      A     DB51.DBX  203.6;
      AN    DB51.DBX  203.7;
      O     ;
      A     M   1000.6;
      AN    M   1001.0;
      A     M   1001.6;
      A     M   1040.0;
      A     M   1040.2;
      A     M   1040.4;
      A     M   1008.1;
      )     ;
      A(    ;
      O     T    123;
      O     ;
      A     M   1000.5;
      A     I    244.5;
      )     ;
      A(    ;
      O     I   1049.1;
      O     I   1048.0;
      )     ;
      A(    ;
      O     I   1057.0;
      O     I   1056.0;
      )     ;
      A     M   1042.6;
      A     M   1043.6;
      A     M   1044.0;
      AN    M   1044.2;
      AN    Q    218.3;
      =     Q    218.2;
NETWORK
TITLE =

      A(    ;
      A     M   1000.5;
      A     DB51.DBX  207.1;
      AN    DB51.DBX  203.6;
      A     DB51.DBX  203.7;
      O     ;
      A     M   1000.6;
      A     M   1001.0;
      O     M   1001.2;
      )     ;
      A(    ;
      O     T    123;
      O     ;
      A     M   1000.5;
      A     I    244.5;
      )     ;
      A(    ;
      O     I   1049.1;
      O     I   1048.0;
      )     ;
      A(    ;
      O     I   1057.0;
      O     I   1056.0;
      )     ;
      A     M   1042.6;
      A     M   1044.1;
      AN    M   1044.3;
      AN    Q    218.2;
      =     Q    218.3;
NETWORK
TITLE =

      A(    ;
      A     M   1000.5;
      A     DB51.DBX  207.2;
      A     DB51.DBX  203.6;
      AN    DB51.DBX  203.7;
      O     ;
      A     M   1000.6;
      AN    M   1001.0;
      A(    ;
      A     M   1001.6;
      A     M   1008.0;
      A     M   1040.0;
      A     M   1040.2;
      A     M   1040.6;
      O     ;
      A     M    184.1;
      AN    M   1008.0;
      A     M   1041.1;
      A     M   1001.7;
      )     ;
      O     M   1001.2;
      )     ;
      A(    ;
      O     T    123;
      O     ;
      A     M   1000.5;
      A     I    244.5;
      )     ;
      A(    ;
      O     I   1049.1;
      O     I   1048.0;
      )     ;
      A(    ;
      O     I   1057.0;
      O     I   1056.0;
      )     ;
      AN    M   1044.4;
      AN    Q    218.5;
      =     Q    218.4;
NETWORK
TITLE =

      A(    ;
      A     M   1000.5;
      A     DB51.DBX  207.2;
      AN    DB51.DBX  203.6;
      A     DB51.DBX  203.7;
      O     ;
      A     M   1000.6;
      AN    M   1001.0;
      A     M    184.0;
      AN    M   1008.0;
      A     M   1041.1;
      A     M   1001.7;
      )     ;
      A(    ;
      O     T    123;
      O     ;
      A     M   1000.5;
      A     I    244.5;
      )     ;
      A(    ;
      O     I   1049.1;
      O     I   1048.0;
      )     ;
      A(    ;
      O     I   1057.0;
      O     I   1056.0;
      )     ;
      AN    M   1044.5;
      AN    Q    218.4;
      =     Q    218.5;
NETWORK
TITLE =

      A     Q    218.4;
      AN    T     30;
      O     ;
      A     Q    218.5;
      AN    T     31;
      =     Q    218.6;
END_FUNCTION

FUNCTION FC 123 : VOID
TITLE =
VERSION : 0.1

BEGIN
NETWORK
TITLE =
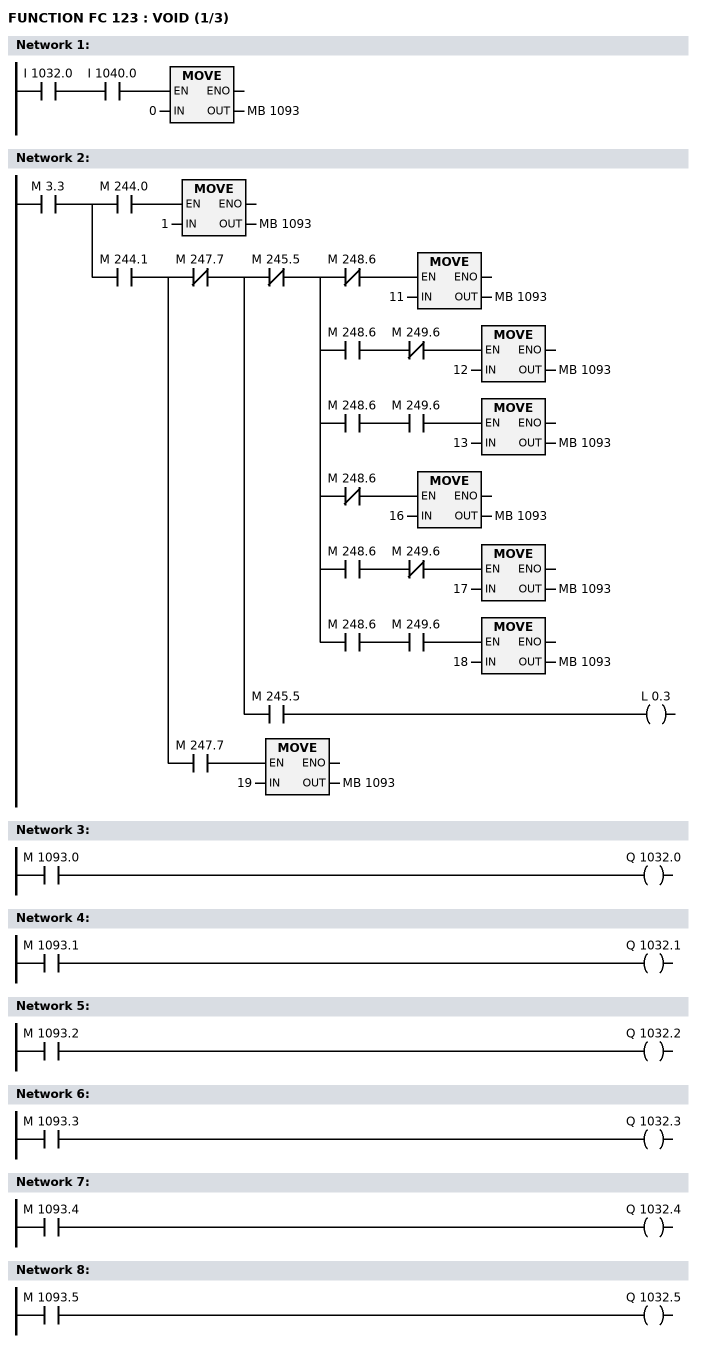

      A     I   1032.0;
      A     I   1040.0;
      JNB   _001;
      L     0;
      T     MB  1093;
_001: NOP   0;
NETWORK
TITLE =

      A     M      3.3;
      =     L      0.0;
      A     L      0.0;
      A     M    244.0;
      JNB   _002;
      L     1;
      T     MB  1093;
_002: NOP   0;
      A     L      0.0;
      A     M    244.1;
      =     L      0.1;
      A     L      0.1;
      AN    M    247.7;
      =     L      0.2;
      A     L      0.2;
      AN    M    245.5;
      =     L      0.3;
      A     L      0.3;
      AN    M    248.6;
      JNB   _003;
      L     11;
      T     MB  1093;
_003: NOP   0;
      A     L      0.3;
      A     M    248.6;
      AN    M    249.6;
      JNB   _004;
      L     12;
      T     MB  1093;
_004: NOP   0;
      A     L      0.3;
      A     M    248.6;
      A     M    249.6;
      JNB   _005;
      L     13;
      T     MB  1093;
_005: NOP   0;
      A     L      0.2;
      A     M    245.5;
      =     L      0.3;
      A     L      0.3;
      AN    M    248.6;
      JNB   _006;
      L     16;
      T     MB  1093;
_006: NOP   0;
      A     L      0.3;
      A     M    248.6;
      AN    M    249.6;
      JNB   _007;
      L     17;
      T     MB  1093;
_007: NOP   0;
      A     L      0.3;
      A     M    248.6;
      A     M    249.6;
      JNB   _008;
      L     18;
      T     MB  1093;
_008: NOP   0;
      A     L      0.1;
      A     M    247.7;
      JNB   _009;
      L     19;
      T     MB  1093;
_009: NOP   0;
NETWORK
TITLE =

      A     M   1093.0;
      =     Q   1032.0;
NETWORK
TITLE =

      A     M   1093.1;
      =     Q   1032.1;
NETWORK
TITLE =

      A     M   1093.2;
      =     Q   1032.2;
NETWORK
TITLE =

      A     M   1093.3;
      =     Q   1032.3;
NETWORK
TITLE =

      A     M   1093.4;
      =     Q   1032.4;
NETWORK
TITLE =

      A     M   1093.5;
      =     Q   1032.5;
NETWORK
TITLE =
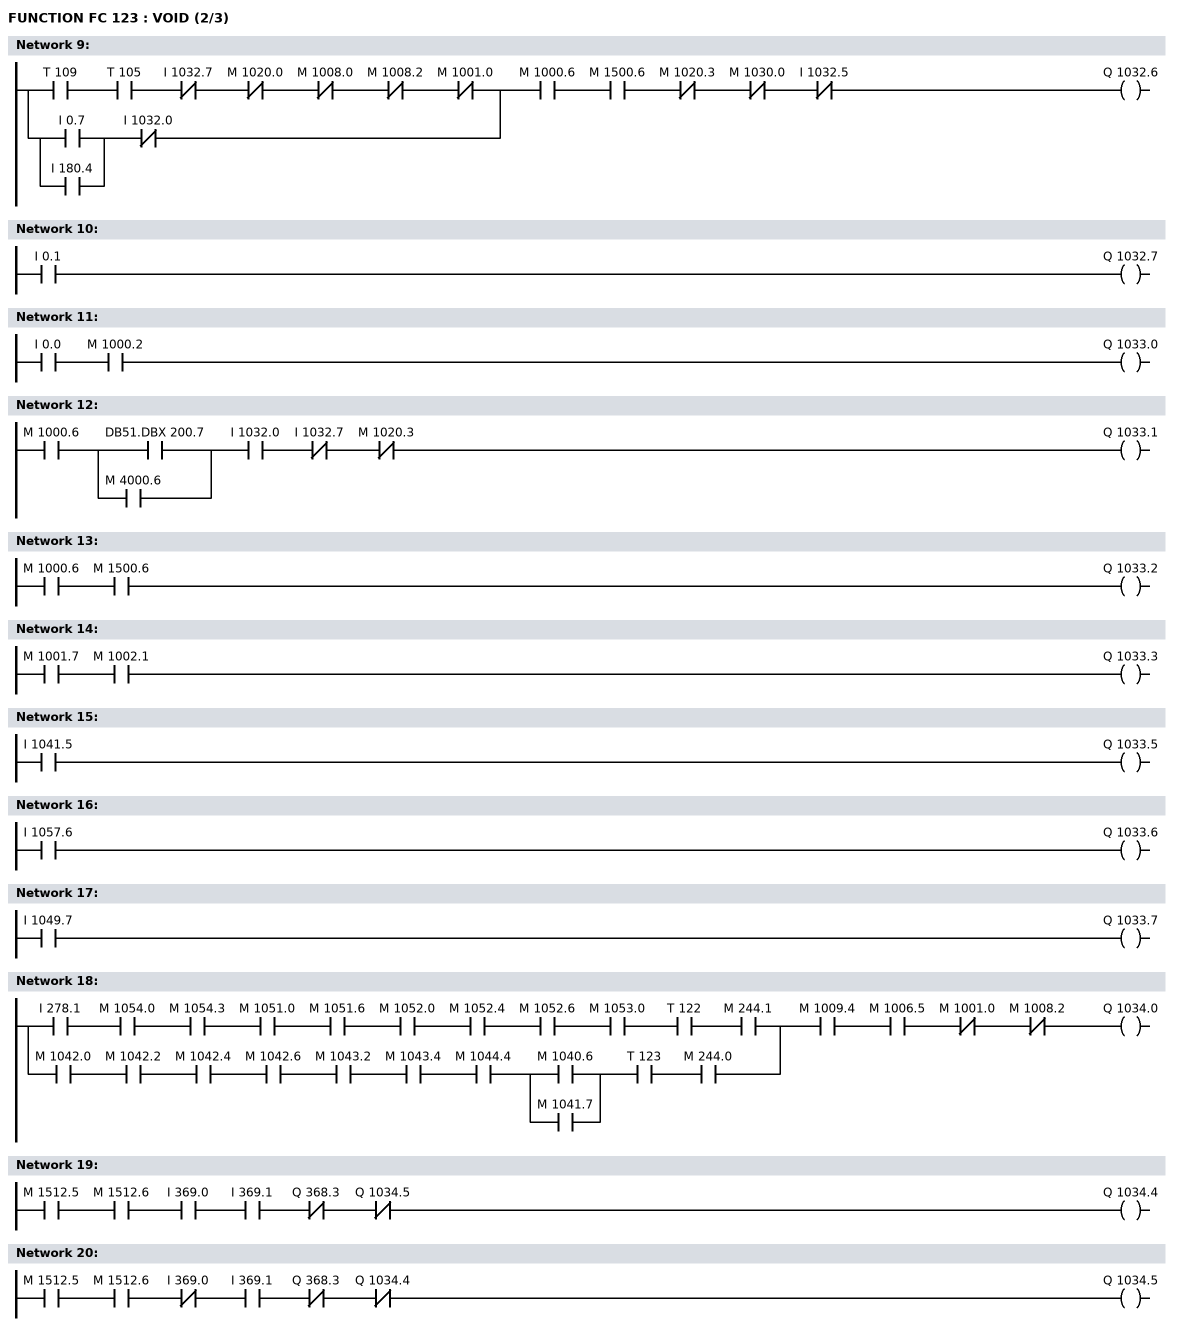

